      -----------------------------------------------------
      Date        Name      Version           Activity                                                                              

   ############################################################*)

   REGION Control Mode
       //AUTO:Auto Mode
       #ioGraphCtrl.AUTO := #ioGraphCtrl.SUP := #iSysInface.Auto.Mode;

       //MAN:Manual Mode
       #ioGraphCtrl.MAN :=  #iSysInface.ManualMode;
       #ioGraphCtrl.OFF := #ioPM_Inface.AlarmImdilyStop OR #iSysInface.ManualMode;
       IF #iSysInface.ManualMode OR #ioPM_Inface.AlarmImdilyStop THEN
           #ioPM_Inface.InitialRun      := 0;
           #ioPM_Inface.InitialOK       := 0;
           #ioPM_Inface.WaitRunning     := 0;
           // #ioPM_Inface.Running         := 0;
           #ioPM_Inface.UnPause    := 0;
           #ioPM_Inface.ProcessComplete := 0;

       END_IF;
       //AutoRunning
       //
       // #ioPM_Inface.Running := ((#iSysInface.Auto.StartAuto AND #iSysInface.Ready) OR #iSysInface.Auto.Running)
       // AND AND NOT "ST10_Sys".Auto.RunningOver 

       IF NOT #iSysInface.ManualMode AND #iSysInface.SysRun AND #ioPM_Inface.InitialOK AND NOT #ioPM_Inface.Alarm
           AND NOT #ioPM_Inface.AlarmImdilyStop AND NOT #iSysInface.Auto.RunningPause THEN
           IF #iSysInface.Auto.StartAuto AND #iSysInface.Ready AND  NOT  #ioPM_Inface.Running  THEN
               #ioPM_Inface.Running := 1;
           END_IF;
       ELSE
           #ioPM_Inface.Running := 0;
       END_IF;

       //Step Num






       //TAP:StepMode
       #ioGraphCtrl.TAP := #iSysInface.Auto.StepMode;
       #ioGraphCtrl.T_PUSH := #iSysInface.Auto.StepMode AND #ioPM_Inface.SetNextStep AND NOT #sHis[0];
       #sHis[0] := #ioPM_Inface.SetNextStep;

       //INTERLOCK
       #ioGraphCtrl.LOCK    := 1;
       #ioGraphCtrl.IL_PERM := 1;
       #ioGraphCtrl.T_PERM  := 1;

   END_REGION

   REGION Initialization

       #sSetInitialDelay(IN := #iSysInface.SetInitial OR #ioPM_Inface.SetInitial,
                         PT := T#2000ms);//20221221DB

       IF #sSetInitialDelay.Q AND #iSysInface.SysRun AND NOT #iSysInface.ManualMode THEN

           IF NOT #sHis[1] THEN
               //     #oStatus.Initializing := TRUE;
               //     #oStatus.InitializeOK := 0;
               //     #oStatus.WaitRunning := 0;
               //     #oStatus.Running := 0;
               //     #oStatus.RunningPause := 0;
               //     #oStatus.RunningFinished := 0;
               #ioGraphCtrl.INIT := #sSetInitialDelay.Q;
           END_IF;

       ELSE
           #ioGraphCtrl.INIT := 0;
       END_IF;
       #sHis[1] := #sSetInitialDelay.Q;
   END_REGION

   REGION Reset
       //
       #ioGraphCtrl.ACK := #iSysInface.Reset;


   END_REGION

   REGION Running and Pause(Halt)
       #ioGraphCtrl.HALT :=(#ioPM_Inface.InitialOK AND NOT #ioPM_Inface.Running )  OR   #ioPM_Inface.Alarm OR #ioPM_Inface.AlarmImdilyStop ; //#ioPM_Inface.UnPause  NOT #iSysInface.Auto.RunningPause
       #ioGraphCtrl.OPS_ZERO := #iSysInface.ManualMode OR NOT #iSysInface.SysRun OR #ioPM_Inface.AlarmImdilyStop ;
       #ioGraphCtrl.TMS_HALT := #iSysInface.ManualMode OR NOT #iSysInface.SysRun OR #ioPM_Inface.AlarmImdilyStop;
   END_REGION


   #S_NEXT_Delay[0](PT := t#3s,
                 IN := #ioGraphCtrl.S_NEXT);

   IF #S_NEXT_Delay[0].Q THEN
       #ioGraphCtrl.S_NEXT := 0;

   END_IF;

   #S_NEXT_Delay[1](PT := t#3s,
                    IN := NOT #ioGraphCtrl.S_NEXT);

   IF #S_NEXT_Delay[1].Q THEN
       #ioGraphCtrl.S_NEXT := 1;
   END_IF;
END_FUNCTION_BLOCK

FUNCTION_BLOCK "ST10_Flow2_A1TableUnloading"   // FB1072, GRAPH
// stored: AcknowledgeErrorsRequired false, AutoNumber false, GraphVersion 6.0, InitialValuesAcquisition false, SetENOAutomatically false
   // inherited from GRAPH_BASE
   VAR_INPUT
      iSysInface : "RCS_SysComInterface_V1";
   END_VAR
   VAR_IN_OUT
      ioPM_Inface : "RCS_PMInterface_V1";
      ioStatus : Int;
   END_VAR
   VAR
      sCtrlMode { S7_SetPoint := 'True'} : "SysFlowCtrlGraph";
      sUpdMES_Data : Bool;   // 更新MES数据
      工件放行中 : Bool;
      前站站号 { ExternalAccessible := 'False'; ExternalVisible := 'False'; ExternalWritable := 'False'} : UInt;
      本站站号 { ExternalAccessible := 'False'; ExternalVisible := 'False'; ExternalWritable := 'False'} : UInt;
      弹窗Temp : Array[1..10] of Int;
      AlarmID : Int;
      TON { S7_SetPoint := 'True'} : Array[0..10] of TON_TIME;
      TOF { S7_SetPoint := 'True'} : Array[0..10] of TOF_TIME;
      sUP { S7_SetPoint := 'True'} : Array[0..10] of Bool;
      更新RFID完成 : Bool;
   END_VAR
   VAR_TEMP
      Tempresult : USInt;
      本站站号乘10 : UInt;
   END_VAR
   // // TON[0] : 托盘流入1托盘到位传感器 / iA-Rotating product Check
   // // TON[1] : 托盘流入1托盘到位传感器
   // // TON[2] : 托盘流入1产品有无传感器
   // // TON[3] : 托盘流入1产品有无传感器
   // // TON[4] : 托盘流入1姿态检测光电2
   // // TON[5] : 托盘流入1姿态检测光电3
   // // TON[0].Q : 托盘流入1托盘到位 / iA-Rotating product Check
   // // TON[1].Q : 托盘流入1托盘无
   // // TON[2].Q : 托盘流入1有产品
   // // TON[3].Q : 托盘流入1无产品
   // // TON[4].Q : 托盘流入1姿态检测光电2
   // // TON[5].Q : 托盘流入1姿态检测光电3
   // // TOF[1] : iA-Rotating product Check
BEGIN
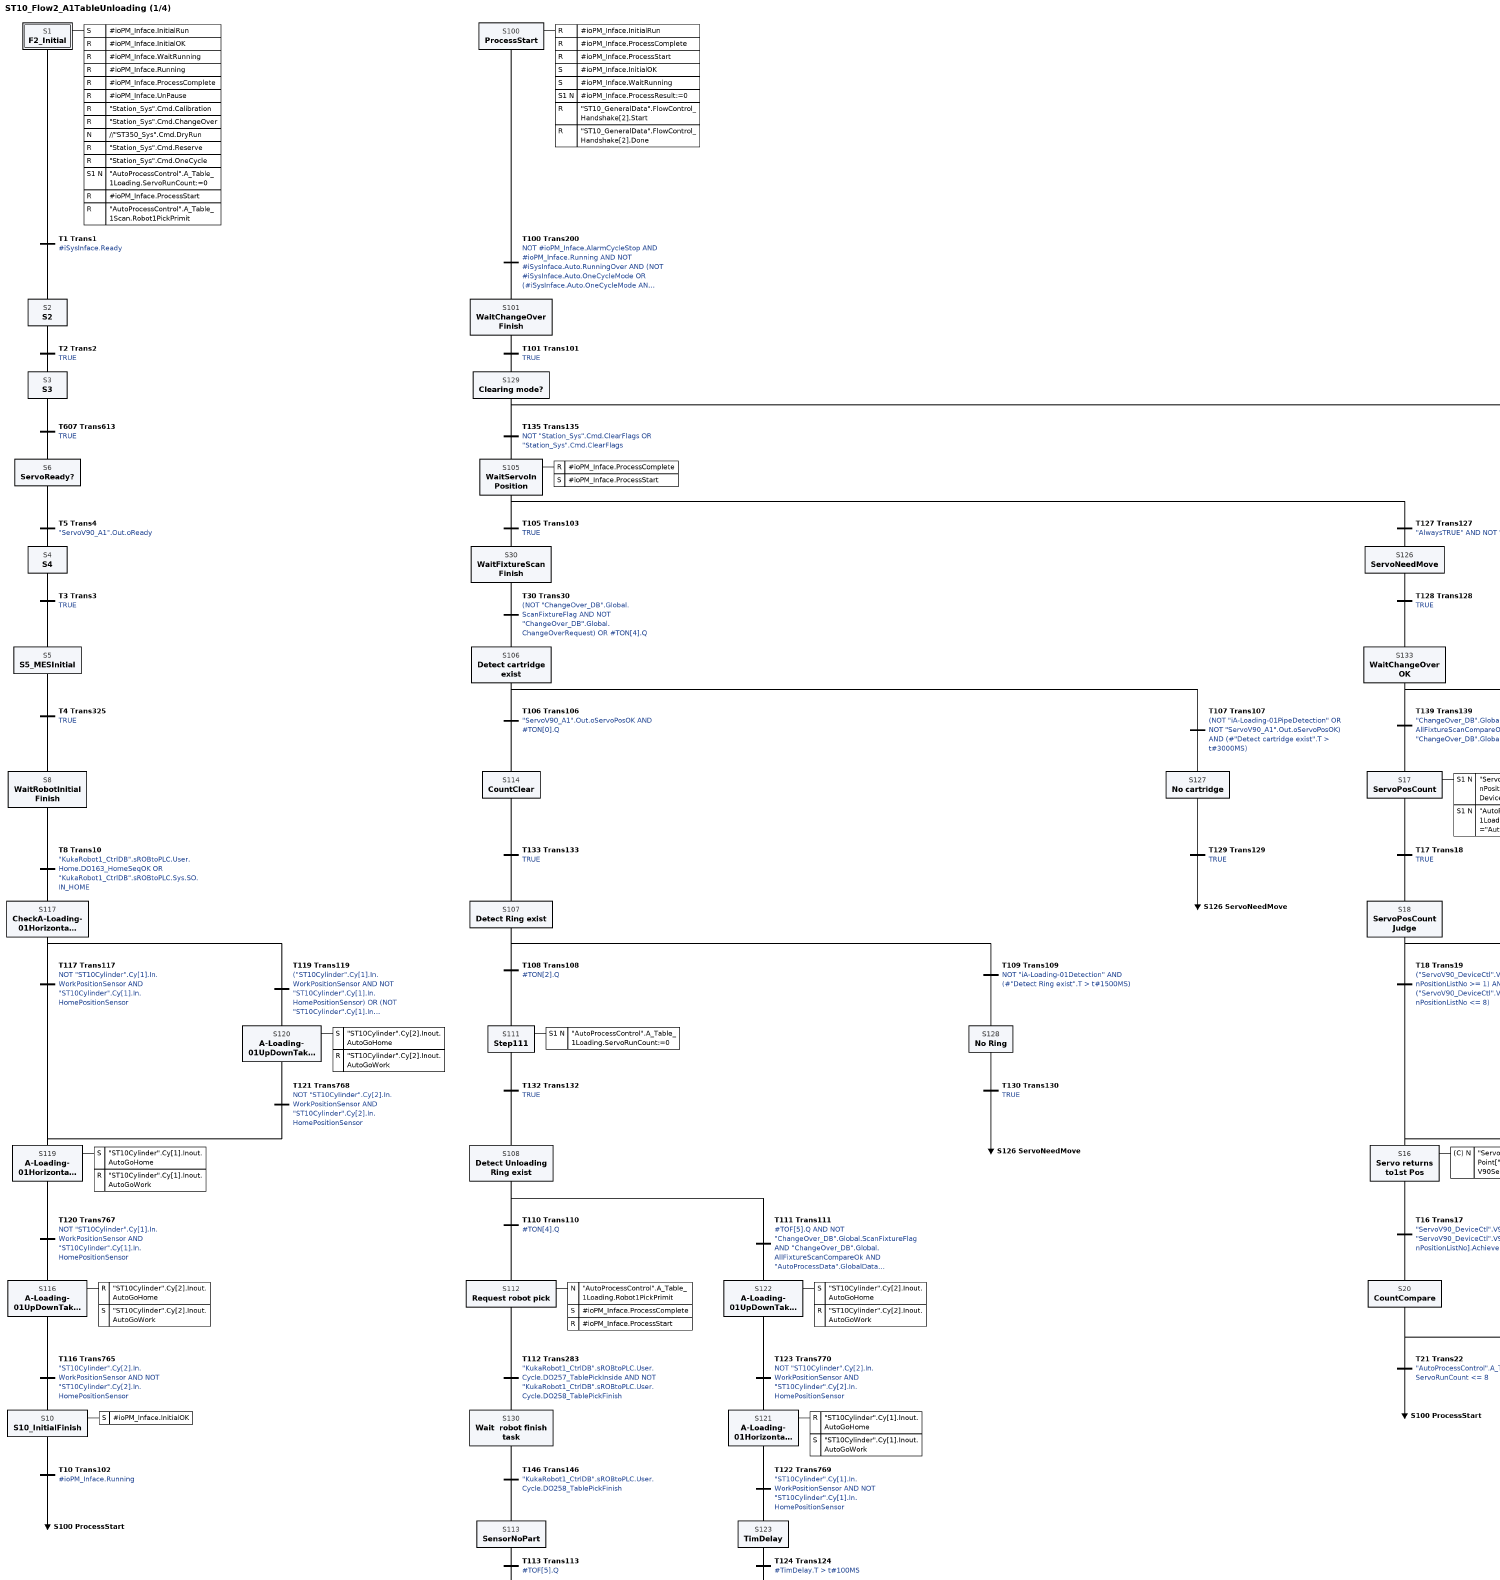
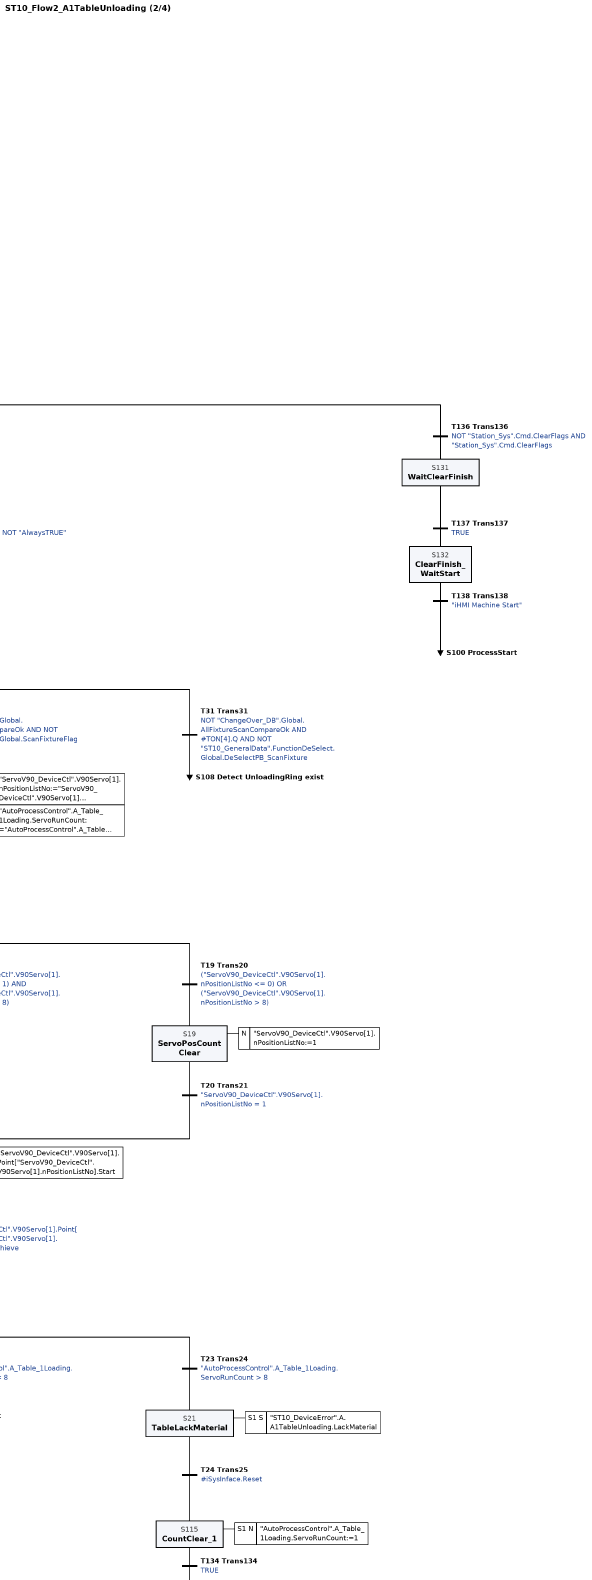
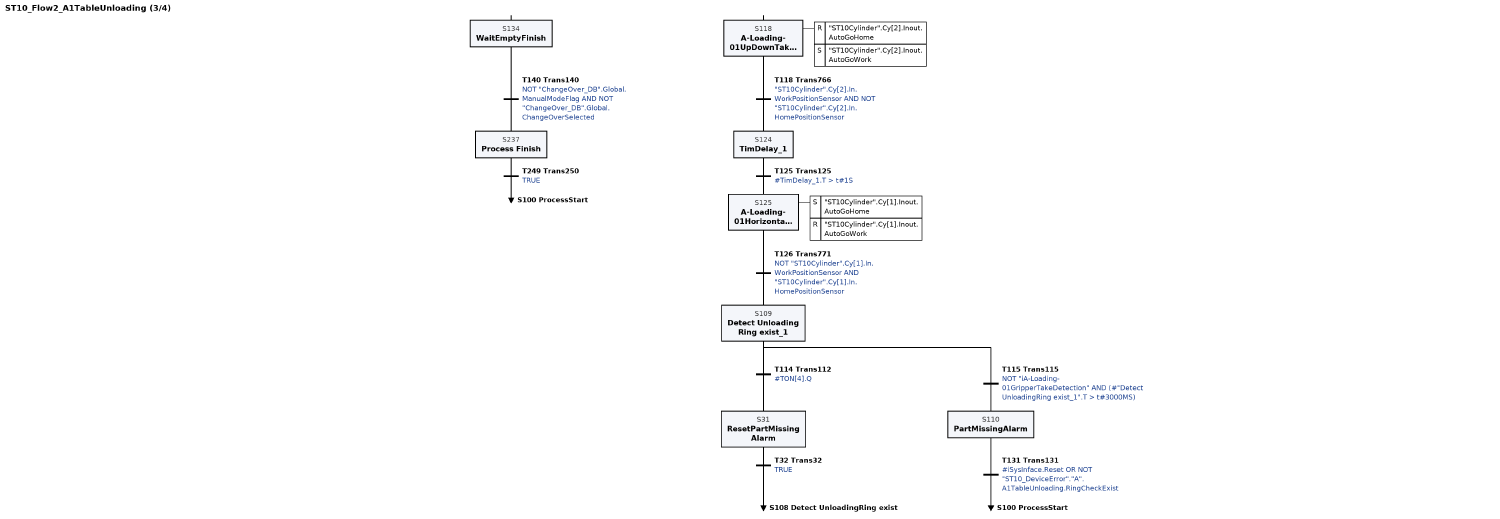
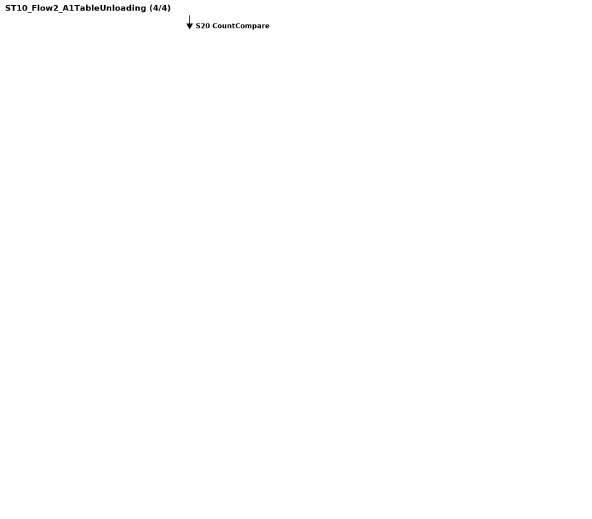
   // permanent pre-instructions
   NETWORK 1
      #TON[10].TON(IN := "AlwaysTRUE" AND "Station_Sys".Alarm.ImmediatelyStop, PT := T#300ms);
      #ioPM_Inface.AlarmImdilyStop := #TON[10].Q;
      #ioPM_Inface.AlarmCycleStop := "AlwaysTRUE" AND "Station_Sys".Alarm.CycleStop;
   NETWORK 2
      IF NOT False THEN
          #sCtrlMode(iSysInface := #iSysInface, ioPM_Inface := #ioPM_Inface, ioGraphCtrl := #RT_DATA.MOP);   // "SysFlowCtrlGraph"
      END_IF;
   NETWORK 3
      #TON[0].TON(IN := "AlwaysTRUE" AND "iA-Loading-01PipeDetection", PT := t#500ms);   // 工位11有托盘
      #TOF[1].TOF(IN := "AlwaysTRUE" AND NOT "iA-Loading-01PipeDetection", PT := T#300ms);   // 工位无托盘
      #TON[2].TON(IN := "AlwaysTRUE" AND "iA-Loading-01Detection", PT := T#300ms);
      #TOF[3].TOF(IN := "AlwaysTRUE" AND NOT "iA-Loading-01Detection", PT := T#300ms);
      #TON[4].TON(IN := "AlwaysTRUE" AND "iA-Loading-01GripperTakeDetection", PT := T#300ms);
      #TOF[5].TOF(IN := "AlwaysTRUE" AND NOT "iA-Loading-01GripperTakeDetection", PT := T#300ms);
   NETWORK 4
      #前站站号 := 345;
      #本站站号 := 350;

   // sequencer 1: S01-S99 初始化 / S01-S99 Initial
   INITIAL_STEP F2_Initial:   // S1, max time T#10S, warning time T#7S
              S    #ioPM_Inface.InitialRun
              R    #ioPM_Inface.InitialOK
              R    #ioPM_Inface.WaitRunning
              R    #ioPM_Inface.Running
              R    #ioPM_Inface.ProcessComplete
              R    #ioPM_Inface.UnPause
              R    "Station_Sys".Cmd.Calibration
              R    "Station_Sys".Cmd.ChangeOver
                   //"ST350_Sys".Cmd.DryRun
              R    "Station_Sys".Cmd.Reserve
              R    "Station_Sys".Cmd.OneCycle
          S1  N    "AutoProcessControl".A_Table_1Loading.ServoRunCount:=0
              R    #ioPM_Inface.ProcessStart
              R    "AutoProcessControl".A_Table_1Scan.Robot1PickPrimit
              R    "AutoProcessControl".A_Table_1Loading.Robot1PickPrimit
              R    "AutoProcessControl".A_Table_2Scan.Robot3PickPrimit
              R    "AutoProcessControl".A_Table_2Loading.Robot3PickPrimit
              R    "AutoProcessControl".A_ScanRotary.Robot1PickPrimit
              R    "AutoProcessControl".A_ScanRotary.Robot1PutPrimit
              R    "AutoProcessControl".H_ShafeLine.Robot1PickPrimit
              R    "AutoProcessControl".J_MagnetLine.Robot2PickPrimit
              R    "AutoProcessControl".K_ShafeLine.Robot2PickPrimit
              R    "AutoProcessControl".L_ShafeLine.Robot3PutPrimit
   END_STEP
   TRANSITION Trans1 FROM F2_Initial TO S2   // T1
      := #iSysInface.Ready;
   END_TRANSITION
   STEP S2:   // S2, max time T#10S, warning time T#7S
   END_STEP
   TRANSITION Trans2 FROM S2 TO S3   // T2
      := TRUE;
   END_TRANSITION
   STEP S4:   // S4, max time T#10S, warning time T#7S
   END_STEP
   TRANSITION Trans3 FROM S4 TO S5_MESInitial   // T3
      := TRUE;
   END_TRANSITION
   STEP S5_MESInitial:   // S5, max time T#10S, warning time T#7S
   END_STEP
   TRANSITION Trans325 FROM S5_MESInitial TO WaitRobotInitialFinish   // T4
      := TRUE;
   END_TRANSITION
   STEP S10_InitialFinish:   // S10, max time T#10S, warning time T#7S
              S    #ioPM_Inface.InitialOK
   END_STEP
   TRANSITION Trans102 FROM S10_InitialFinish TO ProcessStart   // T10, jump
      := #ioPM_Inface.Running;
   END_TRANSITION
   STEP S3:   // S3, max time T#10S, warning time T#7S
   END_STEP
   TRANSITION Trans613 FROM S3 TO "ServoReady?"   // T607
      := TRUE;
   END_TRANSITION
   STEP WaitRobotInitialFinish:   // S8, max time T#10S, warning time T#7S
   END_STEP
   TRANSITION Trans10 FROM WaitRobotInitialFinish TO "CheckA-Loading-01HorizontalCylindePos"   // T8
      := "KukaRobot1_CtrlDB".sROBtoPLC.User.Home.DO163_HomeSeqOK OR "KukaRobot1_CtrlDB".sROBtoPLC.Sys.SO.IN_HOME;
   END_TRANSITION
   STEP "A-Loading-01UpDownTakeCylinderToHP_2":   // S120, max time T#10S, warning time T#7S
              S    "ST10Cylinder".Cy[2].Inout.AutoGoHome
              R    "ST10Cylinder".Cy[2].Inout.AutoGoWork
   END_STEP
   TRANSITION Trans768 FROM "A-Loading-01UpDownTakeCylinderToHP_2" TO "A-Loading-01HorizontalCylinderToHP"   // T121
      := NOT "ST10Cylinder".Cy[2].In.WorkPositionSensor AND "ST10Cylinder".Cy[2].In.HomePositionSensor;
   END_TRANSITION
   STEP "CheckA-Loading-01HorizontalCylindePos":   // S117, max time T#10S, warning time T#7S
   END_STEP
   TRANSITION Trans117 FROM "CheckA-Loading-01HorizontalCylindePos" TO "A-Loading-01HorizontalCylinderToHP"   // T117
      := NOT "ST10Cylinder".Cy[1].In.WorkPositionSensor AND "ST10Cylinder".Cy[1].In.HomePositionSensor;
   END_TRANSITION
   TRANSITION Trans119 FROM "CheckA-Loading-01HorizontalCylindePos" TO "A-Loading-01UpDownTakeCylinderToHP_2"   // T119
      := ("ST10Cylinder".Cy[1].In.WorkPositionSensor AND NOT "ST10Cylinder".Cy[1].In.HomePositionSensor) OR (NOT "ST10Cylinder".Cy[1].In.WorkPositionSensor AND NOT "ST10Cylinder".Cy[1].In.HomePositionSensor);
   END_TRANSITION
   STEP "A-Loading-01HorizontalCylinderToHP":   // S119, max time T#10S, warning time T#7S
              S    "ST10Cylinder".Cy[1].Inout.AutoGoHome
              R    "ST10Cylinder".Cy[1].Inout.AutoGoWork
   END_STEP
   TRANSITION Trans767 FROM "A-Loading-01HorizontalCylinderToHP" TO "A-Loading-01UpDownTakeCylinderToWP"   // T120
      := NOT "ST10Cylinder".Cy[1].In.WorkPositionSensor AND "ST10Cylinder".Cy[1].In.HomePositionSensor;
   END_TRANSITION
   STEP "A-Loading-01UpDownTakeCylinderToWP":   // S116, max time T#10S, warning time T#7S
              R    "ST10Cylinder".Cy[2].Inout.AutoGoHome
              S    "ST10Cylinder".Cy[2].Inout.AutoGoWork
   END_STEP
   TRANSITION Trans765 FROM "A-Loading-01UpDownTakeCylinderToWP" TO S10_InitialFinish   // T116
      := "ST10Cylinder".Cy[2].In.WorkPositionSensor AND NOT "ST10Cylinder".Cy[2].In.HomePositionSensor;
   END_TRANSITION
   STEP "ServoReady?":   // S6, max time T#10S, warning time T#7S
   END_STEP
   TRANSITION Trans4 FROM "ServoReady?" TO S4   // T5
      := "ServoV90_A1".Out.oReady;
   END_TRANSITION

   // sequencer 2: S100-S199 等待到位 / S100-S199 CheckSysStatus
   STEP "A-Loading-01HorizontalCylinderToWP_1":   // S121, max time T#10S, warning time T#7S
              R    "ST10Cylinder".Cy[1].Inout.AutoGoHome
              S    "ST10Cylinder".Cy[1].Inout.AutoGoWork
   END_STEP
   TRANSITION Trans769 FROM "A-Loading-01HorizontalCylinderToWP_1" TO TimDelay   // T122
      := "ST10Cylinder".Cy[1].In.WorkPositionSensor AND NOT "ST10Cylinder".Cy[1].In.HomePositionSensor;
   END_TRANSITION
   STEP "A-Loading-01UpDownTakeCylinderToHP3":   // S122, max time T#10S, warning time T#7S
              S    "ST10Cylinder".Cy[2].Inout.AutoGoHome
              R    "ST10Cylinder".Cy[2].Inout.AutoGoWork
   END_STEP
   TRANSITION Trans770 FROM "A-Loading-01UpDownTakeCylinderToHP3" TO "A-Loading-01HorizontalCylinderToWP_1"   // T123
      := NOT "ST10Cylinder".Cy[2].In.WorkPositionSensor AND "ST10Cylinder".Cy[2].In.HomePositionSensor;
   END_TRANSITION
   STEP TimDelay:   // S123, max time T#10S, warning time T#7S
   END_STEP
   TRANSITION Trans124 FROM TimDelay TO "A-Loading-01UpDownTakeCylinderToWP_1"   // T124
      := #TimDelay.T > t#100MS;
   END_TRANSITION
   STEP SensorNoPart:   // S113, max time T#10S, warning time T#7S
   END_STEP
   TRANSITION Trans113 FROM SensorNoPart TO WaitEmptyFinish   // T113
      := #TOF[5].Q;
   END_TRANSITION
   STEP ProcessStart:   // S100, max time T#10S, warning time T#7S
      // 自动等待开始运行
              R    #ioPM_Inface.InitialRun
              R    #ioPM_Inface.ProcessComplete
              R    #ioPM_Inface.ProcessStart
              S    #ioPM_Inface.InitialOK
              S    #ioPM_Inface.WaitRunning
          S1  N    #ioPM_Inface.ProcessResult:=0
              R    "ST10_GeneralData".FlowControl_Handshake[2].Start
              R    "ST10_GeneralData".FlowControl_Handshake[2].Done
   END_STEP
   TRANSITION Trans200 FROM ProcessStart TO WaitChangeOverFinish   // T100
      := NOT #ioPM_Inface.AlarmCycleStop AND #ioPM_Inface.Running AND NOT #iSysInface.Auto.RunningOver AND (NOT #iSysInface.Auto.OneCycleMode OR (#iSysInface.Auto.OneCycleMode AND #ioPM_Inface.TriggerOneCycle));
   END_TRANSITION
   STEP TimDelay_1:   // S124, max time T#10S, warning time T#7S
   END_STEP
   TRANSITION Trans125 FROM TimDelay_1 TO "A-Loading-01HorizontalCylinderToHP_1"   // T125
      := #TimDelay_1.T > t#1S;
   END_TRANSITION
   STEP "Process Finish":   // S237, max time T#10S, warning time T#7S
   END_STEP
   TRANSITION Trans250 FROM "Process Finish" TO ProcessStart   // T249, jump
      := TRUE;
   END_TRANSITION
   STEP "A-Loading-01HorizontalCylinderToHP_1":   // S125, max time T#10S, warning time T#7S
              S    "ST10Cylinder".Cy[1].Inout.AutoGoHome
              R    "ST10Cylinder".Cy[1].Inout.AutoGoWork
   END_STEP
   TRANSITION Trans771 FROM "A-Loading-01HorizontalCylinderToHP_1" TO "Detect UnloadingRing exist_1"   // T126
      := NOT "ST10Cylinder".Cy[1].In.WorkPositionSensor AND "ST10Cylinder".Cy[1].In.HomePositionSensor;
   END_TRANSITION
   STEP "No cartridge":   // S127, max time T#10S, warning time T#7S
   END_STEP
   TRANSITION Trans129 FROM "No cartridge" TO ServoNeedMove   // T129, jump
      := TRUE;
   END_TRANSITION
   STEP "A-Loading-01UpDownTakeCylinderToWP_1":   // S118, max time T#10S, warning time T#7S
              R    "ST10Cylinder".Cy[2].Inout.AutoGoHome
              S    "ST10Cylinder".Cy[2].Inout.AutoGoWork
   END_STEP
   TRANSITION Trans766 FROM "A-Loading-01UpDownTakeCylinderToWP_1" TO TimDelay_1   // T118
      := "ST10Cylinder".Cy[2].In.WorkPositionSensor AND NOT "ST10Cylinder".Cy[2].In.HomePositionSensor;
   END_TRANSITION
   STEP ServoNeedMove:   // S126, max time T#10S, warning time T#7S
   END_STEP
   TRANSITION Trans128 FROM ServoNeedMove TO WaitChangeOverOK   // T128
      := TRUE;
   END_TRANSITION
   STEP WaitChangeOverFinish:   // S101, max time T#10S, warning time T#7S
   END_STEP
   TRANSITION Trans101 FROM WaitChangeOverFinish TO "Clearing mode?"   // T101
      := TRUE;
   END_TRANSITION
   STEP WaitServoInPosition:   // S105, max time T#10S, warning time T#7S
              R    #ioPM_Inface.ProcessComplete
              S    #ioPM_Inface.ProcessStart
   END_STEP
   TRANSITION Trans103 FROM WaitServoInPosition TO WaitFixtureScanFinish   // T105
      := TRUE;
   END_TRANSITION
   TRANSITION Trans127 FROM WaitServoInPosition TO ServoNeedMove   // T127
      := "AlwaysTRUE" AND NOT "AlwaysTRUE";
   END_TRANSITION
   STEP "Detect cartridge exist":   // S106, max time T#10S, warning time T#7S
   END_STEP
   TRANSITION Trans106 FROM "Detect cartridge exist" TO CountClear   // T106
      := "ServoV90_A1".Out.oServoPosOK AND #TON[0].Q;
   END_TRANSITION
   TRANSITION Trans107 FROM "Detect cartridge exist" TO "No cartridge"   // T107
      := (NOT "iA-Loading-01PipeDetection" OR NOT "ServoV90_A1".Out.oServoPosOK) AND (#"Detect cartridge exist".T > t#3000MS);
   END_TRANSITION
   STEP "Detect UnloadingRing exist":   // S108, max time T#10S, warning time T#7S
   END_STEP
   TRANSITION Trans110 FROM "Detect UnloadingRing exist" TO "Request robot pick"   // T110
      := #TON[4].Q;
   END_TRANSITION
   TRANSITION Trans111 FROM "Detect UnloadingRing exist" TO "A-Loading-01UpDownTakeCylinderToHP3"   // T111
      := #TOF[5].Q AND NOT "ChangeOver_DB".Global.ScanFixtureFlag AND "ChangeOver_DB".Global.AllFixtureScanCompareOk AND "AutoProcessData".GlobalData.Table1CodeOKFlag;
   END_TRANSITION
   STEP "Detect Ring exist":   // S107, max time T#10S, warning time T#7S
   END_STEP
   TRANSITION Trans108 FROM "Detect Ring exist" TO Step111   // T108
      := #TON[2].Q;
   END_TRANSITION
   TRANSITION Trans109 FROM "Detect Ring exist" TO "No Ring"   // T109
      := NOT "iA-Loading-01Detection" AND (#"Detect Ring exist".T > t#1500MS);
   END_TRANSITION
   STEP "Wait  robot finish task":   // S130, max time T#10S, warning time T#7S
   END_STEP
   TRANSITION Trans146 FROM "Wait  robot finish task" TO SensorNoPart   // T146
      := "KukaRobot1_CtrlDB".sROBtoPLC.User.Cycle.DO258_TablePickFinish;
   END_TRANSITION
   STEP "Request robot pick":   // S112, max time T#10S, warning time T#7S
              N    "AutoProcessControl".A_Table_1Loading.Robot1PickPrimit
              S    #ioPM_Inface.ProcessComplete
              R    #ioPM_Inface.ProcessStart
   END_STEP
   TRANSITION Trans283 FROM "Request robot pick" TO "Wait  robot finish task"   // T112
      := "KukaRobot1_CtrlDB".sROBtoPLC.User.Cycle.DO257_TablePickInside AND NOT "KukaRobot1_CtrlDB".sROBtoPLC.User.Cycle.DO258_TablePickFinish;
   END_TRANSITION
   STEP "No Ring":   // S128, max time T#10S, warning time T#7S
   END_STEP
   TRANSITION Trans130 FROM "No Ring" TO ServoNeedMove   // T130, jump
      := TRUE;
   END_TRANSITION
   STEP "Detect UnloadingRing exist_1":   // S109, max time T#10S, warning time T#7S
   END_STEP
   TRANSITION Trans112 FROM "Detect UnloadingRing exist_1" TO ResetPartMissingAlarm   // T114
      := #TON[4].Q;
   END_TRANSITION
   TRANSITION Trans115 FROM "Detect UnloadingRing exist_1" TO PartMissingAlarm   // T115
      := NOT "iA-Loading-01GripperTakeDetection" AND (#"Detect UnloadingRing exist_1".T > t#3000MS);
   END_TRANSITION
   STEP PartMissingAlarm:   // S110, max time T#10S, warning time T#7S
   END_STEP
   TRANSITION Trans131 FROM PartMissingAlarm TO ProcessStart   // T131, jump
      := #iSysInface.Reset OR NOT "ST10_DeviceError"."A".A1TableUnloading.RingCheckExist;
   END_TRANSITION
   STEP Step111:   // S111, max time T#10S, warning time T#7S
          S1  N    "AutoProcessControl".A_Table_1Loading.ServoRunCount:=0
   END_STEP
   TRANSITION Trans132 FROM Step111 TO "Detect UnloadingRing exist"   // T132
      := TRUE;
   END_TRANSITION
   STEP CountClear:   // S114, max time T#10S, warning time T#7S
   END_STEP
   TRANSITION Trans133 FROM CountClear TO "Detect Ring exist"   // T133
      := TRUE;
   END_TRANSITION
   STEP "Servo returns to1st Pos":   // S16, max time T#10S, warning time T#7S
      interlock C := "ServoV90_A1".Out.oReady;
      (C)     N    "ServoV90_DeviceCtl".V90Servo[1].Point["ServoV90_DeviceCtl".V90Servo[1].nPositionListNo].Start
   END_STEP
   TRANSITION Trans17 FROM "Servo returns to1st Pos" TO CountCompare   // T16
      := "ServoV90_DeviceCtl".V90Servo[1].Point["ServoV90_DeviceCtl".V90Servo[1].nPositionListNo].Achieve;
   END_TRANSITION
   STEP ServoPosCount:   // S17, max time T#10S, warning time T#7S
          S1  N    "ServoV90_DeviceCtl".V90Servo[1].nPositionListNo:="ServoV90_DeviceCtl".V90Servo[1].nPositionListNo+1
          S1  N    "AutoProcessControl".A_Table_1Loading.ServoRunCount:="AutoProcessControl".A_Table_1Loading.ServoRunCount+1
   END_STEP
   TRANSITION Trans18 FROM ServoPosCount TO ServoPosCountJudge   // T17
      := TRUE;
   END_TRANSITION
   STEP ServoPosCountJudge:   // S18, max time T#10S, warning time T#7S
   END_STEP
   TRANSITION Trans19 FROM ServoPosCountJudge TO "Servo returns to1st Pos"   // T18
      := ("ServoV90_DeviceCtl".V90Servo[1].nPositionListNo >= 1) AND ("ServoV90_DeviceCtl".V90Servo[1].nPositionListNo <= 8);
   END_TRANSITION
   TRANSITION Trans20 FROM ServoPosCountJudge TO ServoPosCountClear   // T19
      := ("ServoV90_DeviceCtl".V90Servo[1].nPositionListNo <= 0) OR ("ServoV90_DeviceCtl".V90Servo[1].nPositionListNo > 8);
   END_TRANSITION
   STEP ServoPosCountClear:   // S19, max time T#10S, warning time T#7S
              N    "ServoV90_DeviceCtl".V90Servo[1].nPositionListNo:=1
   END_STEP
   TRANSITION Trans21 FROM ServoPosCountClear TO "Servo returns to1st Pos"   // T20
      := "ServoV90_DeviceCtl".V90Servo[1].nPositionListNo = 1;
   END_TRANSITION
   STEP CountCompare:   // S20, max time T#10S, warning time T#7S
   END_STEP
   TRANSITION Trans22 FROM CountCompare TO ProcessStart   // T21, jump
      := "AutoProcessControl".A_Table_1Loading.ServoRunCount <= 8;
   END_TRANSITION
   TRANSITION Trans24 FROM CountCompare TO TableLackMaterial   // T23
      := "AutoProcessControl".A_Table_1Loading.ServoRunCount > 8;
   END_TRANSITION
   STEP TableLackMaterial:   // S21, max time T#10S, warning time T#7S
          S1  S    "ST10_DeviceError".A.A1TableUnloading.LackMaterial
   END_STEP
   TRANSITION Trans25 FROM TableLackMaterial TO CountClear_1   // T24
      := #iSysInface.Reset;
   END_TRANSITION
   STEP CountClear_1:   // S115, max time T#10S, warning time T#7S
          S1  N    "AutoProcessControl".A_Table_1Loading.ServoRunCount:=1
   END_STEP
   TRANSITION Trans134 FROM CountClear_1 TO CountCompare   // T134, jump
      := TRUE;
   END_TRANSITION
   STEP "Clearing mode?":   // S129, max time T#10S, warning time T#7S
   END_STEP
   TRANSITION Trans135 FROM "Clearing mode?" TO WaitServoInPosition   // T135
      := NOT "Station_Sys".Cmd.ClearFlags OR "Station_Sys".Cmd.ClearFlags;
   END_TRANSITION
   TRANSITION Trans136 FROM "Clearing mode?" TO WaitClearFinish   // T136
      := NOT "Station_Sys".Cmd.ClearFlags AND "Station_Sys".Cmd.ClearFlags;
   END_TRANSITION
   STEP WaitClearFinish:   // S131, max time T#10S, warning time T#7S
   END_STEP
   TRANSITION Trans137 FROM WaitClearFinish TO ClearFinish_WaitStart   // T137
      := TRUE;
   END_TRANSITION
   STEP ClearFinish_WaitStart:   // S132, max time T#10S, warning time T#7S
   END_STEP
   TRANSITION Trans138 FROM ClearFinish_WaitStart TO ProcessStart   // T138, jump
      := "iHMI Machine Start";
   END_TRANSITION
   STEP WaitChangeOverOK:   // S133, max time T#10S, warning time T#7S
   END_STEP
   TRANSITION Trans139 FROM WaitChangeOverOK TO ServoPosCount   // T139
      := "ChangeOver_DB".Global.AllFixtureScanCompareOk AND NOT "ChangeOver_DB".Global.ScanFixtureFlag;
   END_TRANSITION
   TRANSITION Trans31 FROM WaitChangeOverOK TO "Detect UnloadingRing exist"   // T31, jump
      := NOT "ChangeOver_DB".Global.AllFixtureScanCompareOk AND #TON[4].Q AND NOT "ST10_GeneralData".FunctionDeSelect.Global.DeSelectPB_ScanFixture;
   END_TRANSITION
   STEP WaitEmptyFinish:   // S134, max time T#10S, warning time T#7S
   END_STEP
   TRANSITION Trans140 FROM WaitEmptyFinish TO "Process Finish"   // T140
      := NOT "ChangeOver_DB".Global.ManualModeFlag AND NOT "ChangeOver_DB".Global.ChangeOverSelected;
   END_TRANSITION
   STEP WaitFixtureScanFinish:   // S30, max time T#10S, warning time T#7S
   END_STEP
   TRANSITION Trans30 FROM WaitFixtureScanFinish TO "Detect cartridge exist"   // T30
      := (NOT "ChangeOver_DB".Global.ScanFixtureFlag AND NOT "ChangeOver_DB".Global.ChangeOverRequest) OR #TON[4].Q;
   END_TRANSITION
   STEP ResetPartMissingAlarm:   // S31, max time T#10S, warning time T#7S
   END_STEP
   TRANSITION Trans32 FROM ResetPartMissingAlarm TO "Detect UnloadingRing exist"   // T32, jump
      := TRUE;
   END_TRANSITION

   // permanent post-instructions
   NETWORK 1
      #ioPM_Inface.StepNum := #RT_DATA.S_DISPLAY;
   NETWORK 2
      IF #iSysInface.Reset THEN #AlarmID := 0; END_IF;
   NETWORK 3
      #TON[10].TON(IN := #工件放行中, PT := T#0.5S);
      IF #TON[10].Q THEN #工件放行中 := FALSE; END_IF;
END_FUNCTION_BLOCK

FUNCTION_BLOCK "ST10_Flow3_A1RotaryShaftScan"   // FB1073, GRAPH
// stored: AcknowledgeErrorsRequired false, AutoNumber false, GraphVersion 6.0, InitialValuesAcquisition false, SetENOAutomatically false
   // inherited from GRAPH_BASE
   VAR_INPUT
      iSysInface : "RCS_SysComInterface_V1";
   END_VAR
   VAR_IN_OUT
      ioPM_Inface : "RCS_PMInterface_V1";
      ioStatus : Int;
   END_VAR
   VAR
      sCtrlMode { S7_SetPoint := 'True'} : "SysFlowCtrlGraph";
      sUpdMES_Data : Bool;   // 更新MES数据
      工件放行中 : Bool;
      前站站号 { ExternalAccessible := 'False'; ExternalVisible := 'False'; ExternalWritable := 'False'} : UInt;
      本站站号 { ExternalAccessible := 'False'; ExternalVisible := 'False'; ExternalWritable := 'False'} : UInt;
      弹窗Temp : Array[1..10] of Int;
      AlarmID : Int;
      TON { S7_SetPoint := 'True'} : Array[0..10] of TON_TIME;
      TOF { S7_SetPoint := 'True'} : Array[0..10] of TOF_TIME;
      sUP { S7_SetPoint := 'True'} : Array[0..10] of Bool;
      更新RFID完成 : Bool;
   END_VAR
   VAR_TEMP
      Tempresult : USInt;
      本站站号乘10 : UInt;
   END_VAR
   // // TON[0] : 托盘流入1托盘到位传感器 / iA-Rotating product Check
   // // TON[1] : 托盘流入1托盘到位传感器
   // // TON[2] : 托盘流入1产品有无传感器
   // // TON[3] : 托盘流入1产品有无传感器
   // // TON[4] : 托盘流入1姿态检测光电2
   // // TON[5] : 托盘流入1姿态检测光电3
   // // TON[0].Q : 托盘流入1托盘到位 / iA-Rotating product Check
   // // TON[1].Q : 托盘流入1托盘无
   // // TON[2].Q : 托盘流入1有产品
   // // TON[3].Q : 托盘流入1无产品
   // // TON[4].Q : 托盘流入1姿态检测光电2
   // // TON[5].Q : 托盘流入1姿态检测光电3
   // // TOF[1] : iA-Rotating product Check
BEGIN
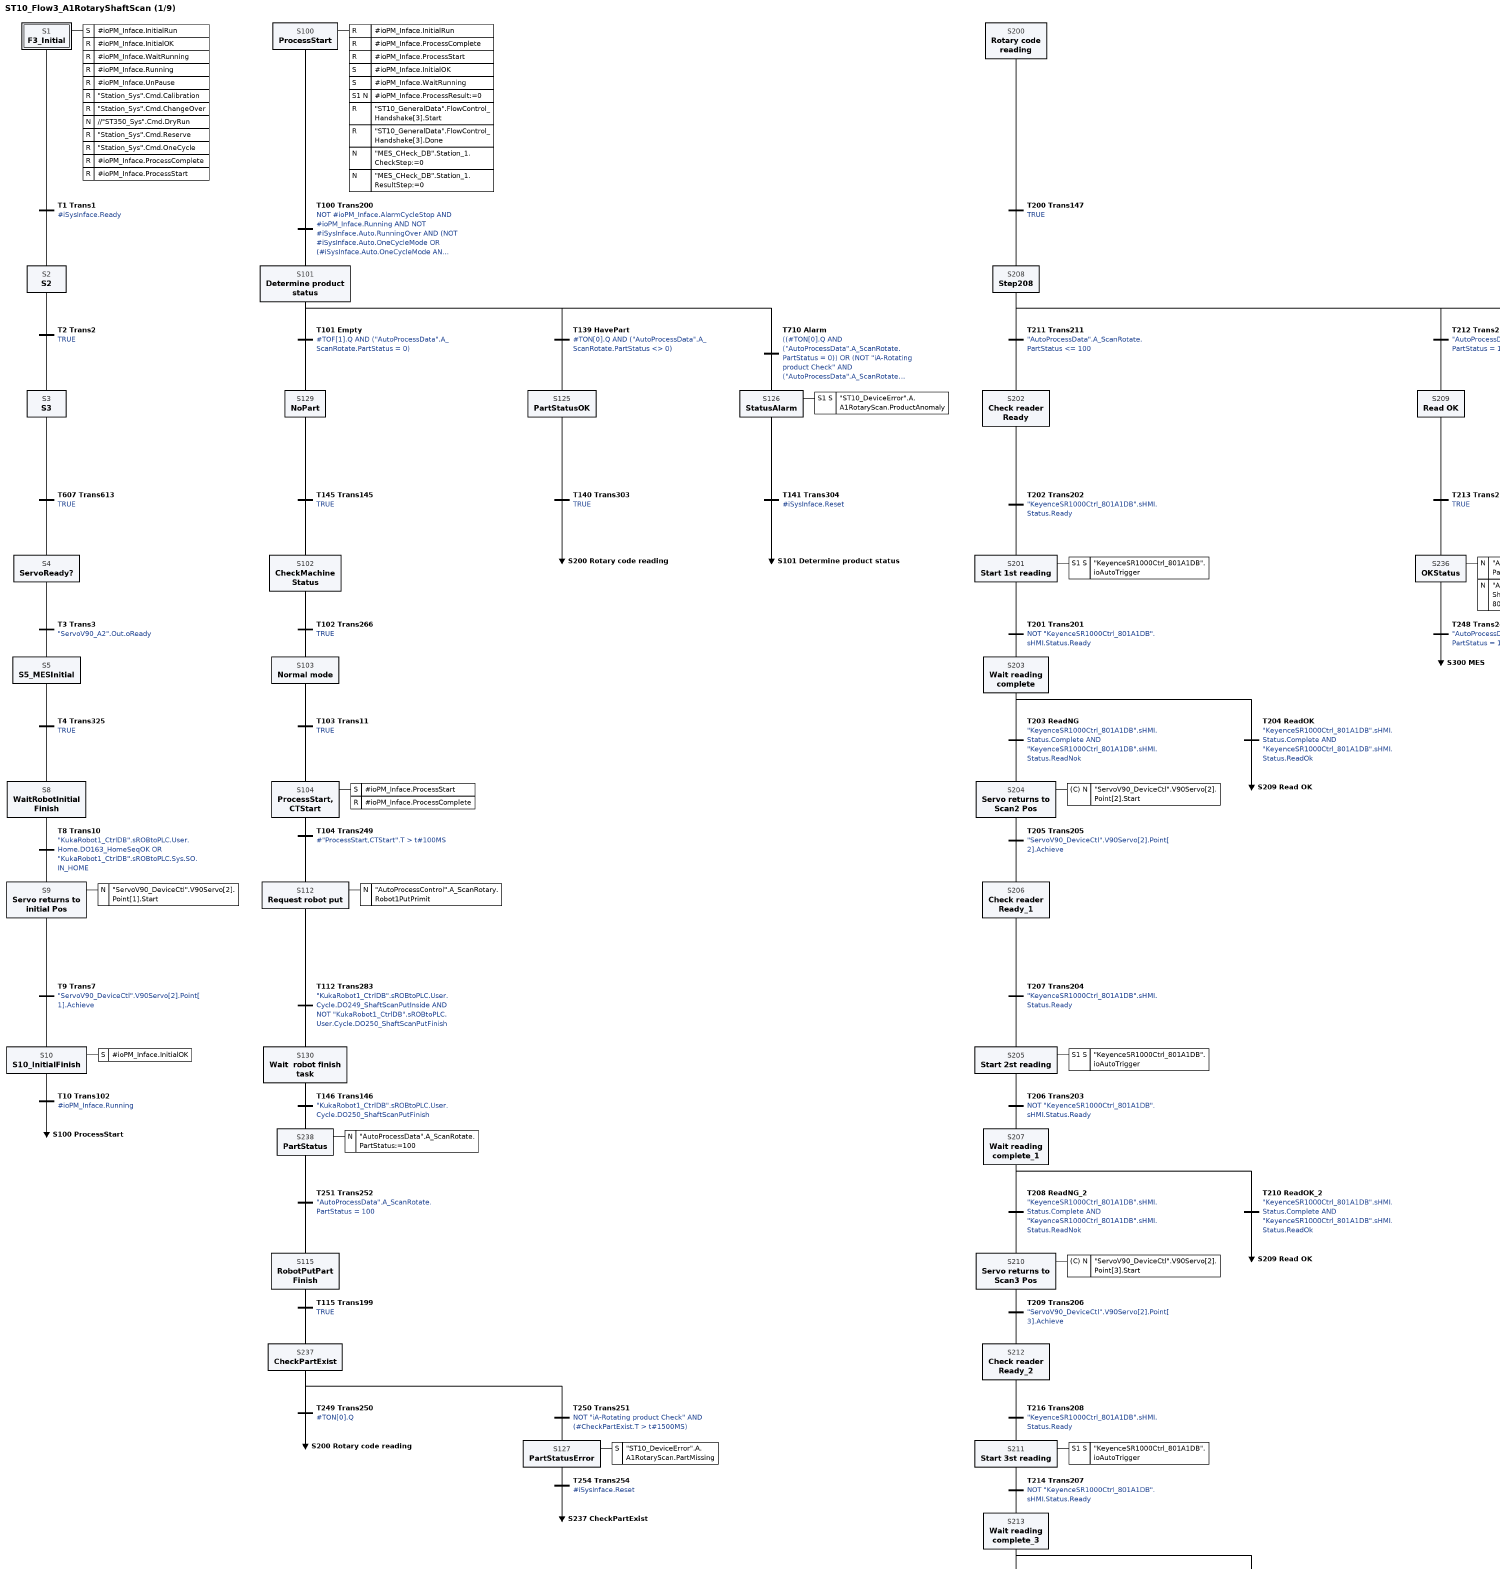
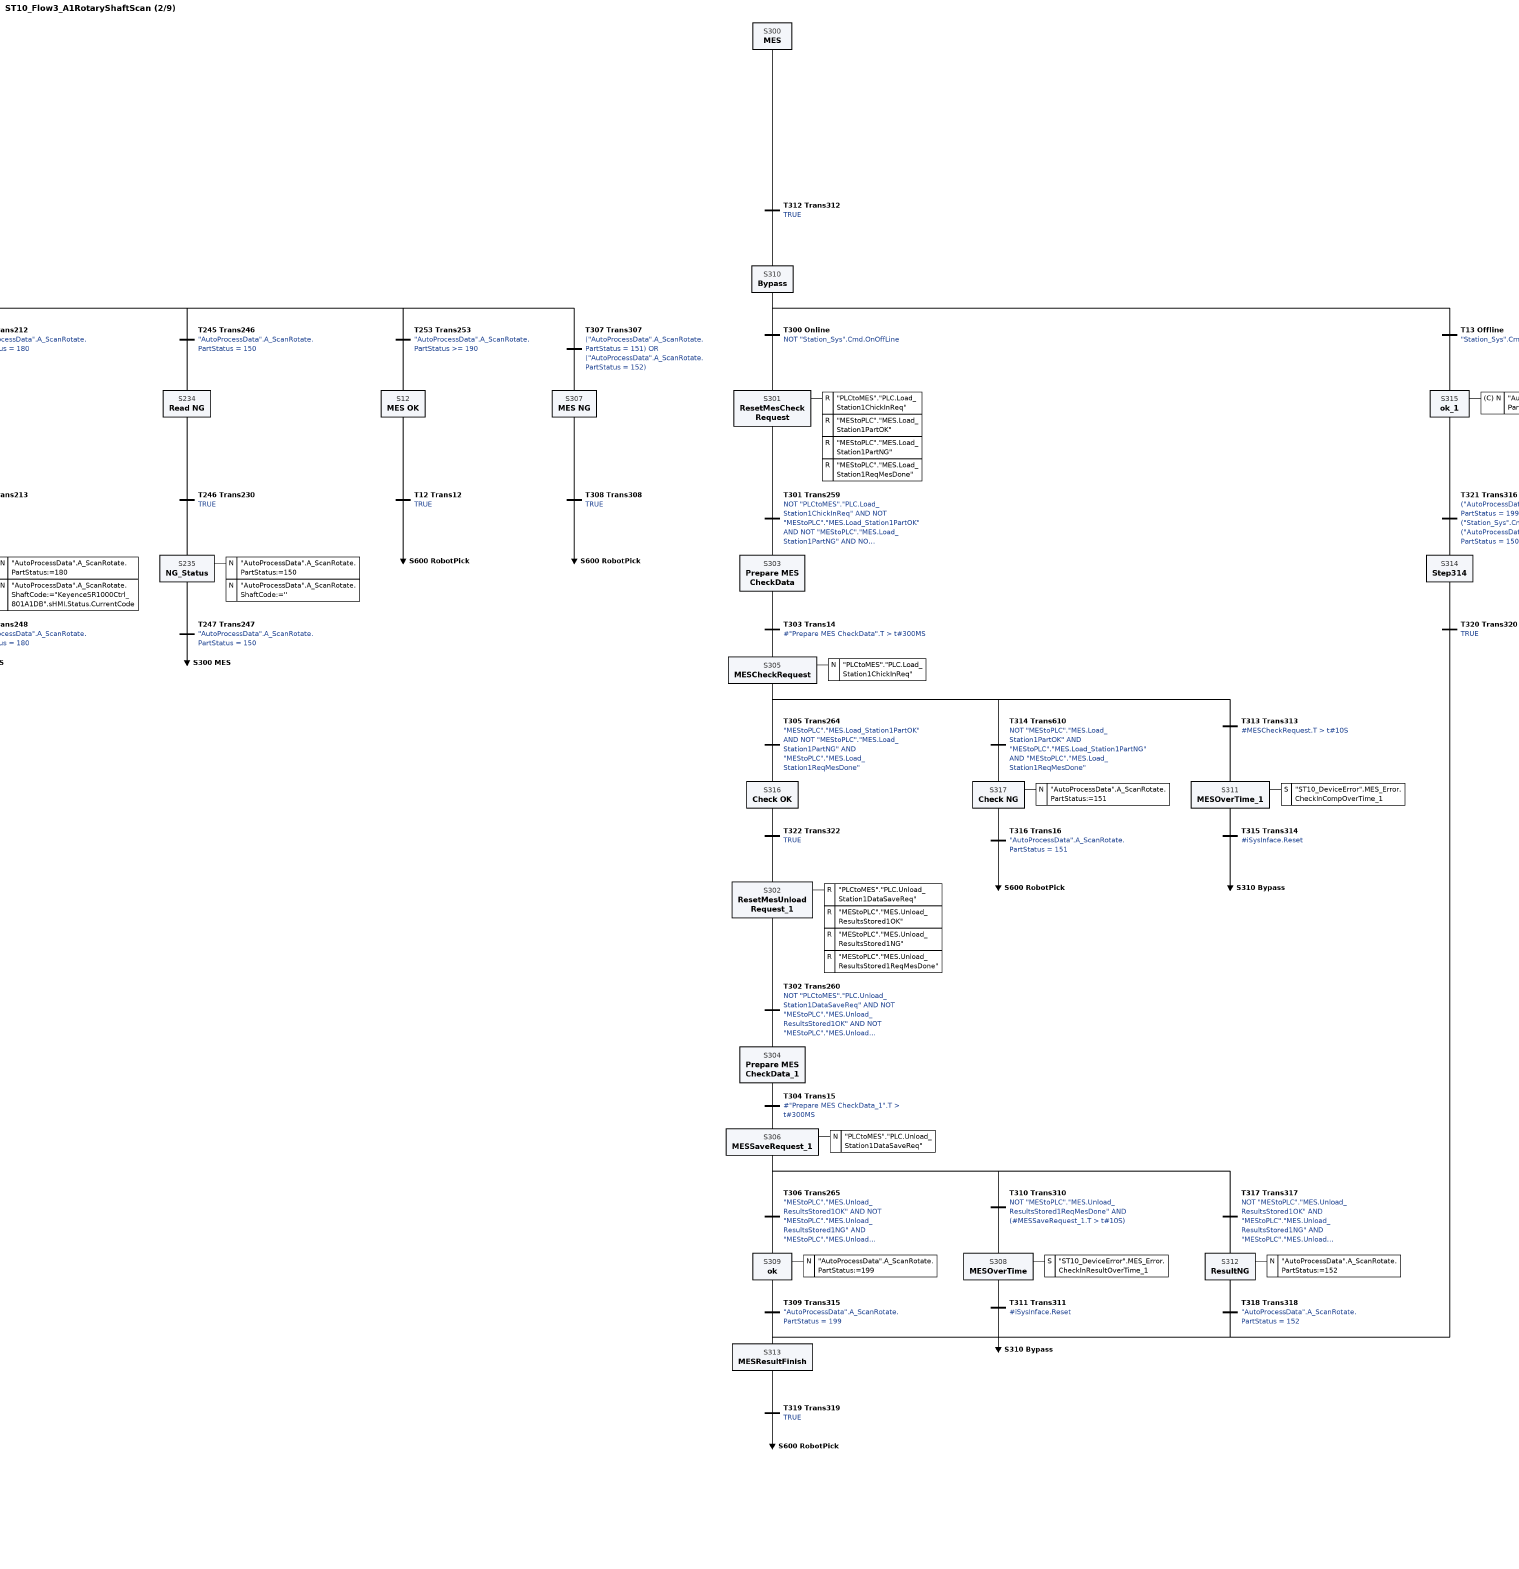
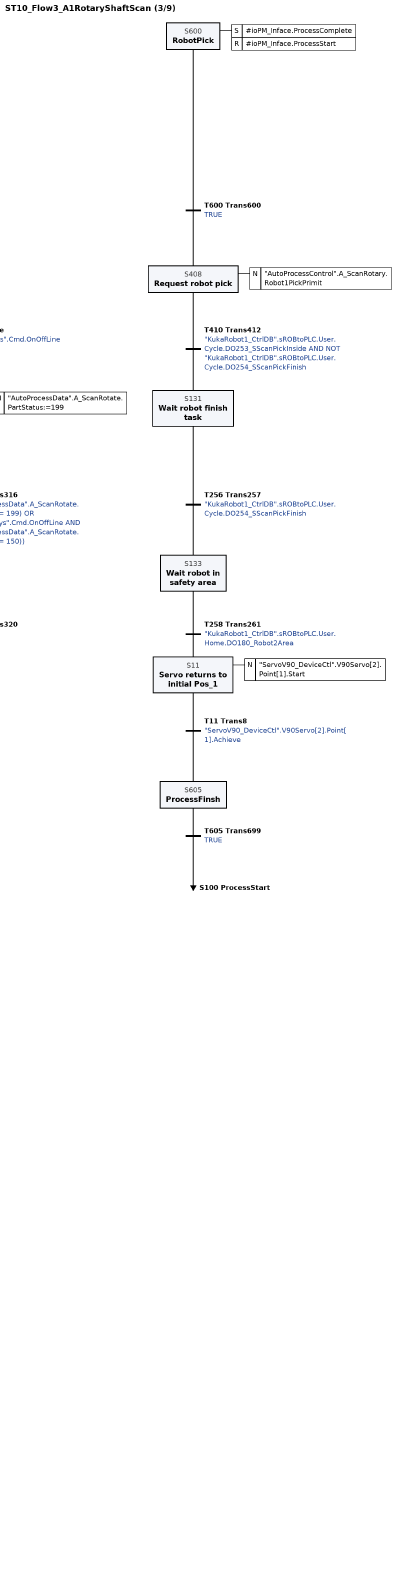
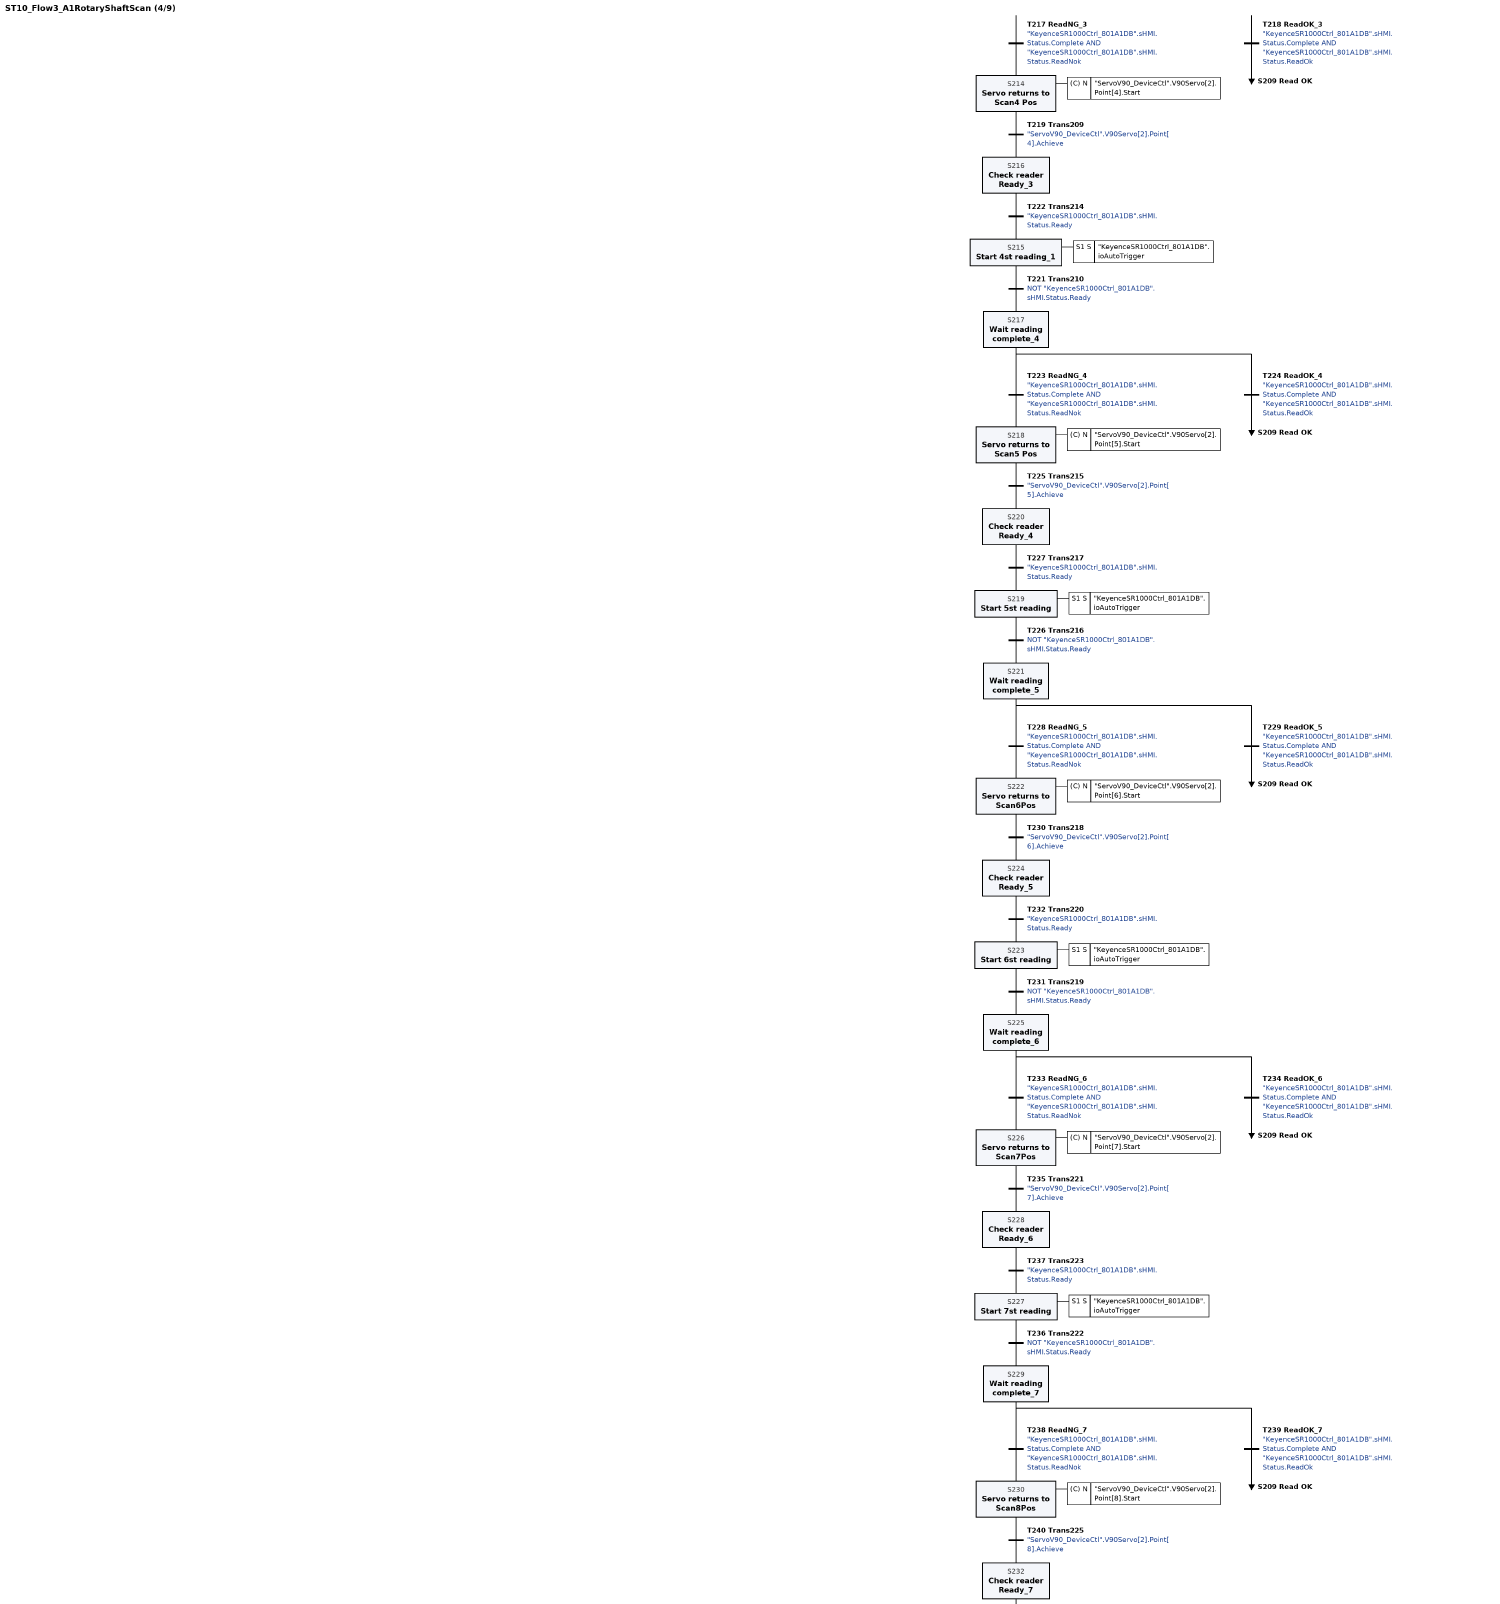
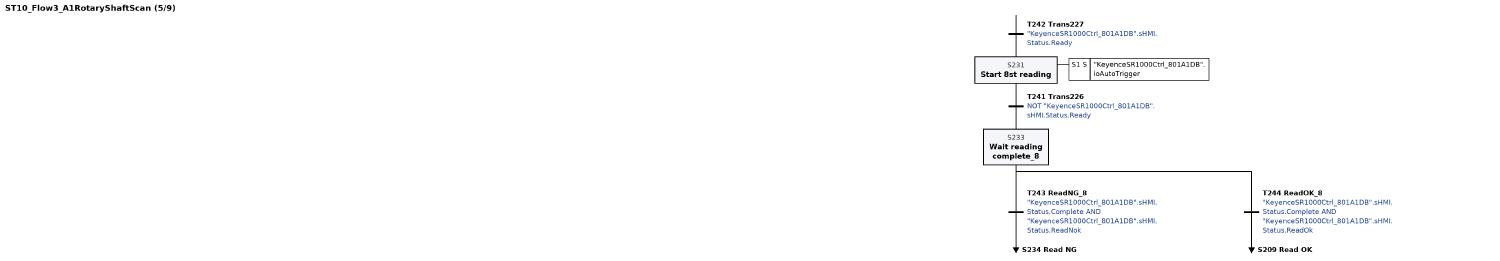
   // permanent pre-instructions
   NETWORK 1
      #TON[10].TON(IN := "AlwaysTRUE" AND "Station_Sys".Alarm.ImmediatelyStop, PT := T#300ms);
      #ioPM_Inface.AlarmImdilyStop := #TON[10].Q;
      #ioPM_Inface.AlarmCycleStop := "AlwaysTRUE" AND "Station_Sys".Alarm.CycleStop;
   NETWORK 2
      IF NOT False THEN
          #sCtrlMode(iSysInface := #iSysInface, ioPM_Inface := #ioPM_Inface, ioGraphCtrl := #RT_DATA.MOP);   // "SysFlowCtrlGraph"
      END_IF;
   NETWORK 3
      #TON[0].TON(IN := "AlwaysTRUE" AND "iA-Rotating product Check", PT := t#500ms);   // 工位11有托盘
      #TOF[1].TOF(IN := "AlwaysTRUE" AND NOT "iA-Rotating product Check", PT := T#300ms);   // 工位无托盘
      #TON[2].TON(IN := "AlwaysTRUE", PT := T#300ms);
      #TON[3].TON(IN := "AlwaysTRUE", PT := T#300ms);
      #TON[4].TON(IN := "AlwaysTRUE", PT := T#300ms);
      #TON[5].TON(IN := "AlwaysTRUE", PT := T#300ms);
   NETWORK 4
      #前站站号 := 345;
      #本站站号 := 350;

   // sequencer 1: S01-S99 初始化 / S01-S99 Initial
   INITIAL_STEP F3_Initial:   // S1, max time T#10S, warning time T#7S
              S    #ioPM_Inface.InitialRun
              R    #ioPM_Inface.InitialOK
              R    #ioPM_Inface.WaitRunning
              R    #ioPM_Inface.Running
              R    #ioPM_Inface.UnPause
              R    "Station_Sys".Cmd.Calibration
              R    "Station_Sys".Cmd.ChangeOver
                   //"ST350_Sys".Cmd.DryRun
              R    "Station_Sys".Cmd.Reserve
              R    "Station_Sys".Cmd.OneCycle
              R    #ioPM_Inface.ProcessComplete
              R    #ioPM_Inface.ProcessStart
   END_STEP
   TRANSITION Trans1 FROM F3_Initial TO S2   // T1
      := #iSysInface.Ready;
   END_TRANSITION
   STEP S2:   // S2, max time T#10S, warning time T#7S
   END_STEP
   TRANSITION Trans2 FROM S2 TO S3   // T2
      := TRUE;
   END_TRANSITION
   STEP "ServoReady?":   // S4, max time T#10S, warning time T#7S
   END_STEP
   TRANSITION Trans3 FROM "ServoReady?" TO S5_MESInitial   // T3
      := "ServoV90_A2".Out.oReady;
   END_TRANSITION
   STEP S5_MESInitial:   // S5, max time T#10S, warning time T#7S
   END_STEP
   TRANSITION Trans325 FROM S5_MESInitial TO WaitRobotInitialFinish   // T4
      := TRUE;
   END_TRANSITION
   STEP S10_InitialFinish:   // S10, max time T#10S, warning time T#7S
              S    #ioPM_Inface.InitialOK
   END_STEP
   TRANSITION Trans102 FROM S10_InitialFinish TO ProcessStart   // T10, jump
      := #ioPM_Inface.Running;
   END_TRANSITION
   STEP S3:   // S3, max time T#10S, warning time T#7S
   END_STEP
   TRANSITION Trans613 FROM S3 TO "ServoReady?"   // T607
      := TRUE;
   END_TRANSITION
   STEP WaitRobotInitialFinish:   // S8, max time T#10S, warning time T#7S
   END_STEP
   TRANSITION Trans10 FROM WaitRobotInitialFinish TO "Servo returns to initial Pos"   // T8
      := "KukaRobot1_CtrlDB".sROBtoPLC.User.Home.DO163_HomeSeqOK OR "KukaRobot1_CtrlDB".sROBtoPLC.Sys.SO.IN_HOME;
   END_TRANSITION
   STEP "Servo returns to initial Pos":   // S9, max time T#10S, warning time T#7S
              N    "ServoV90_DeviceCtl".V90Servo[2].Point[1].Start
   END_STEP
   TRANSITION Trans7 FROM "Servo returns to initial Pos" TO S10_InitialFinish   // T9
      := "ServoV90_DeviceCtl".V90Servo[2].Point[1].Achieve;
   END_TRANSITION

   // sequencer 2: S100-S199 等待到位 / S100-S199 CheckPartStatus
   STEP "Wait  robot finish task":   // S130, max time T#10S, warning time T#7S
   END_STEP
   TRANSITION Trans146 FROM "Wait  robot finish task" TO PartStatus   // T146
      := "KukaRobot1_CtrlDB".sROBtoPLC.User.Cycle.DO250_ShaftScanPutFinish;
   END_TRANSITION
   STEP CheckMachineStatus:   // S102, max time T#10S, warning time T#7S
   END_STEP
   TRANSITION Trans266 FROM CheckMachineStatus TO "Normal mode"   // T102
      := TRUE;
   END_TRANSITION
   STEP "Normal mode":   // S103, max time T#10S, warning time T#7S
   END_STEP
   TRANSITION Trans11 FROM "Normal mode" TO "ProcessStart,CTStart"   // T103
      := TRUE;
   END_TRANSITION
   STEP RobotPutPartFinish:   // S115, max time T#10S, warning time T#7S
   END_STEP
   TRANSITION Trans199 FROM RobotPutPartFinish TO CheckPartExist   // T115
      := TRUE;
   END_TRANSITION
   STEP ProcessStart:   // S100, max time T#10S, warning time T#7S
      // 自动等待开始运行
              R    #ioPM_Inface.InitialRun
              R    #ioPM_Inface.ProcessComplete
              R    #ioPM_Inface.ProcessStart
              S    #ioPM_Inface.InitialOK
              S    #ioPM_Inface.WaitRunning
          S1  N    #ioPM_Inface.ProcessResult:=0
              R    "ST10_GeneralData".FlowControl_Handshake[3].Start
              R    "ST10_GeneralData".FlowControl_Handshake[3].Done
              N    "MES_CHeck_DB".Station_1.CheckStep:=0
              N    "MES_CHeck_DB".Station_1.ResultStep:=0
   END_STEP
   TRANSITION Trans200 FROM ProcessStart TO "Determine product status"   // T100
      := NOT #ioPM_Inface.AlarmCycleStop AND #ioPM_Inface.Running AND NOT #iSysInface.Auto.RunningOver AND (NOT #iSysInface.Auto.OneCycleMode OR (#iSysInface.Auto.OneCycleMode AND #ioPM_Inface.TriggerOneCycle));
   END_TRANSITION
   STEP "ProcessStart,CTStart":   // S104, max time T#10S, warning time T#7S
              S    #ioPM_Inface.ProcessStart
              R    #ioPM_Inface.ProcessComplete
   END_STEP
   TRANSITION Trans249 FROM "ProcessStart,CTStart" TO "Request robot put"   // T104
      := #"ProcessStart,CTStart".T > t#100MS;
   END_TRANSITION
   STEP CheckPartExist:   // S237, max time T#10S, warning time T#7S
   END_STEP
   TRANSITION Trans250 FROM CheckPartExist TO "Rotary code reading"   // T249, jump
      := #TON[0].Q;
   END_TRANSITION
   TRANSITION Trans251 FROM CheckPartExist TO PartStatusError   // T250
      := NOT "iA-Rotating product Check" AND (#CheckPartExist.T > t#1500MS);
   END_TRANSITION
   STEP "Request robot put":   // S112, max time T#10S, warning time T#7S
              N    "AutoProcessControl".A_ScanRotary.Robot1PutPrimit
   END_STEP
   TRANSITION Trans283 FROM "Request robot put" TO "Wait  robot finish task"   // T112
      := "KukaRobot1_CtrlDB".sROBtoPLC.User.Cycle.DO249_ShaftScanPutInside AND NOT "KukaRobot1_CtrlDB".sROBtoPLC.User.Cycle.DO250_ShaftScanPutFinish;
   END_TRANSITION
   STEP PartStatusError:   // S127, max time T#10S, warning time T#7S
              S    "ST10_DeviceError".A.A1RotaryScan.PartMissing
   END_STEP
   TRANSITION Trans254 FROM PartStatusError TO CheckPartExist   // T254, jump
      := #iSysInface.Reset;
   END_TRANSITION
   STEP PartStatus:   // S238, max time T#10S, warning time T#7S
              N    "AutoProcessData".A_ScanRotate.PartStatus:=100
   END_STEP
   TRANSITION Trans252 FROM PartStatus TO RobotPutPartFinish   // T251
      := "AutoProcessData".A_ScanRotate.PartStatus = 100;
   END_TRANSITION
   STEP "Determine product status":   // S101, max time T#10S, warning time T#7S
   END_STEP
   TRANSITION Empty FROM "Determine product status" TO NoPart   // T101
      := #TOF[1].Q AND ("AutoProcessData".A_ScanRotate.PartStatus = 0);
   END_TRANSITION
   TRANSITION HavePart FROM "Determine product status" TO PartStatusOK   // T139
      := #TON[0].Q AND ("AutoProcessData".A_ScanRotate.PartStatus <> 0);
   END_TRANSITION
   TRANSITION Alarm FROM "Determine product status" TO StatusAlarm   // T710
      := ((#TON[0].Q AND ("AutoProcessData".A_ScanRotate.PartStatus = 0)) OR (NOT "iA-Rotating product Check" AND ("AutoProcessData".A_ScanRotate.PartStatus <> 0))) AND (#"Determine product status".T > t#1500MS);
   END_TRANSITION
   STEP PartStatusOK:   // S125, max time T#10S, warning time T#7S
   END_STEP
   TRANSITION Trans303 FROM PartStatusOK TO "Rotary code reading"   // T140, jump
      := TRUE;
   END_TRANSITION
   STEP StatusAlarm:   // S126, max time T#10S, warning time T#7S
          S1  S    "ST10_DeviceError".A.A1RotaryScan.ProductAnomaly
   END_STEP
   TRANSITION Trans304 FROM StatusAlarm TO "Determine product status"   // T141, jump
      := #iSysInface.Reset;
   END_TRANSITION
   STEP NoPart:   // S129, max time T#10S, warning time T#7S
   END_STEP
   TRANSITION Trans145 FROM NoPart TO CheckMachineStatus   // T145
      := TRUE;
   END_TRANSITION

   // sequencer 3: S200-S299Rotary code reading
   STEP "Rotary code reading":   // S200, max time T#10S, warning time T#7S
   END_STEP
   TRANSITION Trans147 FROM "Rotary code reading" TO Step208   // T200
      := TRUE;
   END_TRANSITION
   STEP "Start 1st reading":   // S201, max time T#10S, warning time T#7S
          S1  S    "KeyenceSR1000Ctrl_801A1DB".ioAutoTrigger
   END_STEP
   TRANSITION Trans201 FROM "Start 1st reading" TO "Wait reading complete"   // T201
      := NOT "KeyenceSR1000Ctrl_801A1DB".sHMI.Status.Ready;
   END_TRANSITION
   STEP "Check reader Ready":   // S202, max time T#10S, warning time T#7S
   END_STEP
   TRANSITION Trans202 FROM "Check reader Ready" TO "Start 1st reading"   // T202
      := "KeyenceSR1000Ctrl_801A1DB".sHMI.Status.Ready;
   END_TRANSITION
   STEP "Wait reading complete":   // S203, max time T#10S, warning time T#7S
   END_STEP
   TRANSITION ReadNG FROM "Wait reading complete" TO "Servo returns to Scan2 Pos"   // T203
      := "KeyenceSR1000Ctrl_801A1DB".sHMI.Status.Complete AND "KeyenceSR1000Ctrl_801A1DB".sHMI.Status.ReadNok;
   END_TRANSITION
   TRANSITION ReadOK FROM "Wait reading complete" TO "Read OK"   // T204, jump
      := "KeyenceSR1000Ctrl_801A1DB".sHMI.Status.Complete AND "KeyenceSR1000Ctrl_801A1DB".sHMI.Status.ReadOk;
   END_TRANSITION
   STEP "Servo returns to Scan2 Pos":   // S204, max time T#10S, warning time T#7S
      interlock C := "ServoV90_A2".Out.oReady;
      (C)     N    "ServoV90_DeviceCtl".V90Servo[2].Point[2].Start
   END_STEP
   TRANSITION Trans205 FROM "Servo returns to Scan2 Pos" TO "Check reader Ready_1"   // T205
      := "ServoV90_DeviceCtl".V90Servo[2].Point[2].Achieve;
   END_TRANSITION
   STEP "Start 2st reading":   // S205, max time T#10S, warning time T#7S
          S1  S    "KeyenceSR1000Ctrl_801A1DB".ioAutoTrigger
   END_STEP
   TRANSITION Trans203 FROM "Start 2st reading" TO "Wait reading complete_1"   // T206
      := NOT "KeyenceSR1000Ctrl_801A1DB".sHMI.Status.Ready;
   END_TRANSITION
   STEP "Check reader Ready_1":   // S206, max time T#10S, warning time T#7S
   END_STEP
   TRANSITION Trans204 FROM "Check reader Ready_1" TO "Start 2st reading"   // T207
      := "KeyenceSR1000Ctrl_801A1DB".sHMI.Status.Ready;
   END_TRANSITION
   STEP "Wait reading complete_1":   // S207, max time T#10S, warning time T#7S
   END_STEP
   TRANSITION ReadNG_2 FROM "Wait reading complete_1" TO "Servo returns to Scan3 Pos"   // T208
      := "KeyenceSR1000Ctrl_801A1DB".sHMI.Status.Complete AND "KeyenceSR1000Ctrl_801A1DB".sHMI.Status.ReadNok;
   END_TRANSITION
   TRANSITION ReadOK_2 FROM "Wait reading complete_1" TO "Read OK"   // T210, jump
      := "KeyenceSR1000Ctrl_801A1DB".sHMI.Status.Complete AND "KeyenceSR1000Ctrl_801A1DB".sHMI.Status.ReadOk;
   END_TRANSITION
   STEP Step208:   // S208, max time T#10S, warning time T#7S
   END_STEP
   TRANSITION Trans211 FROM Step208 TO "Check reader Ready"   // T211
      := "AutoProcessData".A_ScanRotate.PartStatus <= 100;
   END_TRANSITION
   TRANSITION Trans212 FROM Step208 TO "Read OK"   // T212
      := "AutoProcessData".A_ScanRotate.PartStatus = 180;
   END_TRANSITION
   TRANSITION Trans246 FROM Step208 TO "Read NG"   // T245
      := "AutoProcessData".A_ScanRotate.PartStatus = 150;
   END_TRANSITION
   TRANSITION Trans253 FROM Step208 TO "MES OK"   // T253
      := "AutoProcessData".A_ScanRotate.PartStatus >= 190;
   END_TRANSITION
   TRANSITION Trans307 FROM Step208 TO "MES NG"   // T307
      := ("AutoProcessData".A_ScanRotate.PartStatus = 151) OR ("AutoProcessData".A_ScanRotate.PartStatus = 152);
   END_TRANSITION
   STEP "Read OK":   // S209, max time T#10S, warning time T#7S
   END_STEP
   TRANSITION Trans213 FROM "Read OK" TO OKStatus   // T213
      := TRUE;
   END_TRANSITION
   STEP "Servo returns to Scan3 Pos":   // S210, max time T#10S, warning time T#7S
      interlock C := "ServoV90_A2".Out.oReady;
      (C)     N    "ServoV90_DeviceCtl".V90Servo[2].Point[3].Start
   END_STEP
   TRANSITION Trans206 FROM "Servo returns to Scan3 Pos" TO "Check reader Ready_2"   // T209
      := "ServoV90_DeviceCtl".V90Servo[2].Point[3].Achieve;
   END_TRANSITION
   STEP "Start 3st reading":   // S211, max time T#10S, warning time T#7S
          S1  S    "KeyenceSR1000Ctrl_801A1DB".ioAutoTrigger
   END_STEP
   TRANSITION Trans207 FROM "Start 3st reading" TO "Wait reading complete_3"   // T214
      := NOT "KeyenceSR1000Ctrl_801A1DB".sHMI.Status.Ready;
   END_TRANSITION
   STEP "Check reader Ready_2":   // S212, max time T#10S, warning time T#7S
   END_STEP
   TRANSITION Trans208 FROM "Check reader Ready_2" TO "Start 3st reading"   // T216
      := "KeyenceSR1000Ctrl_801A1DB".sHMI.Status.Ready;
   END_TRANSITION
   STEP "Wait reading complete_3":   // S213, max time T#10S, warning time T#7S
   END_STEP
   TRANSITION ReadNG_3 FROM "Wait reading complete_3" TO "Servo returns to Scan4 Pos"   // T217
      := "KeyenceSR1000Ctrl_801A1DB".sHMI.Status.Complete AND "KeyenceSR1000Ctrl_801A1DB".sHMI.Status.ReadNok;
   END_TRANSITION
   TRANSITION ReadOK_3 FROM "Wait reading complete_3" TO "Read OK"   // T218, jump
      := "KeyenceSR1000Ctrl_801A1DB".sHMI.Status.Complete AND "KeyenceSR1000Ctrl_801A1DB".sHMI.Status.ReadOk;
   END_TRANSITION
   STEP "Servo returns to Scan4 Pos":   // S214, max time T#10S, warning time T#7S
      interlock C := "ServoV90_A2".Out.oReady;
      (C)     N    "ServoV90_DeviceCtl".V90Servo[2].Point[4].Start
   END_STEP
   TRANSITION Trans209 FROM "Servo returns to Scan4 Pos" TO "Check reader Ready_3"   // T219
      := "ServoV90_DeviceCtl".V90Servo[2].Point[4].Achieve;
   END_TRANSITION
   STEP "Start 4st reading_1":   // S215, max time T#10S, warning time T#7S
          S1  S    "KeyenceSR1000Ctrl_801A1DB".ioAutoTrigger
   END_STEP
   TRANSITION Trans210 FROM "Start 4st reading_1" TO "Wait reading complete_4"   // T221
      := NOT "KeyenceSR1000Ctrl_801A1DB".sHMI.Status.Ready;
   END_TRANSITION
   STEP "Check reader Ready_3":   // S216, max time T#10S, warning time T#7S
   END_STEP
   TRANSITION Trans214 FROM "Check reader Ready_3" TO "Start 4st reading_1"   // T222
      := "KeyenceSR1000Ctrl_801A1DB".sHMI.Status.Ready;
   END_TRANSITION
   STEP "Wait reading complete_4":   // S217, max time T#10S, warning time T#7S
   END_STEP
   TRANSITION ReadNG_4 FROM "Wait reading complete_4" TO "Servo returns to Scan5 Pos"   // T223
      := "KeyenceSR1000Ctrl_801A1DB".sHMI.Status.Complete AND "KeyenceSR1000Ctrl_801A1DB".sHMI.Status.ReadNok;
   END_TRANSITION
   TRANSITION ReadOK_4 FROM "Wait reading complete_4" TO "Read OK"   // T224, jump
      := "KeyenceSR1000Ctrl_801A1DB".sHMI.Status.Complete AND "KeyenceSR1000Ctrl_801A1DB".sHMI.Status.ReadOk;
   END_TRANSITION
   STEP "Servo returns to Scan5 Pos":   // S218, max time T#10S, warning time T#7S
      interlock C := "ServoV90_A2".Out.oReady;
      (C)     N    "ServoV90_DeviceCtl".V90Servo[2].Point[5].Start
   END_STEP
   TRANSITION Trans215 FROM "Servo returns to Scan5 Pos" TO "Check reader Ready_4"   // T225
      := "ServoV90_DeviceCtl".V90Servo[2].Point[5].Achieve;
   END_TRANSITION
   STEP "Start 5st reading":   // S219, max time T#10S, warning time T#7S
          S1  S    "KeyenceSR1000Ctrl_801A1DB".ioAutoTrigger
   END_STEP
   TRANSITION Trans216 FROM "Start 5st reading" TO "Wait reading complete_5"   // T226
      := NOT "KeyenceSR1000Ctrl_801A1DB".sHMI.Status.Ready;
   END_TRANSITION
   STEP "Check reader Ready_4":   // S220, max time T#10S, warning time T#7S
   END_STEP
   TRANSITION Trans217 FROM "Check reader Ready_4" TO "Start 5st reading"   // T227
      := "KeyenceSR1000Ctrl_801A1DB".sHMI.Status.Ready;
   END_TRANSITION
   STEP "Wait reading complete_5":   // S221, max time T#10S, warning time T#7S
   END_STEP
   TRANSITION ReadNG_5 FROM "Wait reading complete_5" TO "Servo returns to Scan6Pos"   // T228
      := "KeyenceSR1000Ctrl_801A1DB".sHMI.Status.Complete AND "KeyenceSR1000Ctrl_801A1DB".sHMI.Status.ReadNok;
   END_TRANSITION
   TRANSITION ReadOK_5 FROM "Wait reading complete_5" TO "Read OK"   // T229, jump
      := "KeyenceSR1000Ctrl_801A1DB".sHMI.Status.Complete AND "KeyenceSR1000Ctrl_801A1DB".sHMI.Status.ReadOk;
   END_TRANSITION
   STEP "Servo returns to Scan6Pos":   // S222, max time T#10S, warning time T#7S
      interlock C := "ServoV90_A2".Out.oReady;
      (C)     N    "ServoV90_DeviceCtl".V90Servo[2].Point[6].Start
   END_STEP
   TRANSITION Trans218 FROM "Servo returns to Scan6Pos" TO "Check reader Ready_5"   // T230
      := "ServoV90_DeviceCtl".V90Servo[2].Point[6].Achieve;
   END_TRANSITION
   STEP "Start 6st reading":   // S223, max time T#10S, warning time T#7S
          S1  S    "KeyenceSR1000Ctrl_801A1DB".ioAutoTrigger
   END_STEP
   TRANSITION Trans219 FROM "Start 6st reading" TO "Wait reading complete_6"   // T231
      := NOT "KeyenceSR1000Ctrl_801A1DB".sHMI.Status.Ready;
   END_TRANSITION
   STEP "Check reader Ready_5":   // S224, max time T#10S, warning time T#7S
   END_STEP
   TRANSITION Trans220 FROM "Check reader Ready_5" TO "Start 6st reading"   // T232
      := "KeyenceSR1000Ctrl_801A1DB".sHMI.Status.Ready;
   END_TRANSITION
   STEP "Wait reading complete_6":   // S225, max time T#10S, warning time T#7S
   END_STEP
   TRANSITION ReadNG_6 FROM "Wait reading complete_6" TO "Servo returns to Scan7Pos"   // T233
      := "KeyenceSR1000Ctrl_801A1DB".sHMI.Status.Complete AND "KeyenceSR1000Ctrl_801A1DB".sHMI.Status.ReadNok;
   END_TRANSITION
   TRANSITION ReadOK_6 FROM "Wait reading complete_6" TO "Read OK"   // T234, jump
      := "KeyenceSR1000Ctrl_801A1DB".sHMI.Status.Complete AND "KeyenceSR1000Ctrl_801A1DB".sHMI.Status.ReadOk;
   END_TRANSITION
   STEP "Servo returns to Scan7Pos":   // S226, max time T#10S, warning time T#7S
      interlock C := "ServoV90_A2".Out.oReady;
      (C)     N    "ServoV90_DeviceCtl".V90Servo[2].Point[7].Start
   END_STEP
   TRANSITION Trans221 FROM "Servo returns to Scan7Pos" TO "Check reader Ready_6"   // T235
      := "ServoV90_DeviceCtl".V90Servo[2].Point[7].Achieve;
   END_TRANSITION
   STEP "Start 7st reading":   // S227, max time T#10S, warning time T#7S
          S1  S    "KeyenceSR1000Ctrl_801A1DB".ioAutoTrigger
   END_STEP
   TRANSITION Trans222 FROM "Start 7st reading" TO "Wait reading complete_7"   // T236
      := NOT "KeyenceSR1000Ctrl_801A1DB".sHMI.Status.Ready;
   END_TRANSITION
   STEP "Check reader Ready_6":   // S228, max time T#10S, warning time T#7S
   END_STEP
   TRANSITION Trans223 FROM "Check reader Ready_6" TO "Start 7st reading"   // T237
      := "KeyenceSR1000Ctrl_801A1DB".sHMI.Status.Ready;
   END_TRANSITION
   STEP "Wait reading complete_7":   // S229, max time T#10S, warning time T#7S
   END_STEP
   TRANSITION ReadNG_7 FROM "Wait reading complete_7" TO "Servo returns to Scan8Pos"   // T238
      := "KeyenceSR1000Ctrl_801A1DB".sHMI.Status.Complete AND "KeyenceSR1000Ctrl_801A1DB".sHMI.Status.ReadNok;
   END_TRANSITION
   TRANSITION ReadOK_7 FROM "Wait reading complete_7" TO "Read OK"   // T239, jump
      := "KeyenceSR1000Ctrl_801A1DB".sHMI.Status.Complete AND "KeyenceSR1000Ctrl_801A1DB".sHMI.Status.ReadOk;
   END_TRANSITION
   STEP "Servo returns to Scan8Pos":   // S230, max time T#10S, warning time T#7S
      interlock C := "ServoV90_A2".Out.oReady;
      (C)     N    "ServoV90_DeviceCtl".V90Servo[2].Point[8].Start
   END_STEP
   TRANSITION Trans225 FROM "Servo returns to Scan8Pos" TO "Check reader Ready_7"   // T240
      := "ServoV90_DeviceCtl".V90Servo[2].Point[8].Achieve;
   END_TRANSITION
   STEP "Start 8st reading":   // S231, max time T#10S, warning time T#7S
          S1  S    "KeyenceSR1000Ctrl_801A1DB".ioAutoTrigger
   END_STEP
   TRANSITION Trans226 FROM "Start 8st reading" TO "Wait reading complete_8"   // T241
      := NOT "KeyenceSR1000Ctrl_801A1DB".sHMI.Status.Ready;
   END_TRANSITION
   STEP "Check reader Ready_7":   // S232, max time T#10S, warning time T#7S
   END_STEP
   TRANSITION Trans227 FROM "Check reader Ready_7" TO "Start 8st reading"   // T242
      := "KeyenceSR1000Ctrl_801A1DB".sHMI.Status.Ready;
   END_TRANSITION
   STEP "Wait reading complete_8":   // S233, max time T#10S, warning time T#7S
   END_STEP
   TRANSITION ReadNG_8 FROM "Wait reading complete_8" TO "Read NG"   // T243, jump
      := "KeyenceSR1000Ctrl_801A1DB".sHMI.Status.Complete AND "KeyenceSR1000Ctrl_801A1DB".sHMI.Status.ReadNok;
   END_TRANSITION
   TRANSITION ReadOK_8 FROM "Wait reading complete_8" TO "Read OK"   // T244, jump
      := "KeyenceSR1000Ctrl_801A1DB".sHMI.Status.Complete AND "KeyenceSR1000Ctrl_801A1DB".sHMI.Status.ReadOk;
   END_TRANSITION
   STEP "Read NG":   // S234, max time T#10S, warning time T#7S
   END_STEP
   TRANSITION Trans230 FROM "Read NG" TO NG_Status   // T246
      := TRUE;
   END_TRANSITION
   STEP NG_Status:   // S235, max time T#10S, warning time T#7S
              N    "AutoProcessData".A_ScanRotate.PartStatus:=150
              N    "AutoProcessData".A_ScanRotate.ShaftCode:=''
   END_STEP
   TRANSITION Trans247 FROM NG_Status TO MES   // T247, jump
      := "AutoProcessData".A_ScanRotate.PartStatus = 150;
   END_TRANSITION
   STEP OKStatus:   // S236, max time T#10S, warning time T#7S
              N    "AutoProcessData".A_ScanRotate.PartStatus:=180
              N    "AutoProcessData".A_ScanRotate.ShaftCode:="KeyenceSR1000Ctrl_801A1DB".sHMI.Status.CurrentCode
   END_STEP
   TRANSITION Trans248 FROM OKStatus TO MES   // T248, jump
      := "AutoProcessData".A_ScanRotate.PartStatus = 180;
   END_TRANSITION
   STEP "MES NG":   // S307, max time T#10S, warning time T#7S
   END_STEP
   TRANSITION Trans308 FROM "MES NG" TO RobotPick   // T308, jump
      := TRUE;
   END_TRANSITION
   STEP "MES OK":   // S12, max time T#10S, warning time T#7S
   END_STEP
   TRANSITION Trans12 FROM "MES OK" TO RobotPick   // T12, jump
      := TRUE;
   END_TRANSITION

   // sequencer 4: S200-S299MES查询获取打标数据 / S300-S399 MES
   STEP "Prepare MES CheckData":   // S303, max time T#10S, warning time T#7S
   END_STEP
   TRANSITION Trans14 FROM "Prepare MES CheckData" TO MESCheckRequest   // T303
      := #"Prepare MES CheckData".T > t#300MS;
   END_TRANSITION
   STEP MESCheckRequest:   // S305, max time T#10S, warning time T#7S
              N    "PLCtoMES"."PLC.Load_Station1ChickInReq"
   END_STEP
   TRANSITION Trans264 FROM MESCheckRequest TO "Check OK"   // T305
      := "MEStoPLC"."MES.Load_Station1PartOK" AND NOT "MEStoPLC"."MES.Load_Station1PartNG" AND "MEStoPLC"."MES.Load_Station1ReqMesDone";
   END_TRANSITION
   TRANSITION Trans610 FROM MESCheckRequest TO "Check NG"   // T314
      := NOT "MEStoPLC"."MES.Load_Station1PartOK" AND "MEStoPLC"."MES.Load_Station1PartNG" AND "MEStoPLC"."MES.Load_Station1ReqMesDone";
   END_TRANSITION
   TRANSITION Trans313 FROM MESCheckRequest TO MESOverTime_1   // T313
      := #MESCheckRequest.T > t#10S;
   END_TRANSITION
   STEP MES:   // S300, max time T#10S, warning time T#7S
   END_STEP
   TRANSITION Trans312 FROM MES TO Bypass   // T312
      := TRUE;
   END_TRANSITION
   STEP ResetMesCheckRequest:   // S301, max time T#10S, warning time T#7S
              R    "PLCtoMES"."PLC.Load_Station1ChickInReq"
              R    "MEStoPLC"."MES.Load_Station1PartOK"
              R    "MEStoPLC"."MES.Load_Station1PartNG"
              R    "MEStoPLC"."MES.Load_Station1ReqMesDone"
   END_STEP
   TRANSITION Trans259 FROM ResetMesCheckRequest TO "Prepare MES CheckData"   // T301
      := NOT "PLCtoMES"."PLC.Load_Station1ChickInReq" AND NOT "MEStoPLC"."MES.Load_Station1PartOK" AND NOT "MEStoPLC"."MES.Load_Station1PartNG" AND NOT "MEStoPLC"."MES.Load_Station1ReqMesDone";
   END_TRANSITION
   STEP ok:   // S309, max time T#10S, warning time T#7S
              N    "AutoProcessData".A_ScanRotate.PartStatus:=199
   END_STEP
   TRANSITION Trans315 FROM ok TO MESResultFinish   // T309
      := "AutoProcessData".A_ScanRotate.PartStatus = 199;
   END_TRANSITION
   STEP "Check OK":   // S316, max time T#10S, warning time T#7S
   END_STEP
   TRANSITION Trans322 FROM "Check OK" TO ResetMesUnloadRequest_1   // T322
      := TRUE;
   END_TRANSITION
   STEP "Check NG":   // S317, max time T#10S, warning time T#7S
              N    "AutoProcessData".A_ScanRotate.PartStatus:=151
   END_STEP
   TRANSITION Trans16 FROM "Check NG" TO RobotPick   // T316, jump
      := "AutoProcessData".A_ScanRotate.PartStatus = 151;
   END_TRANSITION
   STEP "Prepare MES CheckData_1":   // S304, max time T#10S, warning time T#7S
   END_STEP
   TRANSITION Trans15 FROM "Prepare MES CheckData_1" TO MESSaveRequest_1   // T304
      := #"Prepare MES CheckData_1".T > t#300MS;
   END_TRANSITION
   STEP MESSaveRequest_1:   // S306, max time T#10S, warning time T#7S
              N    "PLCtoMES"."PLC.Unload_Station1DataSaveReq"
   END_STEP
   TRANSITION Trans265 FROM MESSaveRequest_1 TO ok   // T306
      := "MEStoPLC"."MES.Unload_ResultsStored1OK" AND NOT "MEStoPLC"."MES.Unload_ResultsStored1NG" AND "MEStoPLC"."MES.Unload_ResultsStored1ReqMesDone";
   END_TRANSITION
   TRANSITION Trans310 FROM MESSaveRequest_1 TO MESOverTime   // T310
      := NOT "MEStoPLC"."MES.Unload_ResultsStored1ReqMesDone" AND (#MESSaveRequest_1.T > t#10S);
   END_TRANSITION
   TRANSITION Trans317 FROM MESSaveRequest_1 TO ResultNG   // T317
      := NOT "MEStoPLC"."MES.Unload_ResultsStored1OK" AND "MEStoPLC"."MES.Unload_ResultsStored1NG" AND "MEStoPLC"."MES.Unload_ResultsStored1ReqMesDone";
   END_TRANSITION
   STEP ResetMesUnloadRequest_1:   // S302, max time T#10S, warning time T#7S
              R    "PLCtoMES"."PLC.Unload_Station1DataSaveReq"
              R    "MEStoPLC"."MES.Unload_ResultsStored1OK"
              R    "MEStoPLC"."MES.Unload_ResultsStored1NG"
              R    "MEStoPLC"."MES.Unload_ResultsStored1ReqMesDone"
   END_STEP
   TRANSITION Trans260 FROM ResetMesUnloadRequest_1 TO "Prepare MES CheckData_1"   // T302
      := NOT "PLCtoMES"."PLC.Unload_Station1DataSaveReq" AND NOT "MEStoPLC"."MES.Unload_ResultsStored1OK" AND NOT "MEStoPLC"."MES.Unload_ResultsStored1NG" AND NOT "MEStoPLC"."MES.Unload_ResultsStored1ReqMesDone";
   END_TRANSITION
   STEP MESOverTime:   // S308, max time T#10S, warning time T#7S
              S    "ST10_DeviceError".MES_Error.CheckInResultOverTime_1
   END_STEP
   TRANSITION Trans311 FROM MESOverTime TO Bypass   // T311, jump
      := #iSysInface.Reset;
   END_TRANSITION
   STEP Bypass:   // S310, max time T#10S, warning time T#7S
   END_STEP
   TRANSITION Online FROM Bypass TO ResetMesCheckRequest   // T300
      := NOT "Station_Sys".Cmd.OnOffLine;
   END_TRANSITION
   TRANSITION Offline FROM Bypass TO ok_1   // T13
      := "Station_Sys".Cmd.OnOffLine;
   END_TRANSITION
   STEP MESOverTime_1:   // S311, max time T#10S, warning time T#7S
              S    "ST10_DeviceError".MES_Error.CheckInCompOverTime_1
   END_STEP
   TRANSITION Trans314 FROM MESOverTime_1 TO Bypass   // T315, jump
      := #iSysInface.Reset;
   END_TRANSITION
   STEP ResultNG:   // S312, max time T#10S, warning time T#7S
              N    "AutoProcessData".A_ScanRotate.PartStatus:=152
   END_STEP
   TRANSITION Trans318 FROM ResultNG TO MESResultFinish   // T318
      := "AutoProcessData".A_ScanRotate.PartStatus = 152;
   END_TRANSITION
   STEP MESResultFinish:   // S313, max time T#10S, warning time T#7S
   END_STEP
   TRANSITION Trans319 FROM MESResultFinish TO RobotPick   // T319, jump
      := TRUE;
   END_TRANSITION
   STEP Step314:   // S314, max time T#10S, warning time T#7S
   END_STEP
   TRANSITION Trans320 FROM Step314 TO MESResultFinish   // T320
      := TRUE;
   END_TRANSITION
   STEP ok_1:   // S315, max time T#10S, warning time T#7S
      interlock C := "AutoProcessData".A_ScanRotate.PartStatus = 180;
      (C)     N    "AutoProcessData".A_ScanRotate.PartStatus:=199
   END_STEP
   TRANSITION Trans316 FROM ok_1 TO Step314   // T321
      := ("AutoProcessData".A_ScanRotate.PartStatus = 199) OR ("Station_Sys".Cmd.OnOffLine AND ("AutoProcessData".A_ScanRotate.PartStatus = 150));
   END_TRANSITION

   // sequencer 5: S600-S699工件放行 / S600-S699 RobotPick
   STEP RobotPick:   // S600, max time T#10S, warning time T#7S
              S    #ioPM_Inface.ProcessComplete
              R    #ioPM_Inface.ProcessStart
   END_STEP
   TRANSITION Trans600 FROM RobotPick TO "Request robot pick"   // T600
      := TRUE;
   END_TRANSITION
   STEP ProcessFinsh:   // S605, max time T#10S, warning time T#7S: 正式使用时，需要激活复位空循环
   END_STEP
   TRANSITION Trans699 FROM ProcessFinsh TO ProcessStart   // T605, jump
      := TRUE;
   END_TRANSITION
   STEP "Request robot pick":   // S408, max time T#10S, warning time T#7S
              N    "AutoProcessControl".A_ScanRotary.Robot1PickPrimit
   END_STEP
   TRANSITION Trans412 FROM "Request robot pick" TO "Wait robot finish task"   // T410
      := "KukaRobot1_CtrlDB".sROBtoPLC.User.Cycle.DO253_SScanPickInside AND NOT "KukaRobot1_CtrlDB".sROBtoPLC.User.Cycle.DO254_SScanPickFinish;
   END_TRANSITION
   STEP "Wait robot finish task":   // S131, max time T#10S, warning time T#7S
   END_STEP
   TRANSITION Trans257 FROM "Wait robot finish task" TO "Wait robot in safety area"   // T256
      := "KukaRobot1_CtrlDB".sROBtoPLC.User.Cycle.DO254_SScanPickFinish;
   END_TRANSITION
   STEP "Wait robot in safety area":   // S133, max time T#10S, warning time T#7S
   END_STEP
   TRANSITION Trans261 FROM "Wait robot in safety area" TO "Servo returns to initial Pos_1"   // T258
      := "KukaRobot1_CtrlDB".sROBtoPLC.User.Home.DO180_Robot2Area;
   END_TRANSITION
   STEP "Servo returns to initial Pos_1":   // S11, max time T#10S, warning time T#7S
              N    "ServoV90_DeviceCtl".V90Servo[2].Point[1].Start
   END_STEP
   TRANSITION Trans8 FROM "Servo returns to initial Pos_1" TO ProcessFinsh   // T11
      := "ServoV90_DeviceCtl".V90Servo[2].Point[1].Achieve;
   END_TRANSITION

   // permanent post-instructions
   NETWORK 1
      #ioPM_Inface.StepNum := #RT_DATA.S_DISPLAY;
   NETWORK 2
      IF #iSysInface.Reset THEN #AlarmID := 0; END_IF;
   NETWORK 3
      #TON[10].TON(IN := #工件放行中, PT := T#0.5S);
      IF #TON[10].Q THEN #工件放行中 := FALSE; END_IF;
END_FUNCTION_BLOCK

FUNCTION_BLOCK "ST10_Flow4_B1Press"   // FB1074, GRAPH
// stored: AcknowledgeErrorsRequired false, AutoNumber false, GraphVersion 6.0, InitialValuesAcquisition false, SetENOAutomatically false
   // inherited from GRAPH_BASE
   VAR_INPUT
      iSysInface : "RCS_SysComInterface_V1";
   END_VAR
   VAR_IN_OUT
      ioPM_Inface : "RCS_PMInterface_V1";
      ioStatus : Int;
   END_VAR
   VAR
      sCtrlMode { S7_SetPoint := 'True'} : "SysFlowCtrlGraph";
      sUpdMES_Data : Bool;   // 更新MES数据
      工件放行中 : Bool;
      前站站号 { ExternalAccessible := 'False'; ExternalVisible := 'False'; ExternalWritable := 'False'} : UInt;
      本站站号 { ExternalAccessible := 'False'; ExternalVisible := 'False'; ExternalWritable := 'False'} : UInt;
      弹窗Temp : Array[1..10] of Int;
      AlarmID : Int;
      TON { S7_SetPoint := 'True'} : Array[0..10] of TON_TIME;
      TOF { S7_SetPoint := 'True'} : Array[0..10] of TOF_TIME;
      sUP { S7_SetPoint := 'True'} : Array[0..10] of Bool;
      更新RFID完成 : Bool;
   END_VAR
   VAR_TEMP
      Tempresult : USInt;
      本站站号乘10 : UInt;
   END_VAR
   // // TON[0] : 托盘流入1托盘到位传感器 / iA-Rotating product Check
   // // TON[1] : 托盘流入1托盘到位传感器
   // // TON[2] : 托盘流入1产品有无传感器
   // // TON[3] : 托盘流入1产品有无传感器
   // // TON[4] : 托盘流入1姿态检测光电2
   // // TON[5] : 托盘流入1姿态检测光电3
   // // TON[0].Q : 托盘流入1托盘到位 / iA-Rotating product Check
   // // TON[1].Q : 托盘流入1托盘无
   // // TON[2].Q : 托盘流入1有产品
   // // TON[3].Q : 托盘流入1无产品
   // // TON[4].Q : 托盘流入1姿态检测光电2
   // // TON[5].Q : 托盘流入1姿态检测光电3
   // // TOF[1] : iA-Rotating product Check
BEGIN
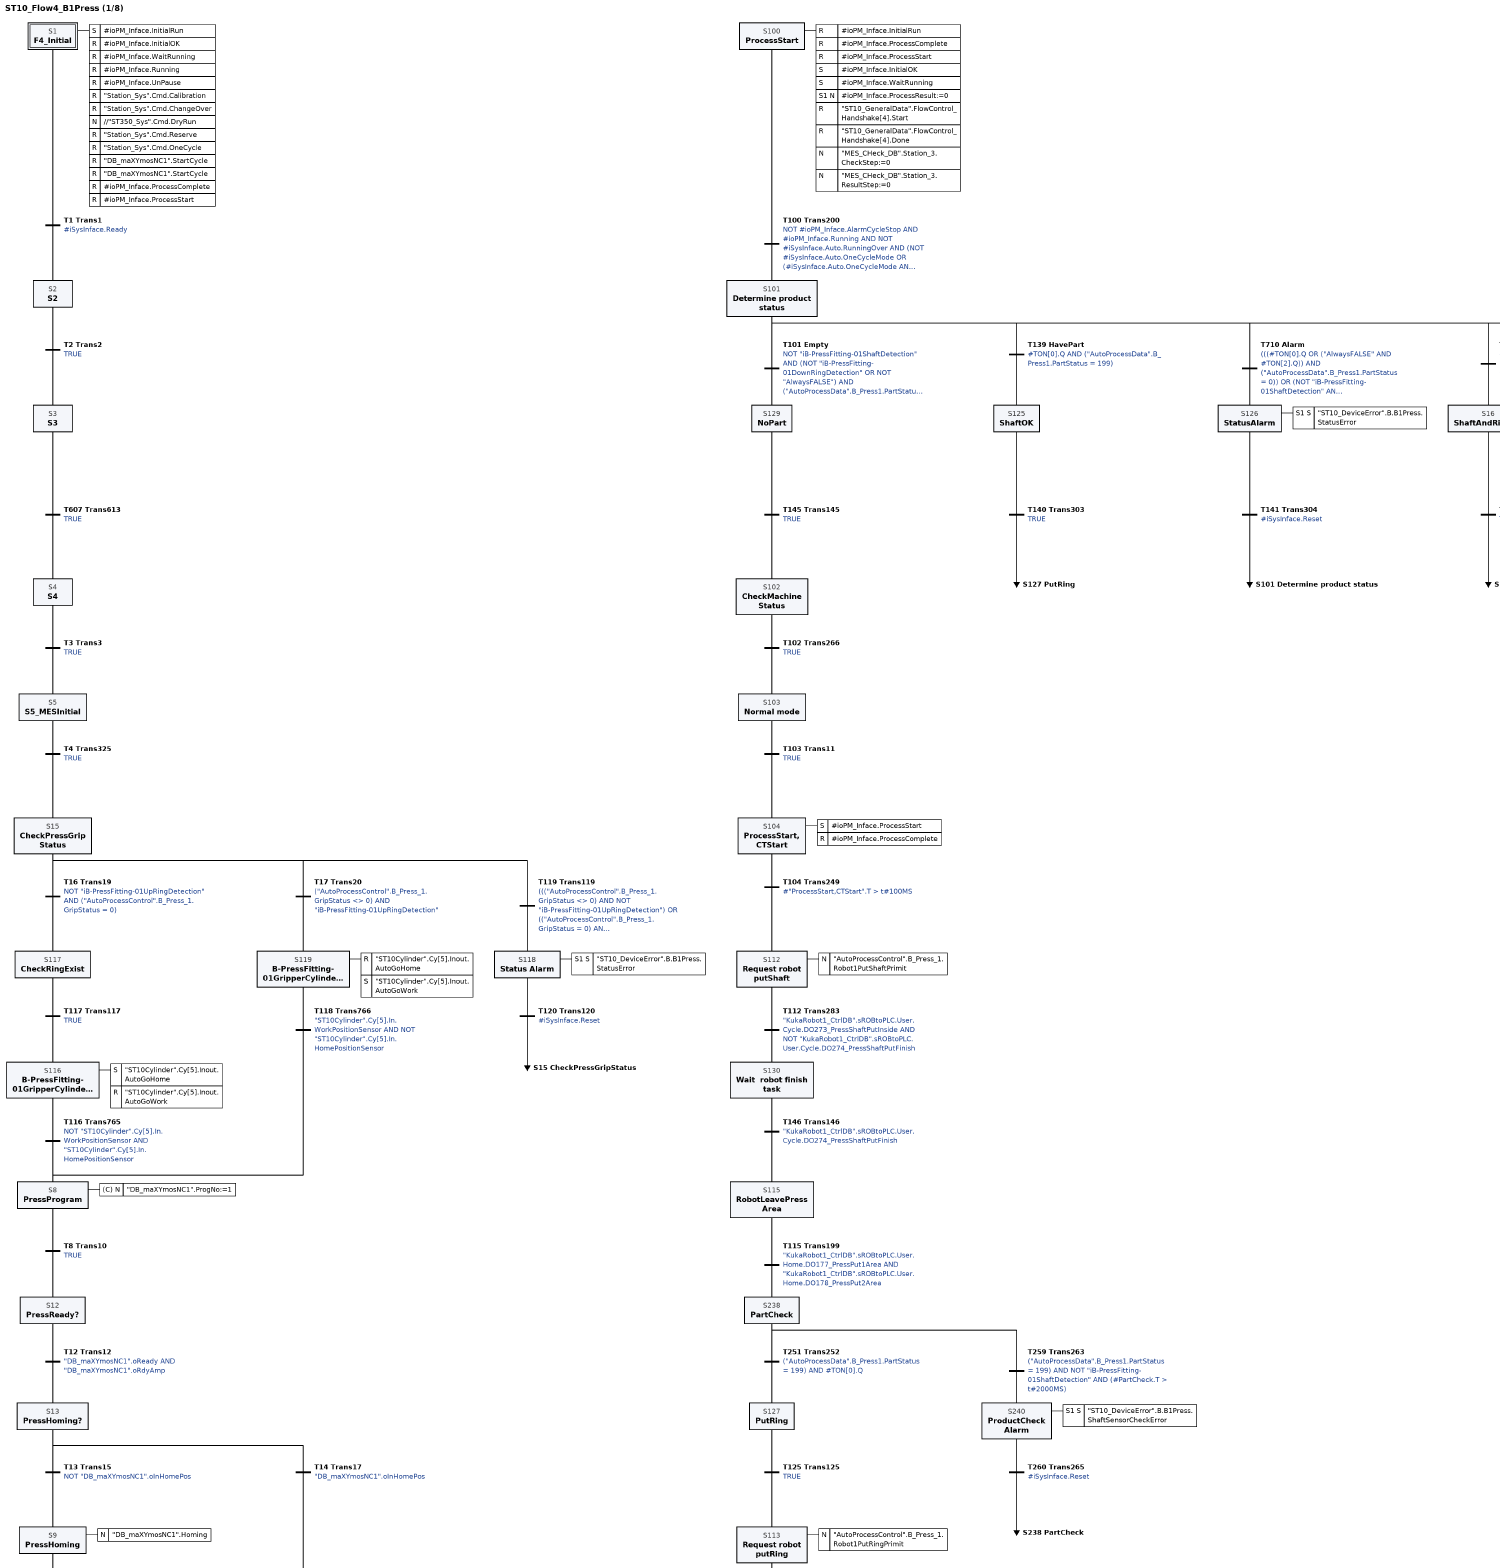
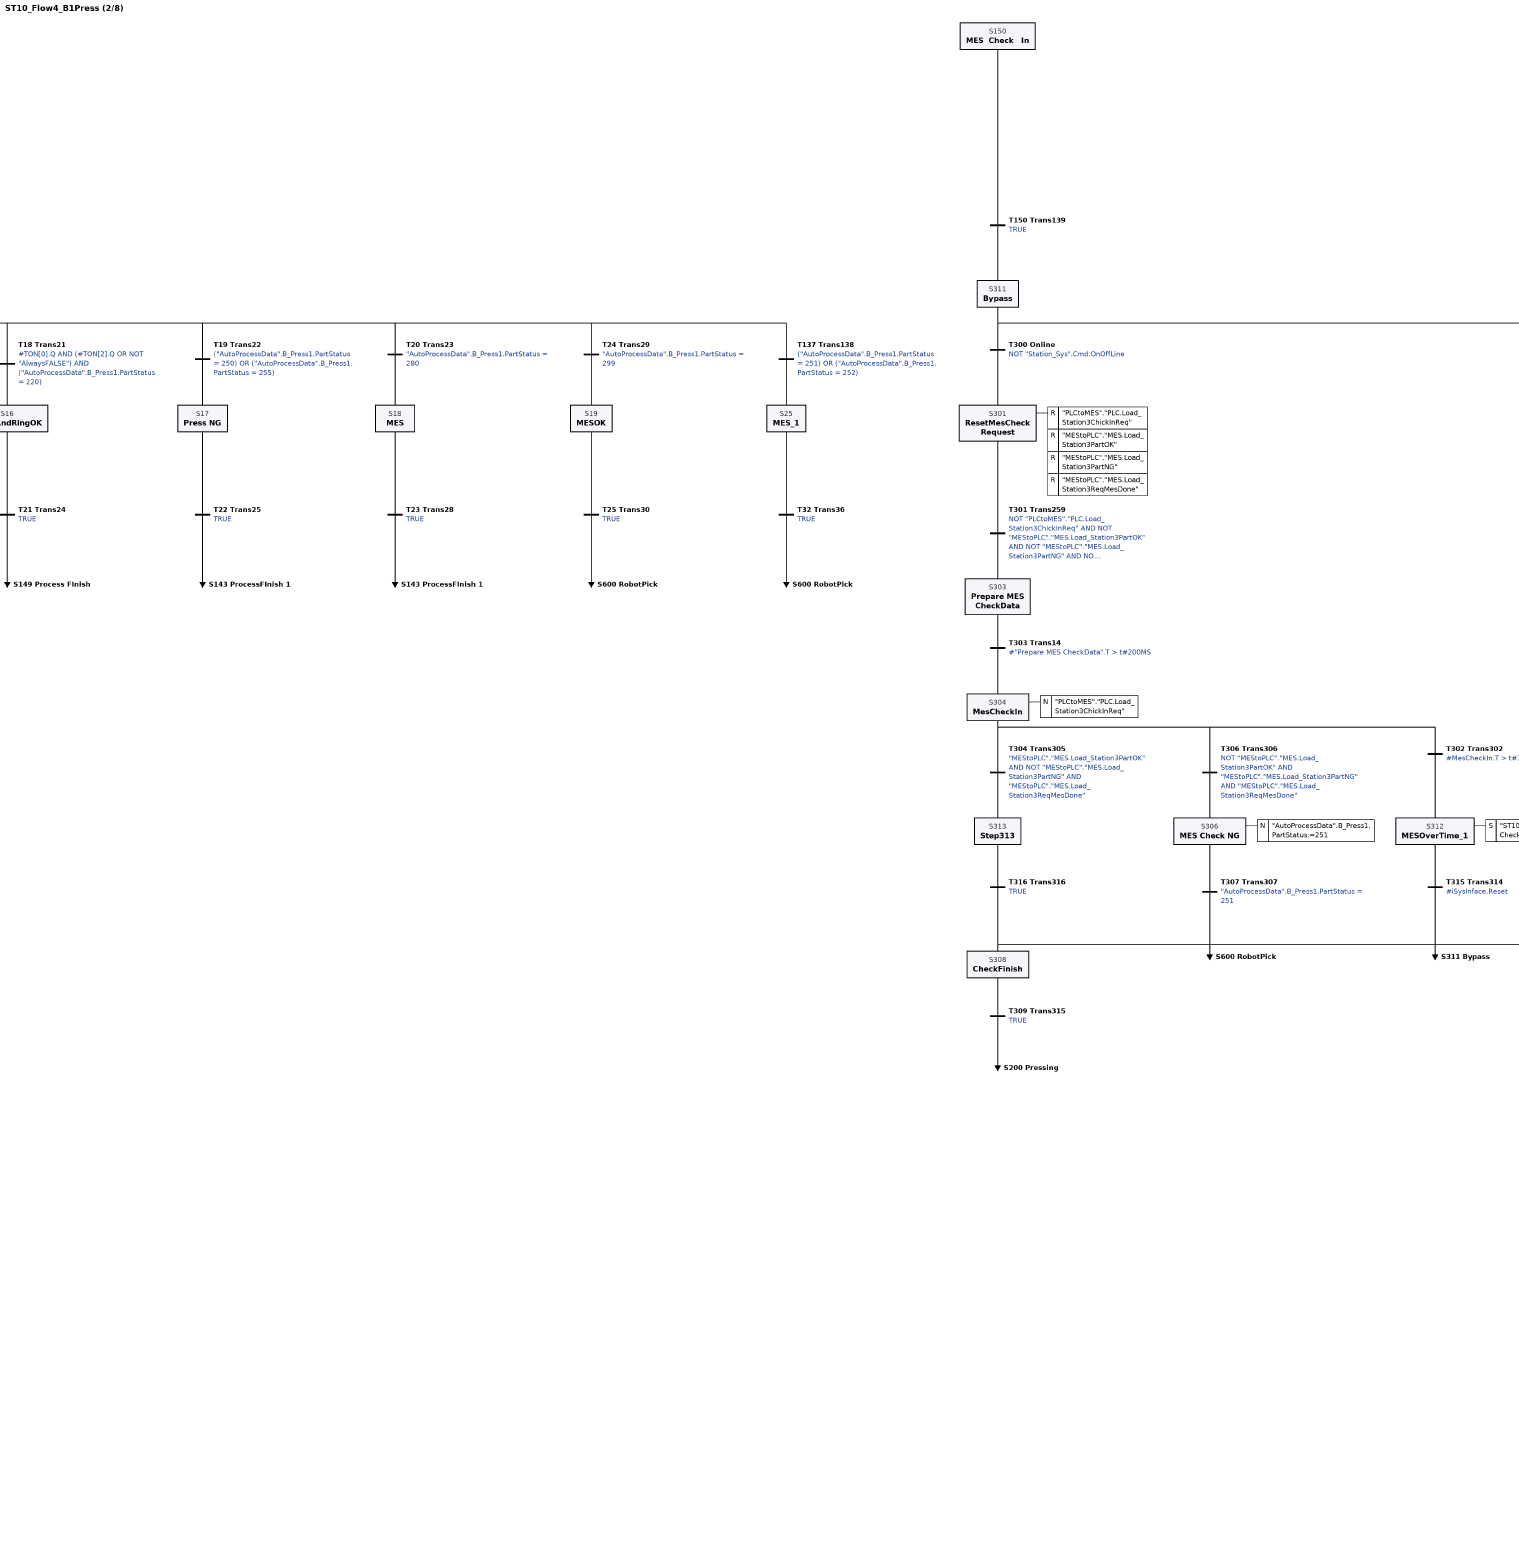
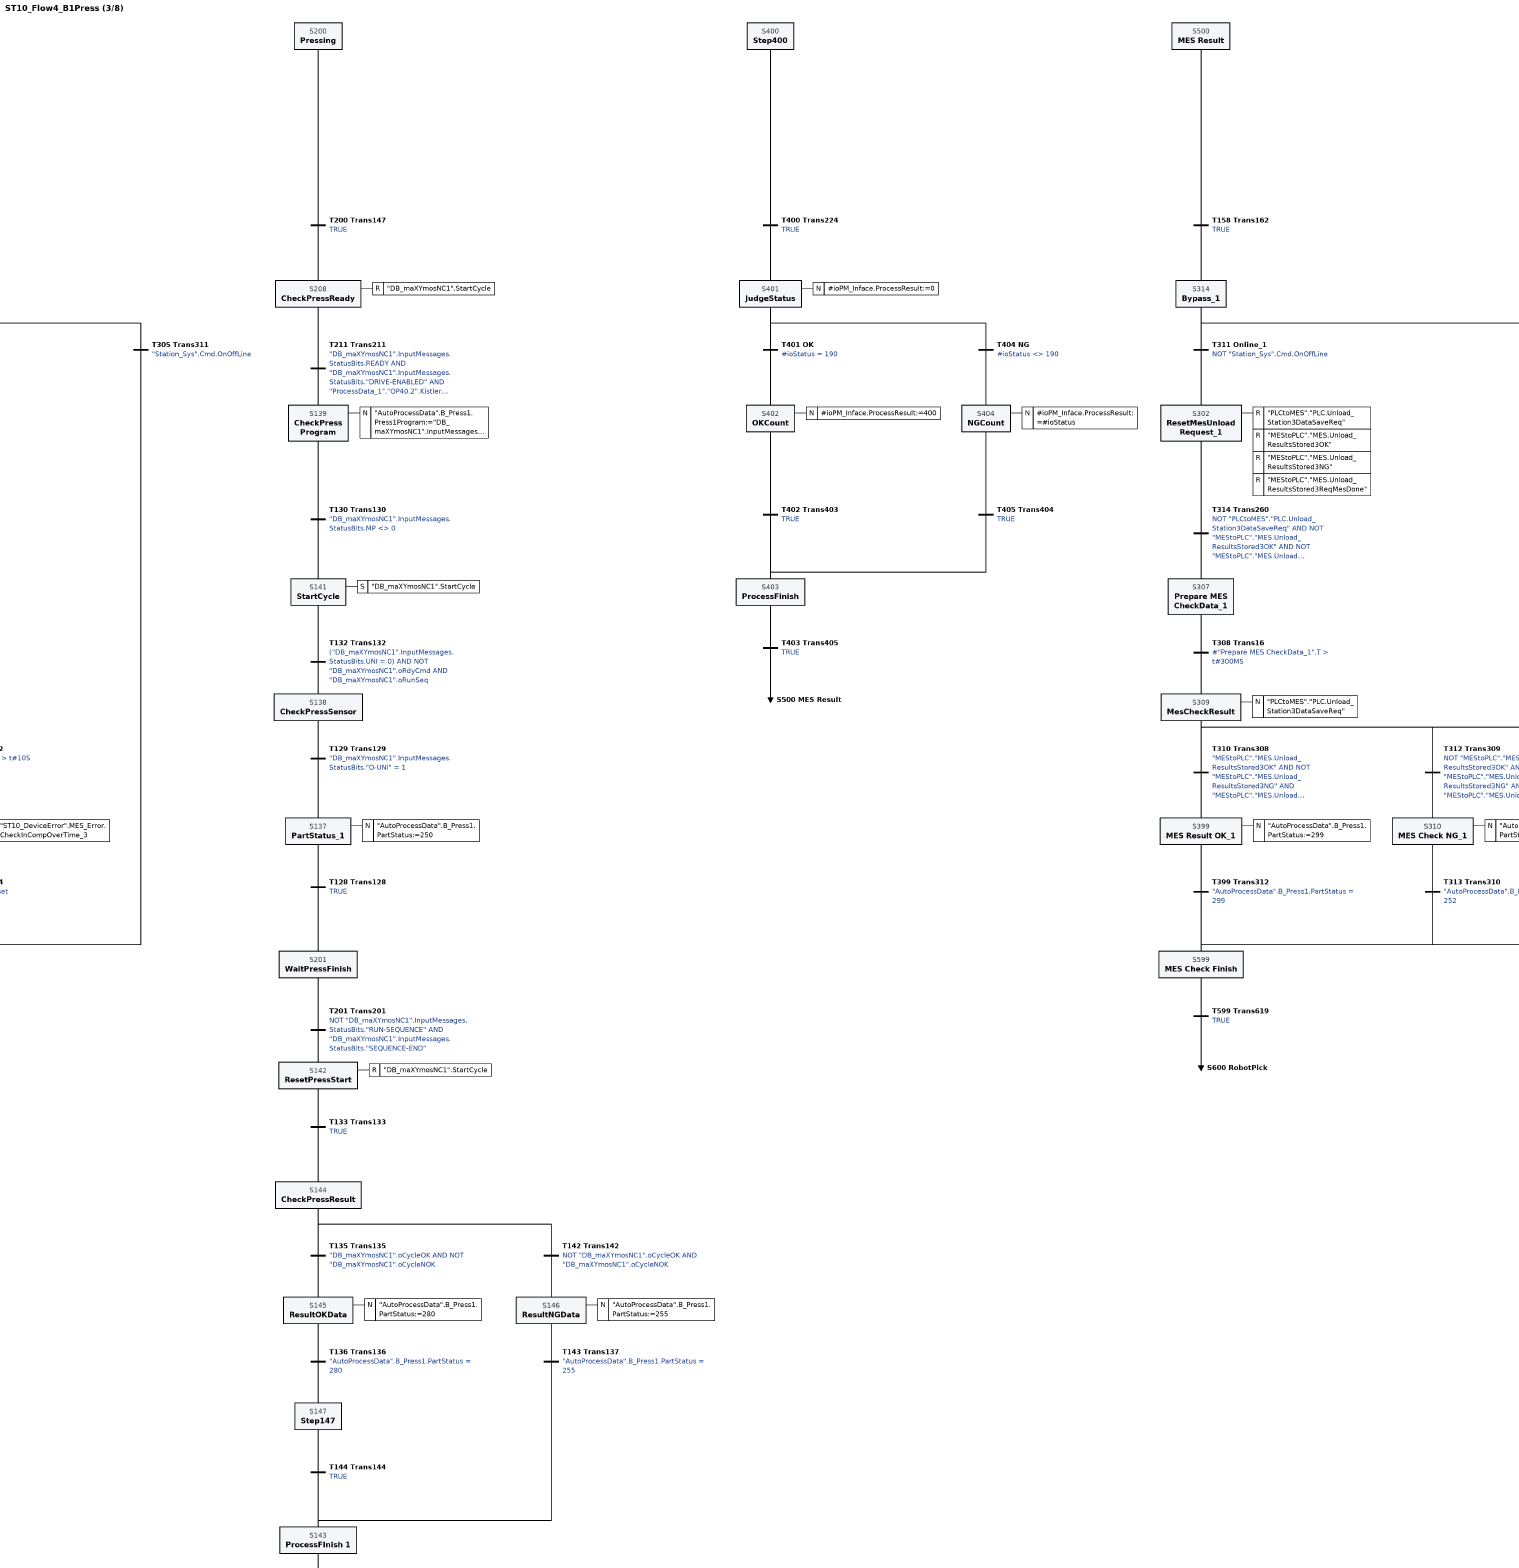
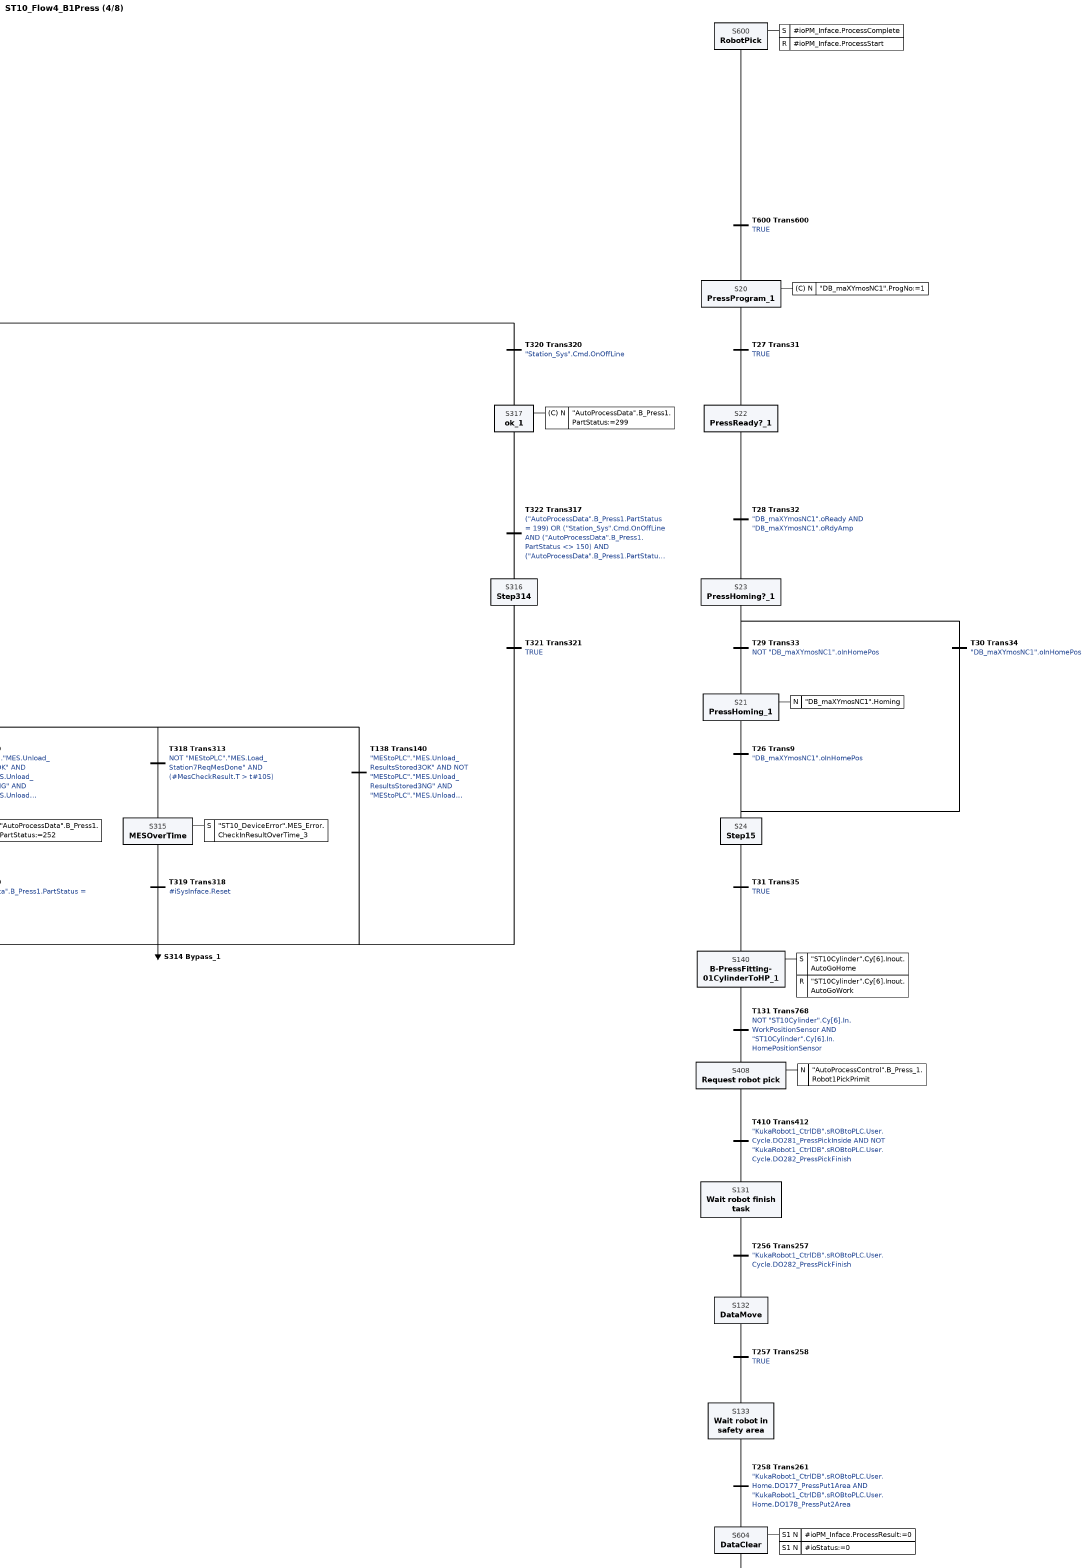
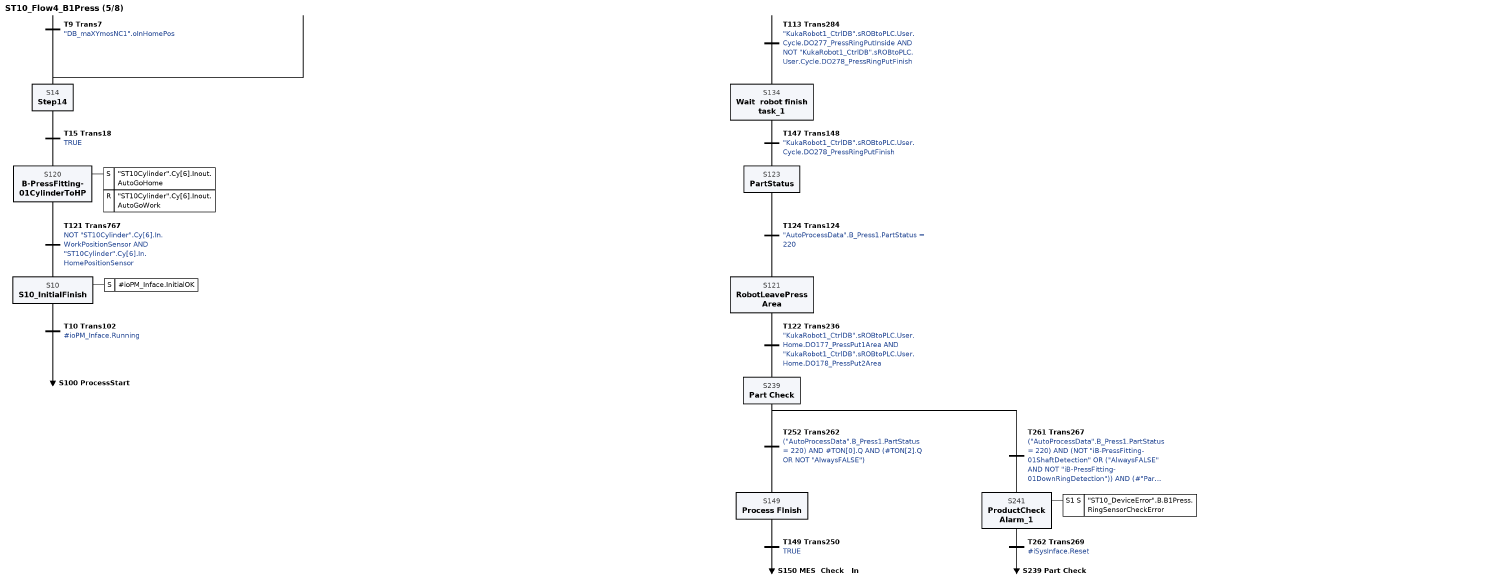
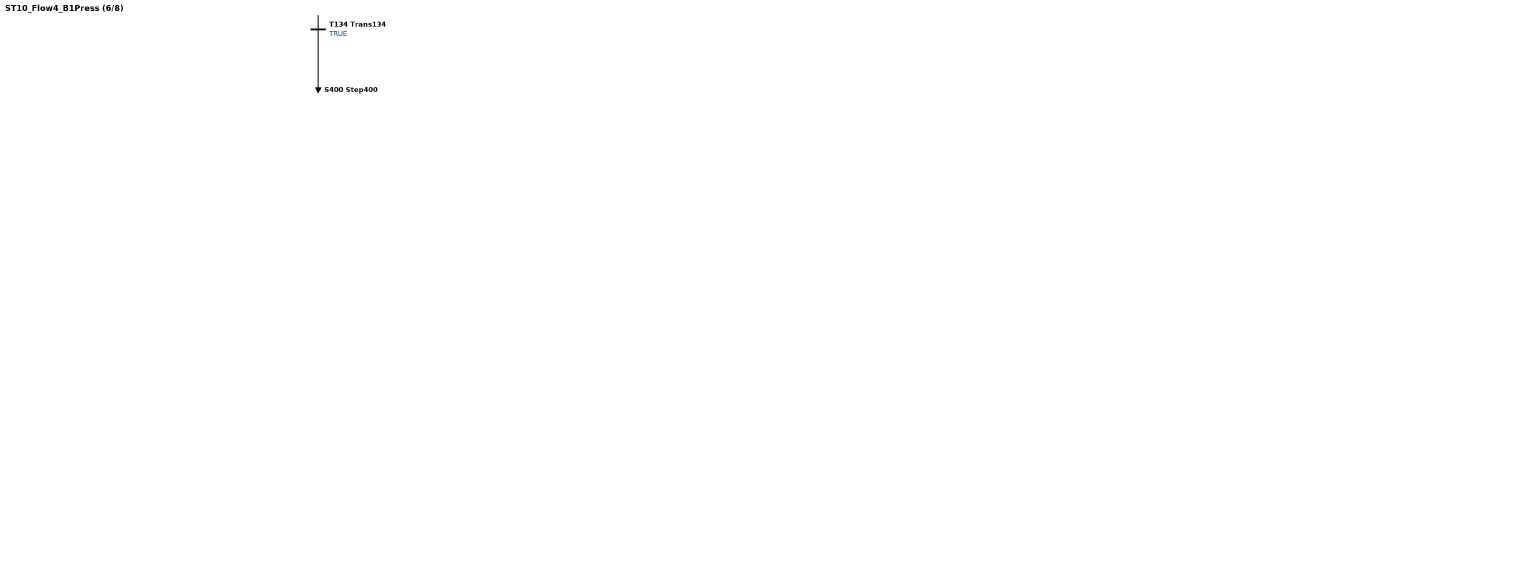
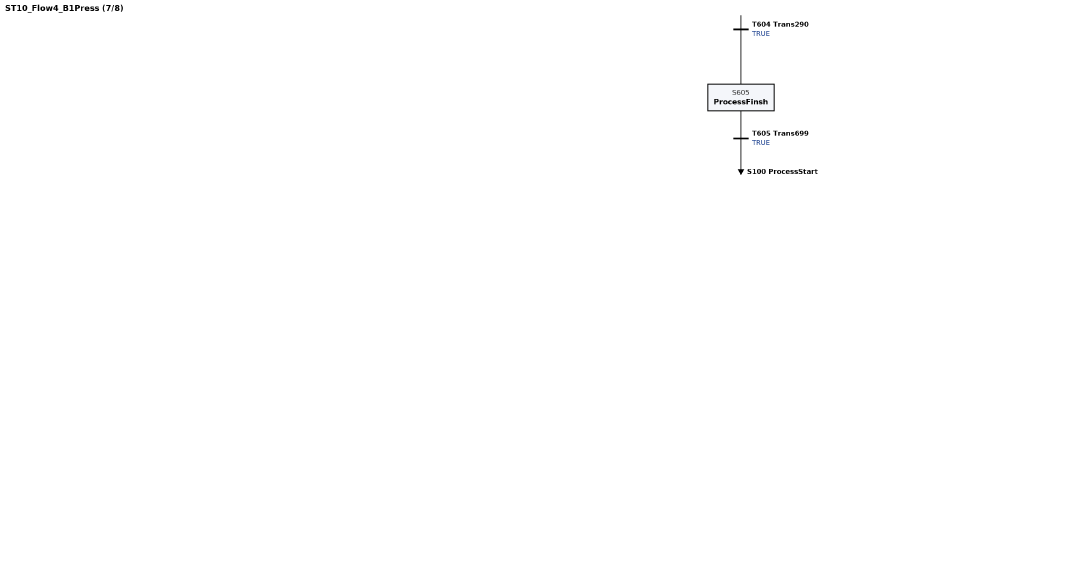
   // permanent pre-instructions
   NETWORK 1
      #TON[10].TON(IN := "AlwaysTRUE" AND "Station_Sys".Alarm.ImmediatelyStop, PT := T#300ms);
      #ioPM_Inface.AlarmImdilyStop := #TON[10].Q;
      #ioPM_Inface.AlarmCycleStop := "AlwaysTRUE" AND "Station_Sys".Alarm.CycleStop;
   NETWORK 2
      IF NOT False THEN
          #sCtrlMode(iSysInface := #iSysInface, ioPM_Inface := #ioPM_Inface, ioGraphCtrl := #RT_DATA.MOP);   // "SysFlowCtrlGraph"
      END_IF;
   NETWORK 3
      #TON[0].TON(IN := "AlwaysTRUE" AND "iB-PressFitting-01ShaftDetection", PT := t#500ms);   // 工位11有托盘
      #TOF[1].TOF(IN := "AlwaysTRUE" AND NOT "iB-PressFitting-01ShaftDetection", PT := T#300ms);   // 工位无托盘
      #TON[2].TON(IN := "AlwaysTRUE" AND "iB-PressFitting-01DownRingDetection", PT := T#300ms);
      #TOF[3].TOF(IN := "AlwaysTRUE" AND NOT "iB-PressFitting-01DownRingDetection", PT := T#300ms);
      #TON[4].TON(IN := "AlwaysTRUE" AND "iB-PressFitting-01UpRingDetection", PT := T#300ms);
      #TON[5].TON(IN := "AlwaysTRUE" AND NOT "iB-PressFitting-01UpRingDetection", PT := T#300ms);
   NETWORK 4
      #前站站号 := 345;
      #本站站号 := 350;

   // sequencer 1: S01-S99 初始化 / S01-S99 Initial
   INITIAL_STEP F4_Initial:   // S1, max time T#10S, warning time T#7S
              S    #ioPM_Inface.InitialRun
              R    #ioPM_Inface.InitialOK
              R    #ioPM_Inface.WaitRunning
              R    #ioPM_Inface.Running
              R    #ioPM_Inface.UnPause
              R    "Station_Sys".Cmd.Calibration
              R    "Station_Sys".Cmd.ChangeOver
                   //"ST350_Sys".Cmd.DryRun
              R    "Station_Sys".Cmd.Reserve
              R    "Station_Sys".Cmd.OneCycle
              R    "DB_maXYmosNC1".StartCycle
              R    "DB_maXYmosNC1".StartCycle
              R    #ioPM_Inface.ProcessComplete
              R    #ioPM_Inface.ProcessStart
              R    "AutoProcessControl".B_Press_1.Robot1PickPrimit
              R    "AutoProcessControl".B_Press_1.Robot1PutShaftPrimit
              R    "AutoProcessControl".B_Press_1.Robot1PutRingPrimit
   END_STEP
   TRANSITION Trans1 FROM F4_Initial TO S2   // T1
      := #iSysInface.Ready;
   END_TRANSITION
   STEP S2:   // S2, max time T#10S, warning time T#7S
   END_STEP
   TRANSITION Trans2 FROM S2 TO S3   // T2
      := TRUE;
   END_TRANSITION
   STEP S4:   // S4, max time T#10S, warning time T#7S
   END_STEP
   TRANSITION Trans3 FROM S4 TO S5_MESInitial   // T3
      := TRUE;
   END_TRANSITION
   STEP S5_MESInitial:   // S5, max time T#10S, warning time T#7S
   END_STEP
   TRANSITION Trans325 FROM S5_MESInitial TO CheckPressGripStatus   // T4
      := TRUE;
   END_TRANSITION
   STEP S10_InitialFinish:   // S10, max time T#10S, warning time T#7S
              S    #ioPM_Inface.InitialOK
   END_STEP
   TRANSITION Trans102 FROM S10_InitialFinish TO ProcessStart   // T10, jump
      := #ioPM_Inface.Running;
   END_TRANSITION
   STEP S3:   // S3, max time T#10S, warning time T#7S
   END_STEP
   TRANSITION Trans613 FROM S3 TO S4   // T607
      := TRUE;
   END_TRANSITION
   STEP PressProgram:   // S8, max time T#10S, warning time T#7S
      interlock C := NOT "ST10_GeneralData".FunctionDeSelect."B".FunctionDeSelected_TestPress372A1;
      (C)     N    "DB_maXYmosNC1".ProgNo:=1
   END_STEP
   TRANSITION Trans10 FROM PressProgram TO "PressReady?"   // T8
      := TRUE;
   END_TRANSITION
   STEP PressHoming:   // S9, max time T#10S, warning time T#7S
              N    "DB_maXYmosNC1".Homing
   END_STEP
   TRANSITION Trans7 FROM PressHoming TO Step14   // T9
      := "DB_maXYmosNC1".oInHomePos;
   END_TRANSITION
   STEP "PressReady?":   // S12, max time T#10S, warning time T#7S
   END_STEP
   TRANSITION Trans12 FROM "PressReady?" TO "PressHoming?"   // T12
      := "DB_maXYmosNC1".oReady AND "DB_maXYmosNC1".oRdyAmp;
   END_TRANSITION
   STEP "PressHoming?":   // S13, max time T#10S, warning time T#7S
   END_STEP
   TRANSITION Trans15 FROM "PressHoming?" TO PressHoming   // T13
      := NOT "DB_maXYmosNC1".oInHomePos;
   END_TRANSITION
   TRANSITION Trans17 FROM "PressHoming?" TO Step14   // T14
      := "DB_maXYmosNC1".oInHomePos;
   END_TRANSITION
   STEP Step14:   // S14, max time T#10S, warning time T#7S
   END_STEP
   TRANSITION Trans18 FROM Step14 TO "B-PressFitting-01CylinderToHP"   // T15
      := TRUE;
   END_TRANSITION
   STEP CheckPressGripStatus:   // S15, max time T#10S, warning time T#7S
   END_STEP
   TRANSITION Trans19 FROM CheckPressGripStatus TO CheckRingExist   // T16
      := NOT "iB-PressFitting-01UpRingDetection" AND ("AutoProcessControl".B_Press_1.GripStatus = 0);
   END_TRANSITION
   TRANSITION Trans20 FROM CheckPressGripStatus TO "B-PressFitting-01GripperCylinderToWP"   // T17
      := ("AutoProcessControl".B_Press_1.GripStatus <> 0) AND "iB-PressFitting-01UpRingDetection";
   END_TRANSITION
   TRANSITION Trans119 FROM CheckPressGripStatus TO "Status Alarm"   // T119
      := ((("AutoProcessControl".B_Press_1.GripStatus <> 0) AND NOT "iB-PressFitting-01UpRingDetection") OR (("AutoProcessControl".B_Press_1.GripStatus = 0) AND "iB-PressFitting-01UpRingDetection")) AND (#CheckPressGripStatus.T > t#1500MS);
   END_TRANSITION
   STEP "B-PressFitting-01GripperCylinderToHP":   // S116, max time T#10S, warning time T#7S
              S    "ST10Cylinder".Cy[5].Inout.AutoGoHome
              R    "ST10Cylinder".Cy[5].Inout.AutoGoWork
   END_STEP
   TRANSITION Trans765 FROM "B-PressFitting-01GripperCylinderToHP" TO PressProgram   // T116
      := NOT "ST10Cylinder".Cy[5].In.WorkPositionSensor AND "ST10Cylinder".Cy[5].In.HomePositionSensor;
   END_TRANSITION
   STEP CheckRingExist:   // S117, max time T#10S, warning time T#7S
   END_STEP
   TRANSITION Trans117 FROM CheckRingExist TO "B-PressFitting-01GripperCylinderToHP"   // T117
      := TRUE;
   END_TRANSITION
   STEP "Status Alarm":   // S118, max time T#10S, warning time T#7S
          S1  S    "ST10_DeviceError".B.B1Press.StatusError
   END_STEP
   TRANSITION Trans120 FROM "Status Alarm" TO CheckPressGripStatus   // T120, jump
      := #iSysInface.Reset;
   END_TRANSITION
   STEP "B-PressFitting-01GripperCylinderToWP":   // S119, max time T#10S, warning time T#7S
              R    "ST10Cylinder".Cy[5].Inout.AutoGoHome
              S    "ST10Cylinder".Cy[5].Inout.AutoGoWork
   END_STEP
   TRANSITION Trans766 FROM "B-PressFitting-01GripperCylinderToWP" TO PressProgram   // T118
      := "ST10Cylinder".Cy[5].In.WorkPositionSensor AND NOT "ST10Cylinder".Cy[5].In.HomePositionSensor;
   END_TRANSITION
   STEP "B-PressFitting-01CylinderToHP":   // S120, max time T#10S, warning time T#7S
              S    "ST10Cylinder".Cy[6].Inout.AutoGoHome
              R    "ST10Cylinder".Cy[6].Inout.AutoGoWork
   END_STEP
   TRANSITION Trans767 FROM "B-PressFitting-01CylinderToHP" TO S10_InitialFinish   // T121
      := NOT "ST10Cylinder".Cy[6].In.WorkPositionSensor AND "ST10Cylinder".Cy[6].In.HomePositionSensor;
   END_TRANSITION

   // sequencer 2: S100-S199 等待到位 / S100-S149 CheckPartStatus
   STEP "Wait  robot finish task":   // S130, max time T#10S, warning time T#7S
   END_STEP
   TRANSITION Trans146 FROM "Wait  robot finish task" TO "RobotLeavePress Area"   // T146
      := "KukaRobot1_CtrlDB".sROBtoPLC.User.Cycle.DO274_PressShaftPutFinish;
   END_TRANSITION
   STEP CheckMachineStatus:   // S102, max time T#10S, warning time T#7S
   END_STEP
   TRANSITION Trans266 FROM CheckMachineStatus TO "Normal mode"   // T102
      := TRUE;
   END_TRANSITION
   STEP "Normal mode":   // S103, max time T#10S, warning time T#7S
   END_STEP
   TRANSITION Trans11 FROM "Normal mode" TO "ProcessStart,CTStart"   // T103
      := TRUE;
   END_TRANSITION
   STEP ProcessStart:   // S100, max time T#10S, warning time T#7S
      // 自动等待开始运行
              R    #ioPM_Inface.InitialRun
              R    #ioPM_Inface.ProcessComplete
              R    #ioPM_Inface.ProcessStart
              S    #ioPM_Inface.InitialOK
              S    #ioPM_Inface.WaitRunning
          S1  N    #ioPM_Inface.ProcessResult:=0
              R    "ST10_GeneralData".FlowControl_Handshake[4].Start
              R    "ST10_GeneralData".FlowControl_Handshake[4].Done
              N    "MES_CHeck_DB".Station_3.CheckStep:=0
              N    "MES_CHeck_DB".Station_3.ResultStep:=0
   END_STEP
   TRANSITION Trans200 FROM ProcessStart TO "Determine product status"   // T100
      := NOT #ioPM_Inface.AlarmCycleStop AND #ioPM_Inface.Running AND NOT #iSysInface.Auto.RunningOver AND (NOT #iSysInface.Auto.OneCycleMode OR (#iSysInface.Auto.OneCycleMode AND #ioPM_Inface.TriggerOneCycle));
   END_TRANSITION
   STEP "ProcessStart,CTStart":   // S104, max time T#10S, warning time T#7S
              S    #ioPM_Inface.ProcessStart
              R    #ioPM_Inface.ProcessComplete
   END_STEP
   TRANSITION Trans249 FROM "ProcessStart,CTStart" TO "Request robot putShaft"   // T104
      := #"ProcessStart,CTStart".T > t#100MS;
   END_TRANSITION
   STEP "Process FInish":   // S149, max time T#10S, warning time T#7S
   END_STEP
   TRANSITION Trans250 FROM "Process FInish" TO "MES  Check   In"   // T149, jump
      := TRUE;
   END_TRANSITION
   STEP "Request robot putShaft":   // S112, max time T#10S, warning time T#7S
              N    "AutoProcessControl".B_Press_1.Robot1PutShaftPrimit
   END_STEP
   TRANSITION Trans283 FROM "Request robot putShaft" TO "Wait  robot finish task"   // T112
      := "KukaRobot1_CtrlDB".sROBtoPLC.User.Cycle.DO273_PressShaftPutInside AND NOT "KukaRobot1_CtrlDB".sROBtoPLC.User.Cycle.DO274_PressShaftPutFinish;
   END_TRANSITION
   STEP PutRing:   // S127, max time T#10S, warning time T#7S
   END_STEP
   TRANSITION Trans125 FROM PutRing TO "Request robot putRing"   // T125
      := TRUE;
   END_TRANSITION
   STEP PartCheck:   // S238, max time T#10S, warning time T#7S
   END_STEP
   TRANSITION Trans252 FROM PartCheck TO PutRing   // T251
      := ("AutoProcessData".B_Press1.PartStatus = 199) AND #TON[0].Q;
   END_TRANSITION
   TRANSITION Trans263 FROM PartCheck TO ProductCheckAlarm   // T259
      := ("AutoProcessData".B_Press1.PartStatus = 199) AND NOT "iB-PressFitting-01ShaftDetection" AND (#PartCheck.T > t#2000MS);
   END_TRANSITION
   STEP "Determine product status":   // S101, max time T#10S, warning time T#7S
   END_STEP
   TRANSITION Empty FROM "Determine product status" TO NoPart   // T101
      := NOT "iB-PressFitting-01ShaftDetection" AND (NOT "iB-PressFitting-01DownRingDetection" OR NOT "AlwaysFALSE") AND ("AutoProcessData".B_Press1.PartStatus = 0) AND (#"Determine product status".T > t#100MS);
   END_TRANSITION
   TRANSITION HavePart FROM "Determine product status" TO ShaftOK   // T139
      := #TON[0].Q AND ("AutoProcessData".B_Press1.PartStatus = 199);
   END_TRANSITION
   TRANSITION Alarm FROM "Determine product status" TO StatusAlarm   // T710
      := (((#TON[0].Q OR ("AlwaysFALSE" AND #TON[2].Q)) AND ("AutoProcessData".B_Press1.PartStatus = 0)) OR (NOT "iB-PressFitting-01ShaftDetection" AND ("AutoProcessData".B_Press1.PartStatus = 199)) OR ("AlwaysFALSE" AND NOT "iB-PressFitting-01DownRingDetection" AND ("AutoProcessData".B_Press1.PartStatus = 220)) OR (NOT "iB-PressFitting-01ShaftDetection" AND (NOT "iB-PressFitting-01DownRingDetection" OR NOT "AlwaysFALSE") AND ("AutoProcessData".B_Press1.PartStatus <> 199) AND ("AutoProcessData".B_Press1.PartStatus <> 220) AND ("AutoProcessData".B_Press1.PartStatus <> 0))) AND (#"Determine product status".T > t#3000MS);
   END_TRANSITION
   TRANSITION Trans21 FROM "Determine product status" TO ShaftAndRingOK   // T18
      := #TON[0].Q AND (#TON[2].Q OR NOT "AlwaysFALSE") AND ("AutoProcessData".B_Press1.PartStatus = 220);
   END_TRANSITION
   TRANSITION Trans22 FROM "Determine product status" TO "Press NG"   // T19
      := ("AutoProcessData".B_Press1.PartStatus = 250) OR ("AutoProcessData".B_Press1.PartStatus = 255);
   END_TRANSITION
   TRANSITION Trans23 FROM "Determine product status" TO MES   // T20
      := "AutoProcessData".B_Press1.PartStatus = 280;
   END_TRANSITION
   TRANSITION Trans29 FROM "Determine product status" TO MESOK   // T24
      := "AutoProcessData".B_Press1.PartStatus = 299;
   END_TRANSITION
   TRANSITION Trans138 FROM "Determine product status" TO MES_1   // T137
      := ("AutoProcessData".B_Press1.PartStatus = 251) OR ("AutoProcessData".B_Press1.PartStatus = 252);
   END_TRANSITION
   STEP ShaftOK:   // S125, max time T#10S, warning time T#7S
   END_STEP
   TRANSITION Trans303 FROM ShaftOK TO PutRing   // T140, jump
      := TRUE;
   END_TRANSITION
   STEP StatusAlarm:   // S126, max time T#10S, warning time T#7S
          S1  S    "ST10_DeviceError".B.B1Press.StatusError
   END_STEP
   TRANSITION Trans304 FROM StatusAlarm TO "Determine product status"   // T141, jump
      := #iSysInface.Reset;
   END_TRANSITION
   STEP NoPart:   // S129, max time T#10S, warning time T#7S
   END_STEP
   TRANSITION Trans145 FROM NoPart TO CheckMachineStatus   // T145
      := TRUE;
   END_TRANSITION
   STEP ShaftAndRingOK:   // S16, max time T#10S, warning time T#7S
   END_STEP
   TRANSITION Trans24 FROM ShaftAndRingOK TO "Process FInish"   // T21, jump
      := TRUE;
   END_TRANSITION
   STEP "Press NG":   // S17, max time T#10S, warning time T#7S
   END_STEP
   TRANSITION Trans25 FROM "Press NG" TO "ProcessFInish 1"   // T22, jump
      := TRUE;
   END_TRANSITION
   STEP MES:   // S18, max time T#10S, warning time T#7S
   END_STEP
   TRANSITION Trans28 FROM MES TO "ProcessFInish 1"   // T23, jump
      := TRUE;
   END_TRANSITION
   STEP MESOK:   // S19, max time T#10S, warning time T#7S
   END_STEP
   TRANSITION Trans30 FROM MESOK TO RobotPick   // T25, jump
      := TRUE;
   END_TRANSITION
   STEP "Wait  robot finish task_1":   // S134, max time T#10S, warning time T#7S
   END_STEP
   TRANSITION Trans148 FROM "Wait  robot finish task_1" TO PartStatus   // T147
      := "KukaRobot1_CtrlDB".sROBtoPLC.User.Cycle.DO278_PressRingPutFinish;
   END_TRANSITION
   STEP "Request robot putRing":   // S113, max time T#10S, warning time T#7S
              N    "AutoProcessControl".B_Press_1.Robot1PutRingPrimit
   END_STEP
   TRANSITION Trans284 FROM "Request robot putRing" TO "Wait  robot finish task_1"   // T113
      := "KukaRobot1_CtrlDB".sROBtoPLC.User.Cycle.DO277_PressRingPutInside AND NOT "KukaRobot1_CtrlDB".sROBtoPLC.User.Cycle.DO278_PressRingPutFinish;
   END_TRANSITION
   STEP "Part Check":   // S239, max time T#10S, warning time T#7S
   END_STEP
   TRANSITION Trans262 FROM "Part Check" TO "Process FInish"   // T252
      := ("AutoProcessData".B_Press1.PartStatus = 220) AND #TON[0].Q AND (#TON[2].Q OR NOT "AlwaysFALSE");
   END_TRANSITION
   TRANSITION Trans267 FROM "Part Check" TO ProductCheckAlarm_1   // T261
      := ("AutoProcessData".B_Press1.PartStatus = 220) AND (NOT "iB-PressFitting-01ShaftDetection" OR ("AlwaysFALSE" AND NOT "iB-PressFitting-01DownRingDetection")) AND (#"Part Check".T > t#2000MS);
   END_TRANSITION
   STEP ProductCheckAlarm:   // S240, max time T#10S, warning time T#7S
          S1  S    "ST10_DeviceError".B.B1Press.ShaftSensorCheckError
   END_STEP
   TRANSITION Trans265 FROM ProductCheckAlarm TO PartCheck   // T260, jump
      := #iSysInface.Reset;
   END_TRANSITION
   STEP ProductCheckAlarm_1:   // S241, max time T#10S, warning time T#7S
          S1  S    "ST10_DeviceError".B.B1Press.RingSensorCheckError
   END_STEP
   TRANSITION Trans269 FROM ProductCheckAlarm_1 TO "Part Check"   // T262, jump
      := #iSysInface.Reset;
   END_TRANSITION
   STEP RobotLeavePressArea:   // S121, max time T#10S, warning time T#7S
   END_STEP
   TRANSITION Trans236 FROM RobotLeavePressArea TO "Part Check"   // T122
      := "KukaRobot1_CtrlDB".sROBtoPLC.User.Home.DO177_PressPut1Area AND "KukaRobot1_CtrlDB".sROBtoPLC.User.Home.DO178_PressPut2Area;
   END_TRANSITION
   STEP "RobotLeavePress Area":   // S115, max time T#10S, warning time T#7S
   END_STEP
   TRANSITION Trans199 FROM "RobotLeavePress Area" TO PartCheck   // T115
      := "KukaRobot1_CtrlDB".sROBtoPLC.User.Home.DO177_PressPut1Area AND "KukaRobot1_CtrlDB".sROBtoPLC.User.Home.DO178_PressPut2Area;
   END_TRANSITION
   STEP PartStatus:   // S123, max time T#10S, warning time T#7S
   END_STEP
   TRANSITION Trans124 FROM PartStatus TO RobotLeavePressArea   // T124
      := "AutoProcessData".B_Press1.PartStatus = 220;
   END_TRANSITION
   STEP MES_1:   // S25, max time T#10S, warning time T#7S
   END_STEP
   TRANSITION Trans36 FROM MES_1 TO RobotPick   // T32, jump
      := TRUE;
   END_TRANSITION

   // sequencer 3: S150-S199 MES Check In
   STEP "MES  Check   In":   // S150, max time T#10S, warning time T#7S
   END_STEP
   TRANSITION Trans139 FROM "MES  Check   In" TO Bypass   // T150
      := TRUE;
   END_TRANSITION
   STEP MESOverTime_1:   // S312, max time T#10S, warning time T#7S
              S    "ST10_DeviceError".MES_Error.CheckInCompOverTime_3
   END_STEP
   TRANSITION Trans314 FROM MESOverTime_1 TO Bypass   // T315, jump
      := #iSysInface.Reset;
   END_TRANSITION
   STEP "MES Check NG":   // S306, max time T#10S, warning time T#7S
              N    "AutoProcessData".B_Press1.PartStatus:=251
   END_STEP
   TRANSITION Trans307 FROM "MES Check NG" TO RobotPick   // T307, jump
      := "AutoProcessData".B_Press1.PartStatus = 251;
   END_TRANSITION
   STEP ResetMesCheckRequest:   // S301, max time T#10S, warning time T#7S
              R    "PLCtoMES"."PLC.Load_Station3ChickInReq"
              R    "MEStoPLC"."MES.Load_Station3PartOK"
              R    "MEStoPLC"."MES.Load_Station3PartNG"
              R    "MEStoPLC"."MES.Load_Station3ReqMesDone"
   END_STEP
   TRANSITION Trans259 FROM ResetMesCheckRequest TO "Prepare MES CheckData"   // T301
      := NOT "PLCtoMES"."PLC.Load_Station3ChickInReq" AND NOT "MEStoPLC"."MES.Load_Station3PartOK" AND NOT "MEStoPLC"."MES.Load_Station3PartNG" AND NOT "MEStoPLC"."MES.Load_Station3ReqMesDone";
   END_TRANSITION
   STEP "Prepare MES CheckData":   // S303, max time T#10S, warning time T#7S
   END_STEP
   TRANSITION Trans14 FROM "Prepare MES CheckData" TO MesCheckIn   // T303
      := #"Prepare MES CheckData".T > t#200MS;
   END_TRANSITION
   STEP MesCheckIn:   // S304, max time T#10S, warning time T#7S
              N    "PLCtoMES"."PLC.Load_Station3ChickInReq"
   END_STEP
   TRANSITION Trans305 FROM MesCheckIn TO Step313   // T304
      := "MEStoPLC"."MES.Load_Station3PartOK" AND NOT "MEStoPLC"."MES.Load_Station3PartNG" AND "MEStoPLC"."MES.Load_Station3ReqMesDone";
   END_TRANSITION
   TRANSITION Trans306 FROM MesCheckIn TO "MES Check NG"   // T306
      := NOT "MEStoPLC"."MES.Load_Station3PartOK" AND "MEStoPLC"."MES.Load_Station3PartNG" AND "MEStoPLC"."MES.Load_Station3ReqMesDone";
   END_TRANSITION
   TRANSITION Trans302 FROM MesCheckIn TO MESOverTime_1   // T302
      := #MesCheckIn.T > t#10S;
   END_TRANSITION
   STEP CheckFinish:   // S308, max time T#10S, warning time T#7S
   END_STEP
   TRANSITION Trans315 FROM CheckFinish TO Pressing   // T309, jump
      := TRUE;
   END_TRANSITION
   STEP Bypass:   // S311, max time T#10S, warning time T#7S
   END_STEP
   TRANSITION Online FROM Bypass TO ResetMesCheckRequest   // T300
      := NOT "Station_Sys".Cmd.OnOffLine;
   END_TRANSITION
   TRANSITION Trans311 FROM Bypass TO CheckFinish   // T305
      := "Station_Sys".Cmd.OnOffLine;
   END_TRANSITION
   STEP Step313:   // S313, max time T#10S, warning time T#7S
   END_STEP
   TRANSITION Trans316 FROM Step313 TO CheckFinish   // T316
      := TRUE;
   END_TRANSITION

   // sequencer 4: S200-S299Pressing
   STEP Pressing:   // S200, max time T#10S, warning time T#7S
   END_STEP
   TRANSITION Trans147 FROM Pressing TO CheckPressReady   // T200
      := TRUE;
   END_TRANSITION
   STEP WaitPressFinish:   // S201, max time T#10S, warning time T#7S
   END_STEP
   TRANSITION Trans201 FROM WaitPressFinish TO ResetPressStart   // T201
      := NOT "DB_maXYmosNC1".InputMessages.StatusBits."RUN-SEQUENCE" AND "DB_maXYmosNC1".InputMessages.StatusBits."SEQUENCE-END";
   END_TRANSITION
   STEP ResultNGData:   // S146, max time T#10S, warning time T#7S
              N    "AutoProcessData".B_Press1.PartStatus:=255
   END_STEP
   TRANSITION Trans137 FROM ResultNGData TO "ProcessFInish 1"   // T143
      := "AutoProcessData".B_Press1.PartStatus = 255;
   END_TRANSITION
   STEP PartStatus_1:   // S137, max time T#10S, warning time T#7S
              N    "AutoProcessData".B_Press1.PartStatus:=250
   END_STEP
   TRANSITION Trans128 FROM PartStatus_1 TO WaitPressFinish   // T128
      := TRUE;
   END_TRANSITION
   STEP CheckPressSensor:   // S138, max time T#10S, warning time T#7S
   END_STEP
   TRANSITION Trans129 FROM CheckPressSensor TO PartStatus_1   // T129
      := "DB_maXYmosNC1".InputMessages.StatusBits."O-UNI" = 1;
   END_TRANSITION
   STEP ResetPressStart:   // S142, max time T#10S, warning time T#7S
              R    "DB_maXYmosNC1".StartCycle
   END_STEP
   TRANSITION Trans133 FROM ResetPressStart TO CheckPressResult   // T133
      := TRUE;
   END_TRANSITION
   STEP CheckPressProgram:   // S139, max time T#10S, warning time T#7S
              N    "AutoProcessData".B_Press1.Press1Program:="DB_maXYmosNC1".InputMessages.StatusBits.MP
   END_STEP
   TRANSITION Trans130 FROM CheckPressProgram TO StartCycle   // T130
      := "DB_maXYmosNC1".InputMessages.StatusBits.MP <> 0;
   END_TRANSITION
   STEP StartCycle:   // S141, max time T#10S, warning time T#7S
              S    "DB_maXYmosNC1".StartCycle
   END_STEP
   TRANSITION Trans132 FROM StartCycle TO CheckPressSensor   // T132
      := ("DB_maXYmosNC1".InputMessages.StatusBits.UNI = 0) AND NOT "DB_maXYmosNC1".oRdyCmd AND "DB_maXYmosNC1".oRunSeq;
   END_TRANSITION
   STEP CheckPressReady:   // S208, max time T#10S, warning time T#7S
              R    "DB_maXYmosNC1".StartCycle
   END_STEP
   TRANSITION Trans211 FROM CheckPressReady TO CheckPressProgram   // T211
      := "DB_maXYmosNC1".InputMessages.StatusBits.READY AND "DB_maXYmosNC1".InputMessages.StatusBits."DRIVE-ENABLED" AND "ProcessData_1"."OP40.2".Kistler_Interlock;
   END_TRANSITION
   STEP "ProcessFInish 1":   // S143, max time T#10S, warning time T#7S
   END_STEP
   TRANSITION Trans134 FROM "ProcessFInish 1" TO Step400   // T134, jump
      := TRUE;
   END_TRANSITION
   STEP ResultOKData:   // S145, max time T#10S, warning time T#7S
              N    "AutoProcessData".B_Press1.PartStatus:=280
   END_STEP
   TRANSITION Trans136 FROM ResultOKData TO Step147   // T136
      := "AutoProcessData".B_Press1.PartStatus = 280;
   END_TRANSITION
   STEP CheckPressResult:   // S144, max time T#10S, warning time T#7S
   END_STEP
   TRANSITION Trans135 FROM CheckPressResult TO ResultOKData   // T135
      := "DB_maXYmosNC1".oCycleOK AND NOT "DB_maXYmosNC1".oCycleNOK;
   END_TRANSITION
   TRANSITION Trans142 FROM CheckPressResult TO ResultNGData   // T142
      := NOT "DB_maXYmosNC1".oCycleOK AND "DB_maXYmosNC1".oCycleNOK;
   END_TRANSITION
   STEP Step147:   // S147, max time T#10S, warning time T#7S
   END_STEP
   TRANSITION Trans144 FROM Step147 TO "ProcessFInish 1"   // T144
      := TRUE;
   END_TRANSITION

   // sequencer 5: S400-S499OK&NG数据处理 / S400-S499OK&NG Status Count
   STEP Step400:   // S400, max time T#10S, warning time T#7S
   END_STEP
   TRANSITION Trans224 FROM Step400 TO JudgeStatus   // T400
      := TRUE;
   END_TRANSITION
   STEP JudgeStatus:   // S401, max time T#10S, warning time T#7S
              N    #ioPM_Inface.ProcessResult:=0
   END_STEP
   TRANSITION OK FROM JudgeStatus TO OKCount   // T401
      := #ioStatus = 190;
   END_TRANSITION
   TRANSITION NG FROM JudgeStatus TO NGCount   // T404
      := #ioStatus <> 190;
   END_TRANSITION
   STEP OKCount:   // S402, max time T#10S, warning time T#7S
              N    #ioPM_Inface.ProcessResult:=400
   END_STEP
   TRANSITION Trans403 FROM OKCount TO ProcessFinish   // T402
      := TRUE;
   END_TRANSITION
   STEP NGCount:   // S404, max time T#10S, warning time T#7S
              N    #ioPM_Inface.ProcessResult:=#ioStatus
   END_STEP
   TRANSITION Trans404 FROM NGCount TO ProcessFinish   // T405
      := TRUE;
   END_TRANSITION
   STEP ProcessFinish:   // S403, max time T#10S, warning time T#7S
   END_STEP
   TRANSITION Trans405 FROM ProcessFinish TO "MES Result"   // T403, jump
      := TRUE;
   END_TRANSITION

   // sequencer 6: S500-S599 MES上传RFID写入 / S500-S599 MES Result
   STEP "MES Result":   // S500, max time T#10S, warning time T#7S
   END_STEP
   TRANSITION Trans162 FROM "MES Result" TO Bypass_1   // T158
      := TRUE;
   END_TRANSITION
   STEP "MES Result OK_1":   // S399, max time T#10S, warning time T#7S
              N    "AutoProcessData".B_Press1.PartStatus:=299
   END_STEP
   TRANSITION Trans312 FROM "MES Result OK_1" TO "MES Check Finish"   // T399
      := "AutoProcessData".B_Press1.PartStatus = 299;
   END_TRANSITION
   STEP "Prepare MES CheckData_1":   // S307, max time T#10S, warning time T#7S
   END_STEP
   TRANSITION Trans16 FROM "Prepare MES CheckData_1" TO MesCheckResult   // T308
      := #"Prepare MES CheckData_1".T > t#300MS;
   END_TRANSITION
   STEP "MES Check Finish":   // S599, max time T#10S, warning time T#7S
   END_STEP
   TRANSITION Trans619 FROM "MES Check Finish" TO RobotPick   // T599, jump
      := TRUE;
   END_TRANSITION
   STEP "MES Check NG_1":   // S310, max time T#10S, warning time T#7S
              N    "AutoProcessData".B_Press1.PartStatus:=252
   END_STEP
   TRANSITION Trans310 FROM "MES Check NG_1" TO "MES Check Finish"   // T313
      := "AutoProcessData".B_Press1.PartStatus = 252;
   END_TRANSITION
   STEP MesCheckResult:   // S309, max time T#10S, warning time T#7S
              N    "PLCtoMES"."PLC.Unload_Station3DataSaveReq"
   END_STEP
   TRANSITION Trans308 FROM MesCheckResult TO "MES Result OK_1"   // T310
      := "MEStoPLC"."MES.Unload_ResultsStored3OK" AND NOT "MEStoPLC"."MES.Unload_ResultsStored3NG" AND "MEStoPLC"."MES.Unload_ResultsStored3ReqMesDone" AND ("AutoProcessData".B_Press1.PartStatus = 280);
   END_TRANSITION
   TRANSITION Trans309 FROM MesCheckResult TO "MES Check NG_1"   // T312
      := NOT "MEStoPLC"."MES.Unload_ResultsStored3OK" AND "MEStoPLC"."MES.Unload_ResultsStored3NG" AND "MEStoPLC"."MES.Unload_ResultsStored3ReqMesDone";
   END_TRANSITION
   TRANSITION Trans313 FROM MesCheckResult TO MESOverTime   // T318
      := NOT "MEStoPLC"."MES.Load_Station7ReqMesDone" AND (#MesCheckResult.T > t#10S);
   END_TRANSITION
   TRANSITION Trans140 FROM MesCheckResult TO "MES Check Finish"   // T138
      := "MEStoPLC"."MES.Unload_ResultsStored3OK" AND NOT "MEStoPLC"."MES.Unload_ResultsStored3NG" AND "MEStoPLC"."MES.Unload_ResultsStored3ReqMesDone" AND ("AutoProcessData".B_Press1.PartStatus <> 280);
   END_TRANSITION
   STEP Bypass_1:   // S314, max time T#10S, warning time T#7S
   END_STEP
   TRANSITION Online_1 FROM Bypass_1 TO ResetMesUnloadRequest_1   // T311
      := NOT "Station_Sys".Cmd.OnOffLine;
   END_TRANSITION
   TRANSITION Trans320 FROM Bypass_1 TO ok_1   // T320
      := "Station_Sys".Cmd.OnOffLine;
   END_TRANSITION
   STEP ResetMesUnloadRequest_1:   // S302, max time T#10S, warning time T#7S
              R    "PLCtoMES"."PLC.Unload_Station3DataSaveReq"
              R    "MEStoPLC"."MES.Unload_ResultsStored3OK"
              R    "MEStoPLC"."MES.Unload_ResultsStored3NG"
              R    "MEStoPLC"."MES.Unload_ResultsStored3ReqMesDone"
   END_STEP
   TRANSITION Trans260 FROM ResetMesUnloadRequest_1 TO "Prepare MES CheckData_1"   // T314
      := NOT "PLCtoMES"."PLC.Unload_Station3DataSaveReq" AND NOT "MEStoPLC"."MES.Unload_ResultsStored3OK" AND NOT "MEStoPLC"."MES.Unload_ResultsStored3NG" AND NOT "MEStoPLC"."MES.Unload_ResultsStored3ReqMesDone";
   END_TRANSITION
   STEP Step314:   // S316, max time T#10S, warning time T#7S
   END_STEP
   TRANSITION Trans321 FROM Step314 TO "MES Check Finish"   // T321
      := TRUE;
   END_TRANSITION
   STEP MESOverTime:   // S315, max time T#10S, warning time T#7S
              S    "ST10_DeviceError".MES_Error.CheckInResultOverTime_3
   END_STEP
   TRANSITION Trans318 FROM MESOverTime TO Bypass_1   // T319, jump
      := #iSysInface.Reset;
   END_TRANSITION
   STEP ok_1:   // S317, max time T#10S, warning time T#7S
      interlock C := "AutoProcessData".B_Press1.PartStatus = 280;
      (C)     N    "AutoProcessData".B_Press1.PartStatus:=299
   END_STEP
   TRANSITION Trans317 FROM ok_1 TO Step314   // T322
      := ("AutoProcessData".B_Press1.PartStatus = 199) OR ("Station_Sys".Cmd.OnOffLine AND ("AutoProcessData".B_Press1.PartStatus <> 150) AND ("AutoProcessData".B_Press1.PartStatus <> 155));
   END_TRANSITION

   // sequencer 7: S600-S699工件放行 / S600-S699 RobotPick
   STEP RobotPick:   // S600, max time T#10S, warning time T#7S
              S    #ioPM_Inface.ProcessComplete
              R    #ioPM_Inface.ProcessStart
   END_STEP
   TRANSITION Trans600 FROM RobotPick TO PressProgram_1   // T600
      := TRUE;
   END_TRANSITION
   STEP ProcessFinsh:   // S605, max time T#10S, warning time T#7S: 正式使用时，需要激活复位空循环
   END_STEP
   TRANSITION Trans699 FROM ProcessFinsh TO ProcessStart   // T605, jump
      := TRUE;
   END_TRANSITION
   STEP DataClear:   // S604, max time T#10S, warning time T#7S
          S1  N    #ioPM_Inface.ProcessResult:=0
          S1  N    #ioStatus:=0
   END_STEP
   TRANSITION Trans290 FROM DataClear TO ProcessFinsh   // T604
      := TRUE;
   END_TRANSITION
   STEP "Request robot pick":   // S408, max time T#10S, warning time T#7S
              N    "AutoProcessControl".B_Press_1.Robot1PickPrimit
   END_STEP
   TRANSITION Trans412 FROM "Request robot pick" TO "Wait robot finish task"   // T410
      := "KukaRobot1_CtrlDB".sROBtoPLC.User.Cycle.DO281_PressPickInside AND NOT "KukaRobot1_CtrlDB".sROBtoPLC.User.Cycle.DO282_PressPickFinish;
   END_TRANSITION
   STEP "Wait robot finish task":   // S131, max time T#10S, warning time T#7S
   END_STEP
   TRANSITION Trans257 FROM "Wait robot finish task" TO DataMove   // T256
      := "KukaRobot1_CtrlDB".sROBtoPLC.User.Cycle.DO282_PressPickFinish;
   END_TRANSITION
   STEP DataMove:   // S132, max time T#10S, warning time T#7S
   END_STEP
   TRANSITION Trans258 FROM DataMove TO "Wait robot in safety area"   // T257
      := TRUE;
   END_TRANSITION
   STEP "Wait robot in safety area":   // S133, max time T#10S, warning time T#7S
   END_STEP
   TRANSITION Trans261 FROM "Wait robot in safety area" TO DataClear   // T258
      := "KukaRobot1_CtrlDB".sROBtoPLC.User.Home.DO177_PressPut1Area AND "KukaRobot1_CtrlDB".sROBtoPLC.User.Home.DO178_PressPut2Area;
   END_TRANSITION
   STEP PressProgram_1:   // S20, max time T#10S, warning time T#7S
      interlock C := NOT "ST10_GeneralData".FunctionDeSelect."B".FunctionDeSelected_TestPress372A1;
      (C)     N    "DB_maXYmosNC1".ProgNo:=1
   END_STEP
   TRANSITION Trans31 FROM PressProgram_1 TO "PressReady?_1"   // T27
      := TRUE;
   END_TRANSITION
   STEP PressHoming_1:   // S21, max time T#10S, warning time T#7S
              N    "DB_maXYmosNC1".Homing
   END_STEP
   TRANSITION Trans9 FROM PressHoming_1 TO Step15   // T26
      := "DB_maXYmosNC1".oInHomePos;
   END_TRANSITION
   STEP "PressReady?_1":   // S22, max time T#10S, warning time T#7S
   END_STEP
   TRANSITION Trans32 FROM "PressReady?_1" TO "PressHoming?_1"   // T28
      := "DB_maXYmosNC1".oReady AND "DB_maXYmosNC1".oRdyAmp;
   END_TRANSITION
   STEP "PressHoming?_1":   // S23, max time T#10S, warning time T#7S
   END_STEP
   TRANSITION Trans33 FROM "PressHoming?_1" TO PressHoming_1   // T29
      := NOT "DB_maXYmosNC1".oInHomePos;
   END_TRANSITION
   TRANSITION Trans34 FROM "PressHoming?_1" TO Step15   // T30
      := "DB_maXYmosNC1".oInHomePos;
   END_TRANSITION
   STEP Step15:   // S24, max time T#10S, warning time T#7S
   END_STEP
   TRANSITION Trans35 FROM Step15 TO "B-PressFitting-01CylinderToHP_1"   // T31
      := TRUE;
   END_TRANSITION
   STEP "B-PressFitting-01CylinderToHP_1":   // S140, max time T#10S, warning time T#7S
              S    "ST10Cylinder".Cy[6].Inout.AutoGoHome
              R    "ST10Cylinder".Cy[6].Inout.AutoGoWork
   END_STEP
   TRANSITION Trans768 FROM "B-PressFitting-01CylinderToHP_1" TO "Request robot pick"   // T131
      := NOT "ST10Cylinder".Cy[6].In.WorkPositionSensor AND "ST10Cylinder".Cy[6].In.HomePositionSensor;
   END_TRANSITION

   // permanent post-instructions
   NETWORK 1
      #ioPM_Inface.StepNum := #RT_DATA.S_DISPLAY;
   NETWORK 2
      IF #iSysInface.Reset THEN #AlarmID := 0; END_IF;
   NETWORK 3
      #TON[10].TON(IN := #工件放行中, PT := T#0.5S);
      IF #TON[10].Q THEN #工件放行中 := FALSE; END_IF;
END_FUNCTION_BLOCK

FUNCTION_BLOCK "ST10_Flow5_FRobot_1"   // FB1075, GRAPH
// stored: AcknowledgeErrorsRequired false, AutoNumber false, GraphVersion 6.0, InitialValuesAcquisition false, SetENOAutomatically false
   // inherited from GRAPH_BASE
   VAR_INPUT
      iSysInface : "RCS_SysComInterface_V1";
   END_VAR
   VAR_IN_OUT
      ioPM_Inface : "RCS_PMInterface_V1";
      ioStatus : Int;
   END_VAR
   VAR
      sCtrlMode { S7_SetPoint := 'True'} : "SysFlowCtrlGraph";
      sUpdMES_Data : Bool;   // 更新MES数据
      工件放行中 : Bool;
      前站站号 { ExternalAccessible := 'False'; ExternalVisible := 'False'; ExternalWritable := 'False'} : UInt;
      本站站号 { ExternalAccessible := 'False'; ExternalVisible := 'False'; ExternalWritable := 'False'} : UInt;
      弹窗Temp : Array[1..10] of Int;
      AlarmID : Int;
      TON { S7_SetPoint := 'True'} : Array[0..10] of TON_TIME;
      TOF { S7_SetPoint := 'True'} : Array[0..10] of TOF_TIME;
      sUP { S7_SetPoint := 'True'} : Array[0..10] of Bool;
      更新RFID完成 : Bool;
   END_VAR
   VAR_TEMP
      Tempresult : USInt;
      本站站号乘10 : UInt;
   END_VAR
   // // TON[0] : 托盘流入1托盘到位传感器
   // // TON[1] : 托盘流入1托盘到位传感器
   // // TON[2] : 托盘流入1产品有无传感器
   // // TON[3] : 托盘流入1产品有无传感器
   // // TON[4] : 托盘流入1姿态检测光电2
   // // TON[5] : 托盘流入1姿态检测光电3
   // // TON[0].Q : 托盘流入1托盘到位
   // // TON[1].Q : 托盘流入1托盘无
   // // TON[2].Q : 托盘流入1有产品
   // // TON[3].Q : 托盘流入1无产品
   // // TON[4].Q : 托盘流入1姿态检测光电2
   // // TON[5].Q : 托盘流入1姿态检测光电3
BEGIN
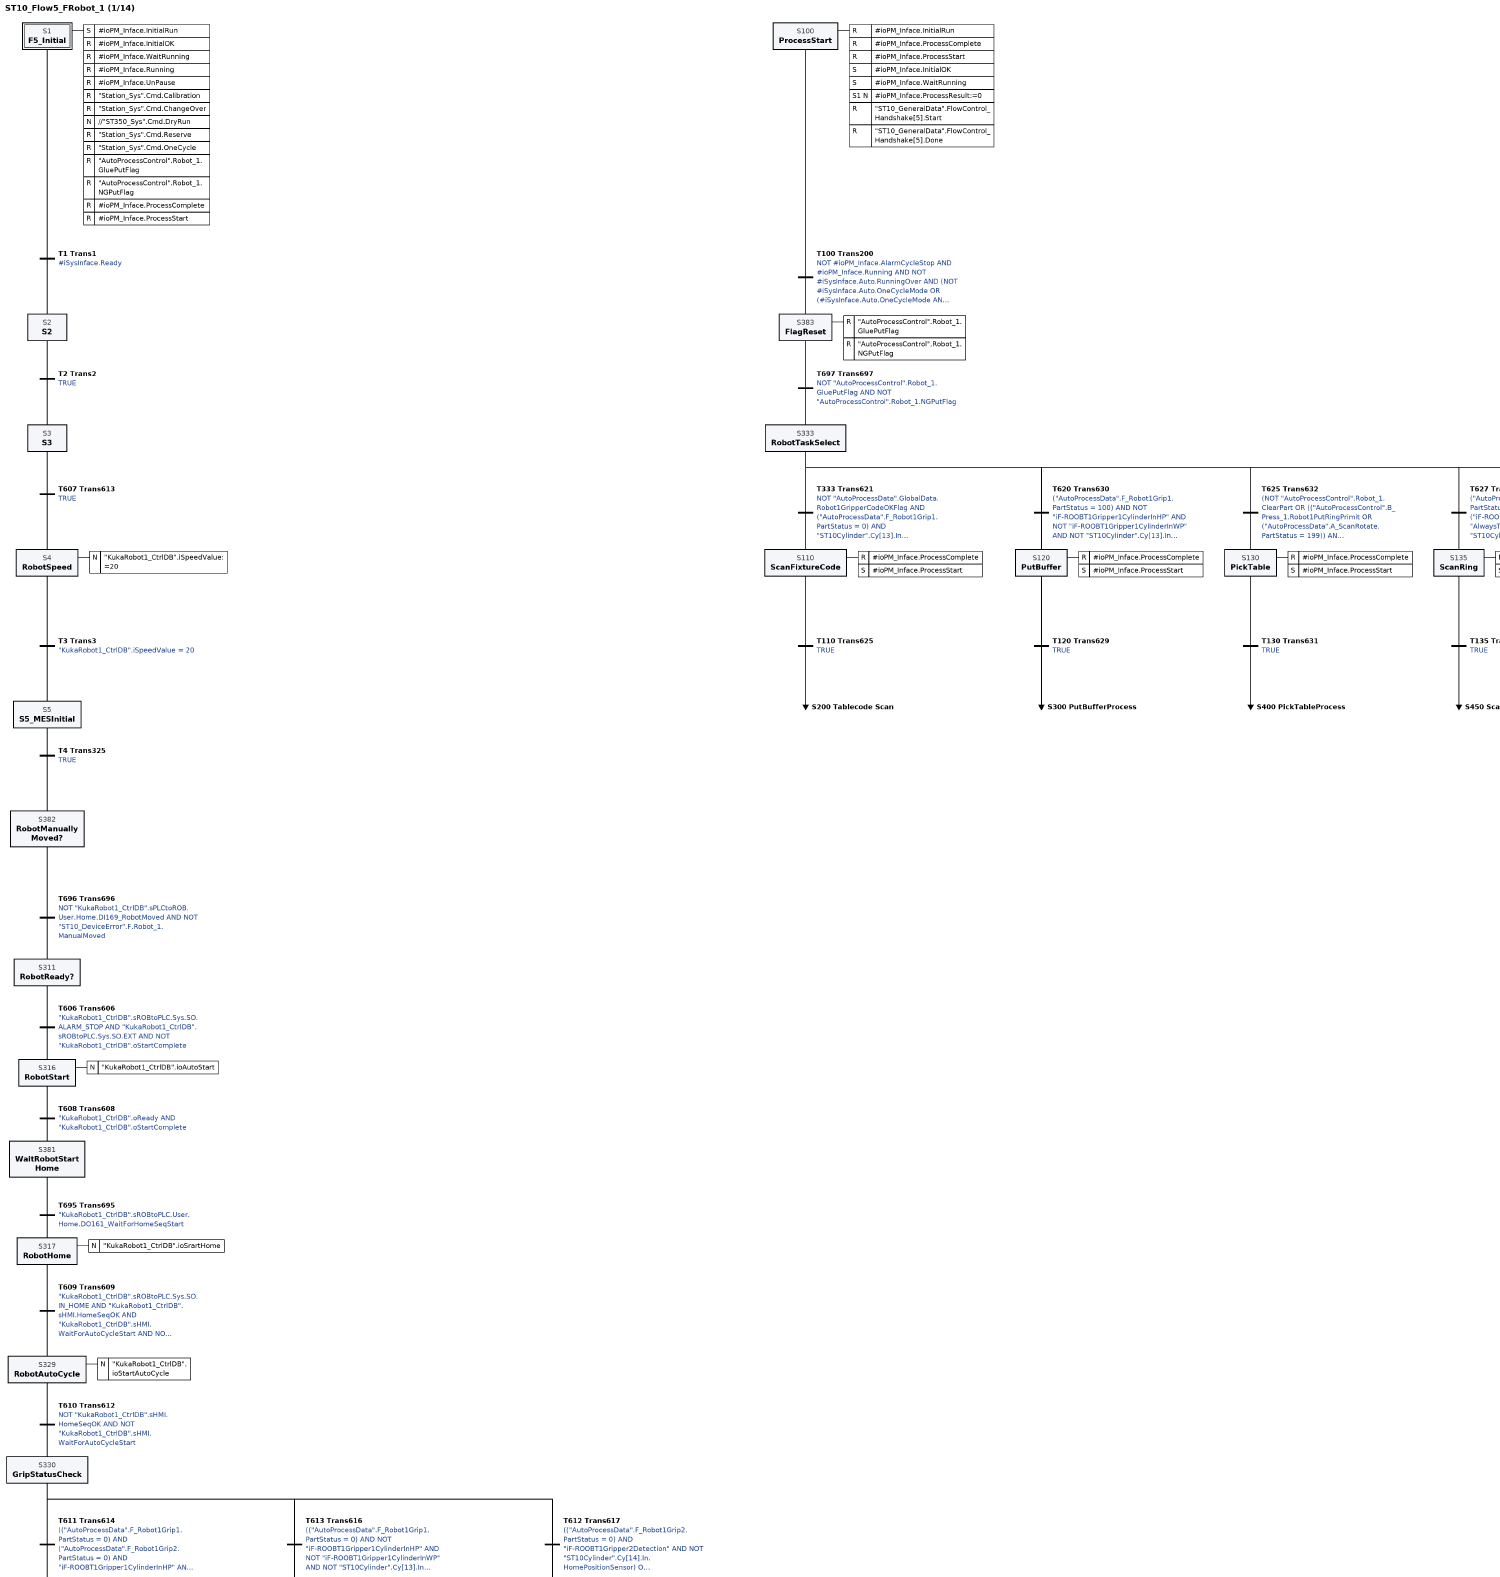
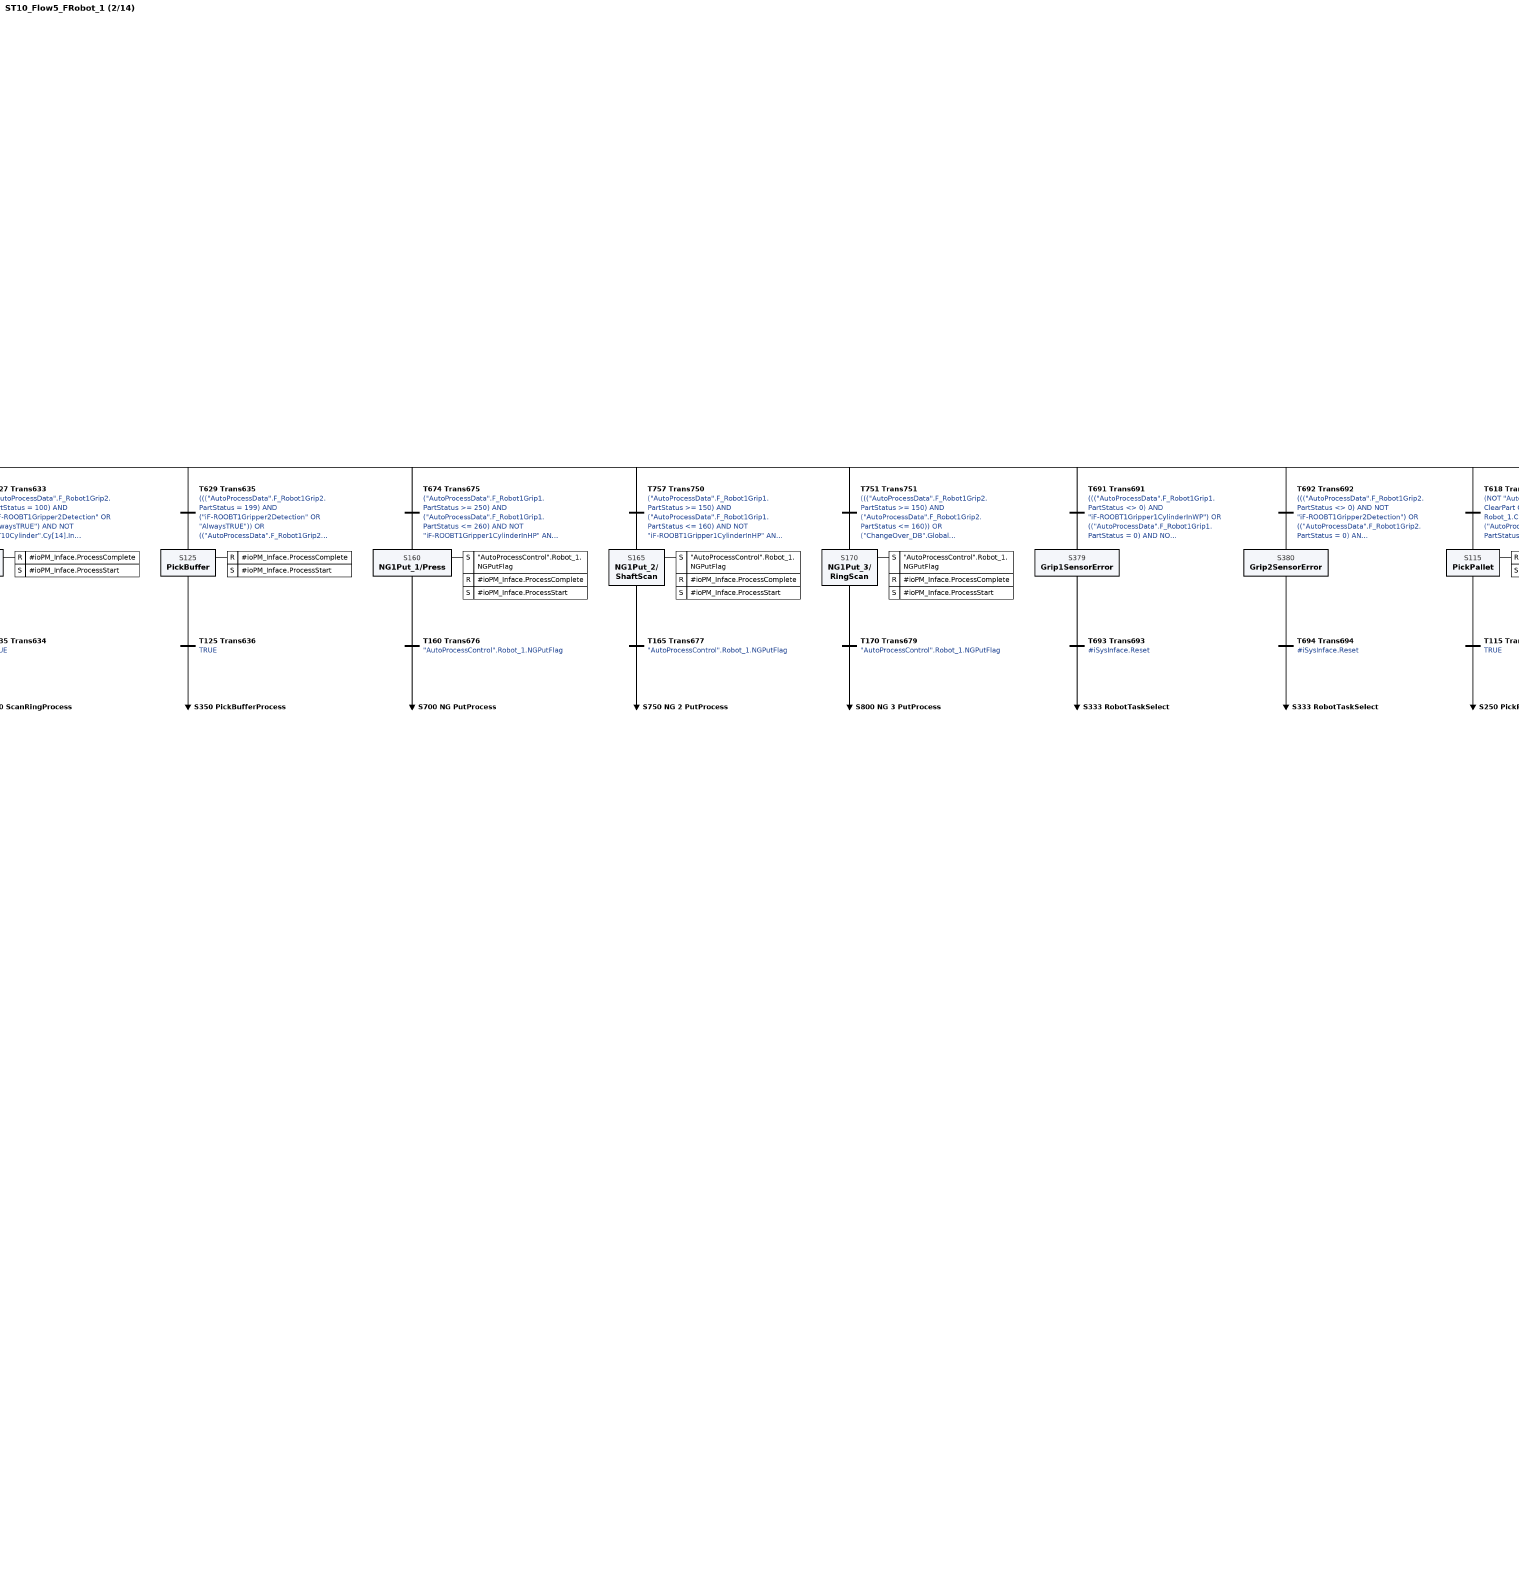
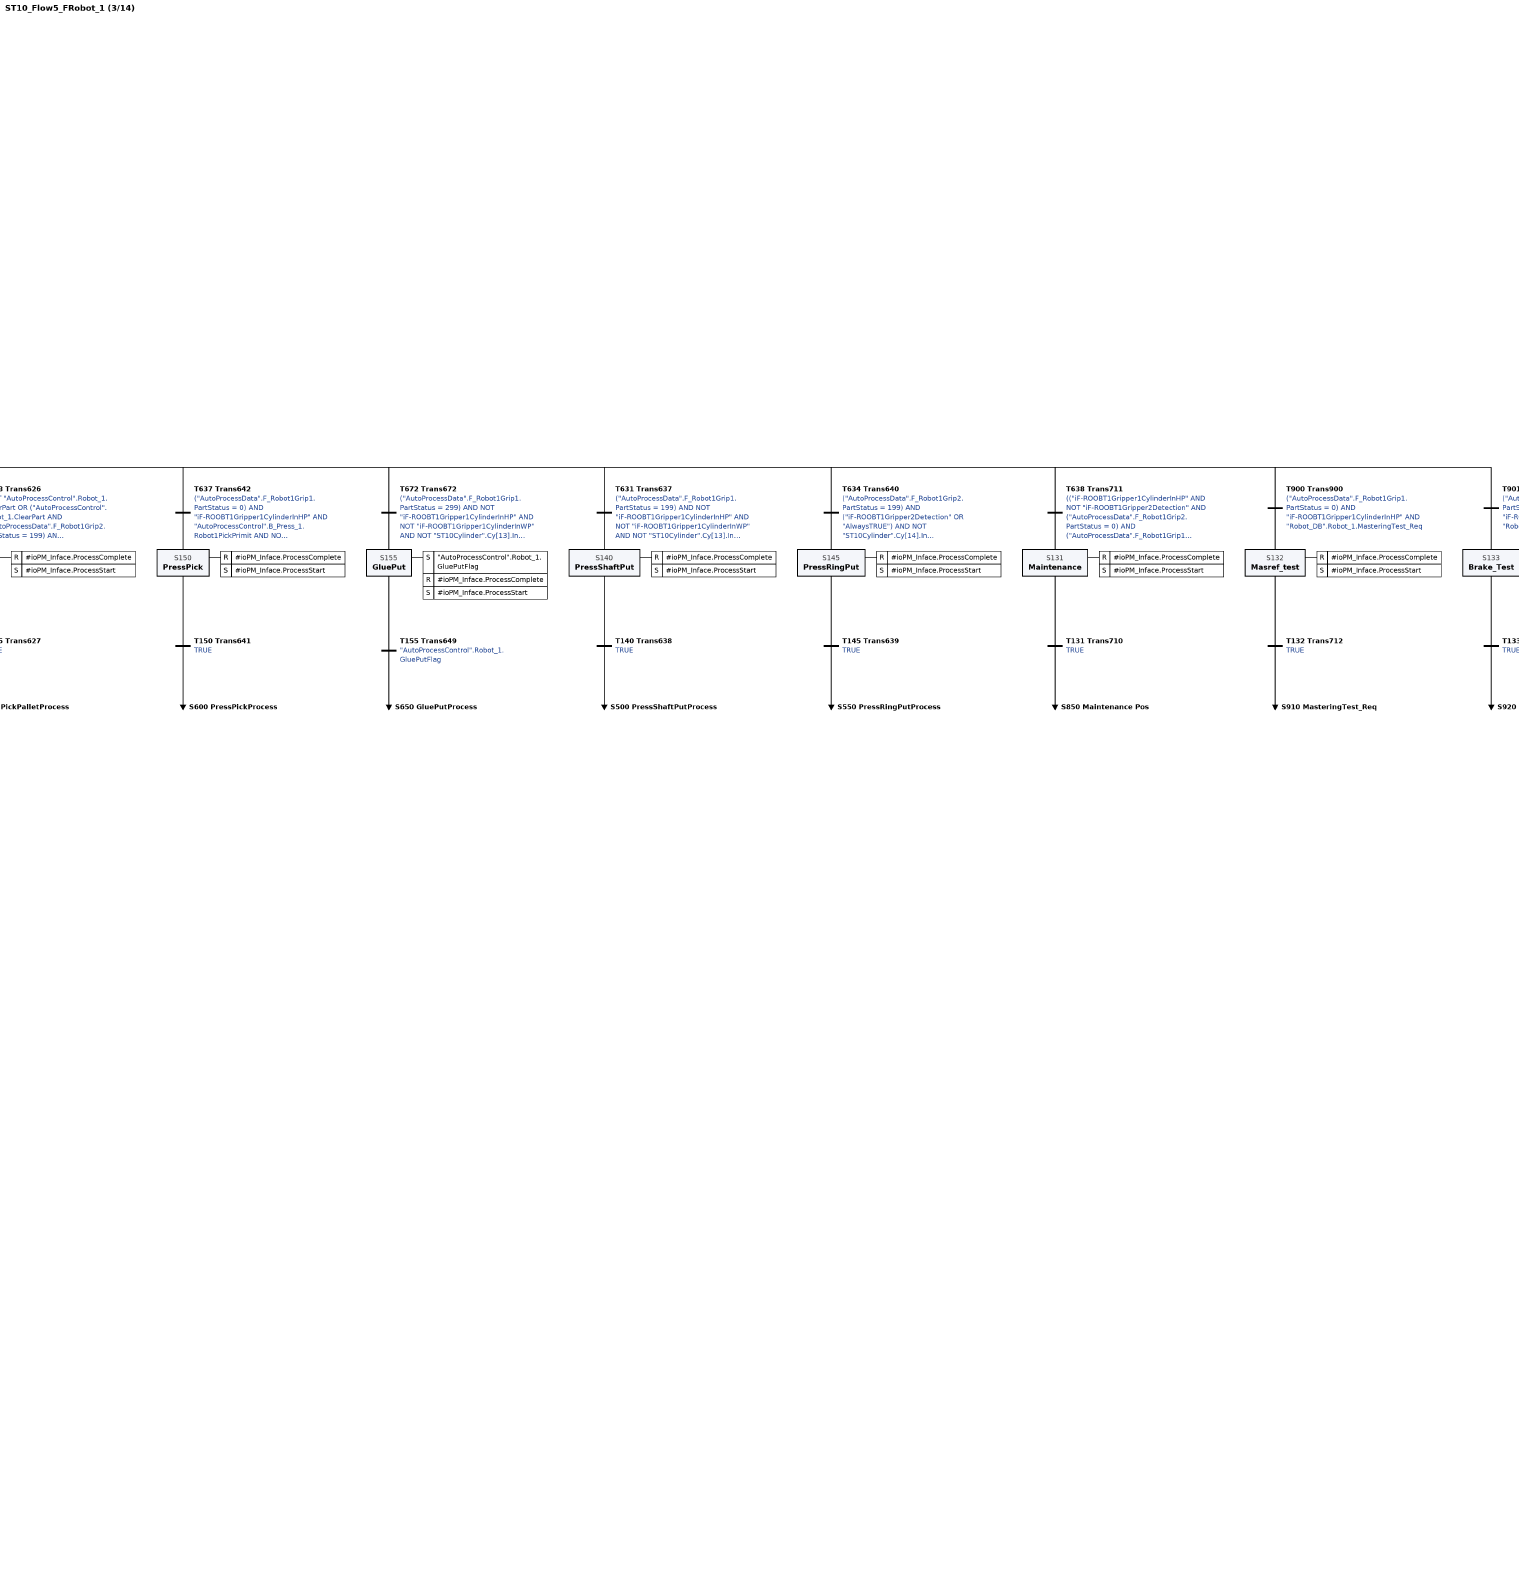
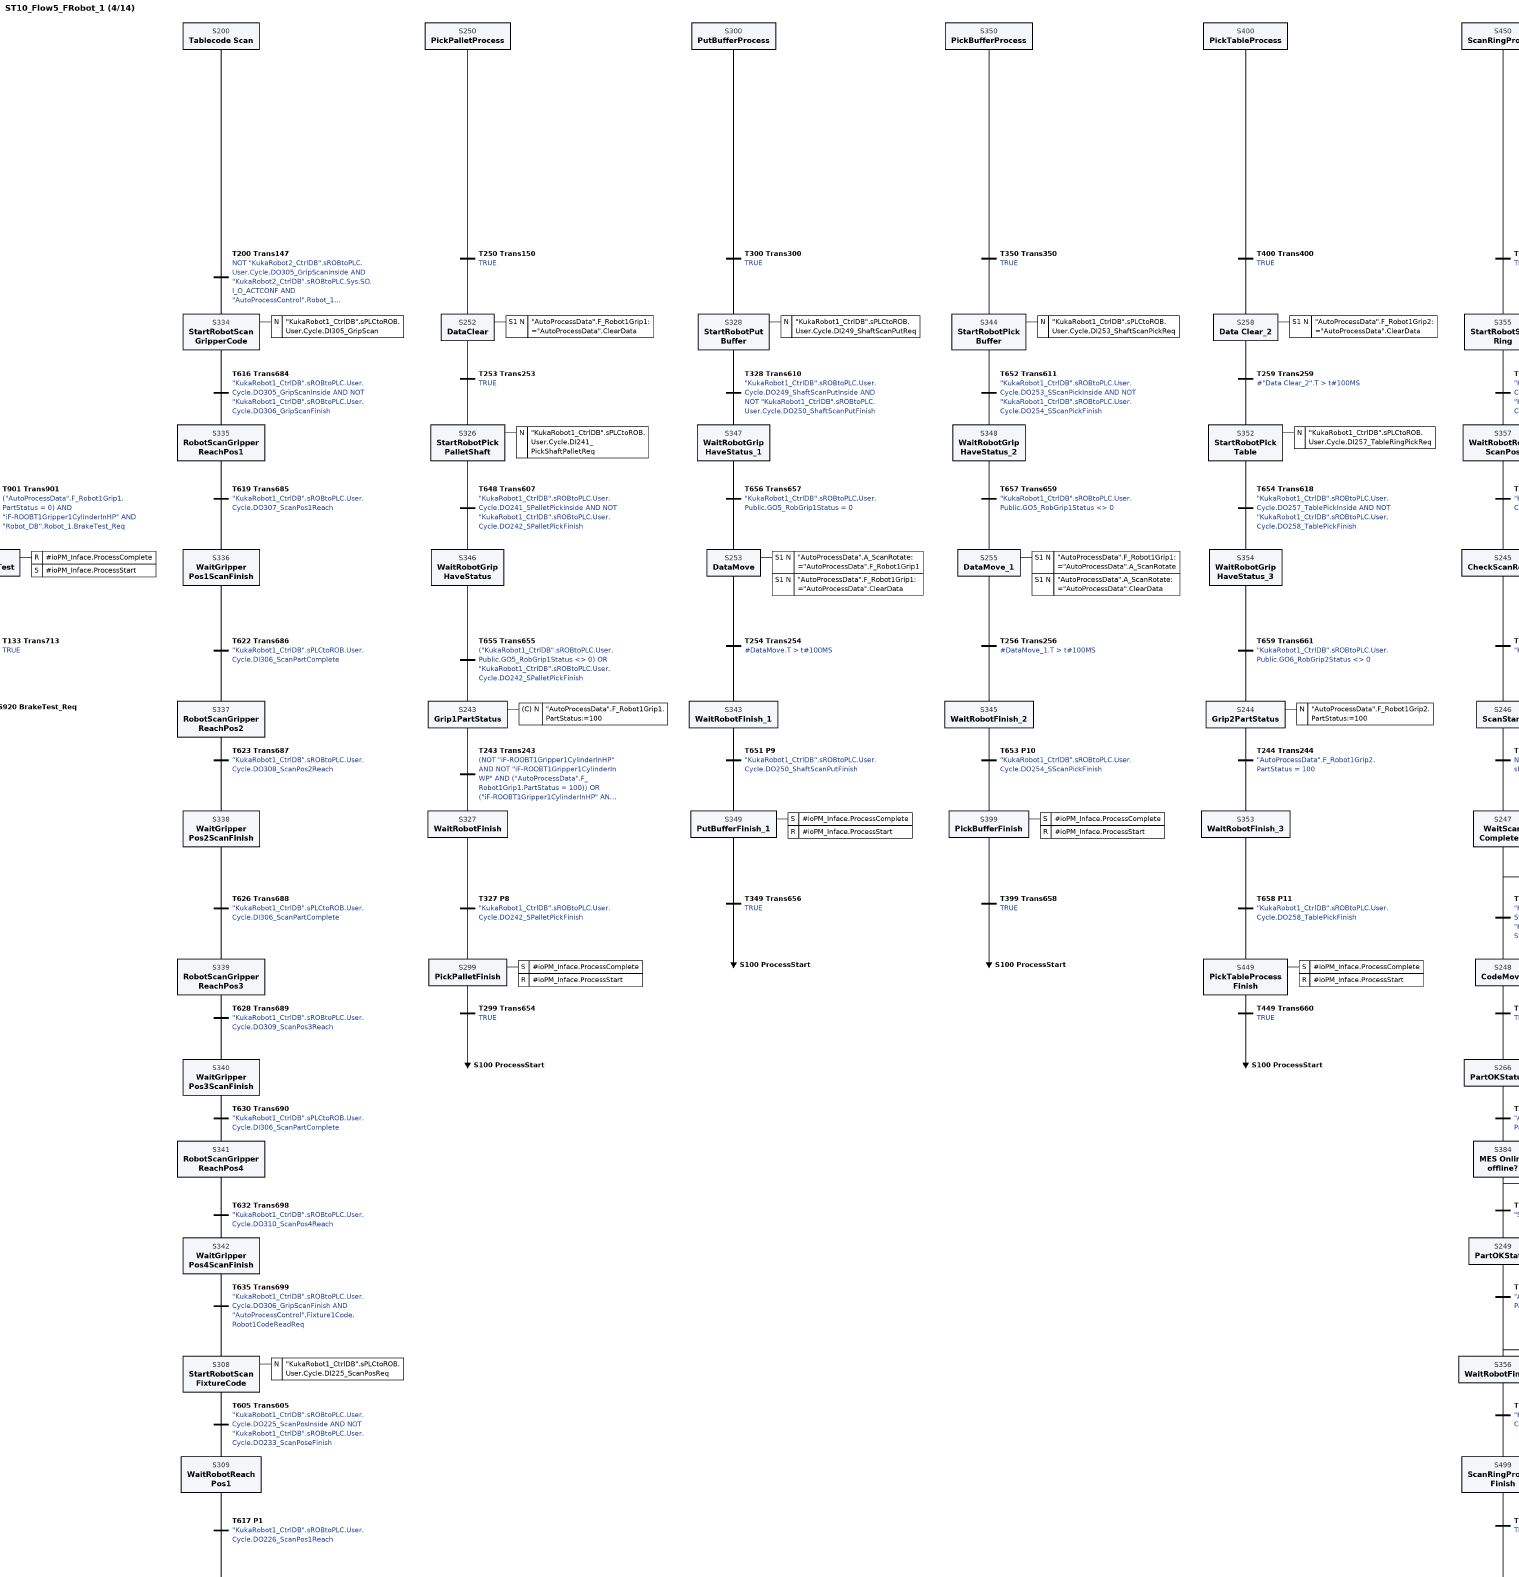
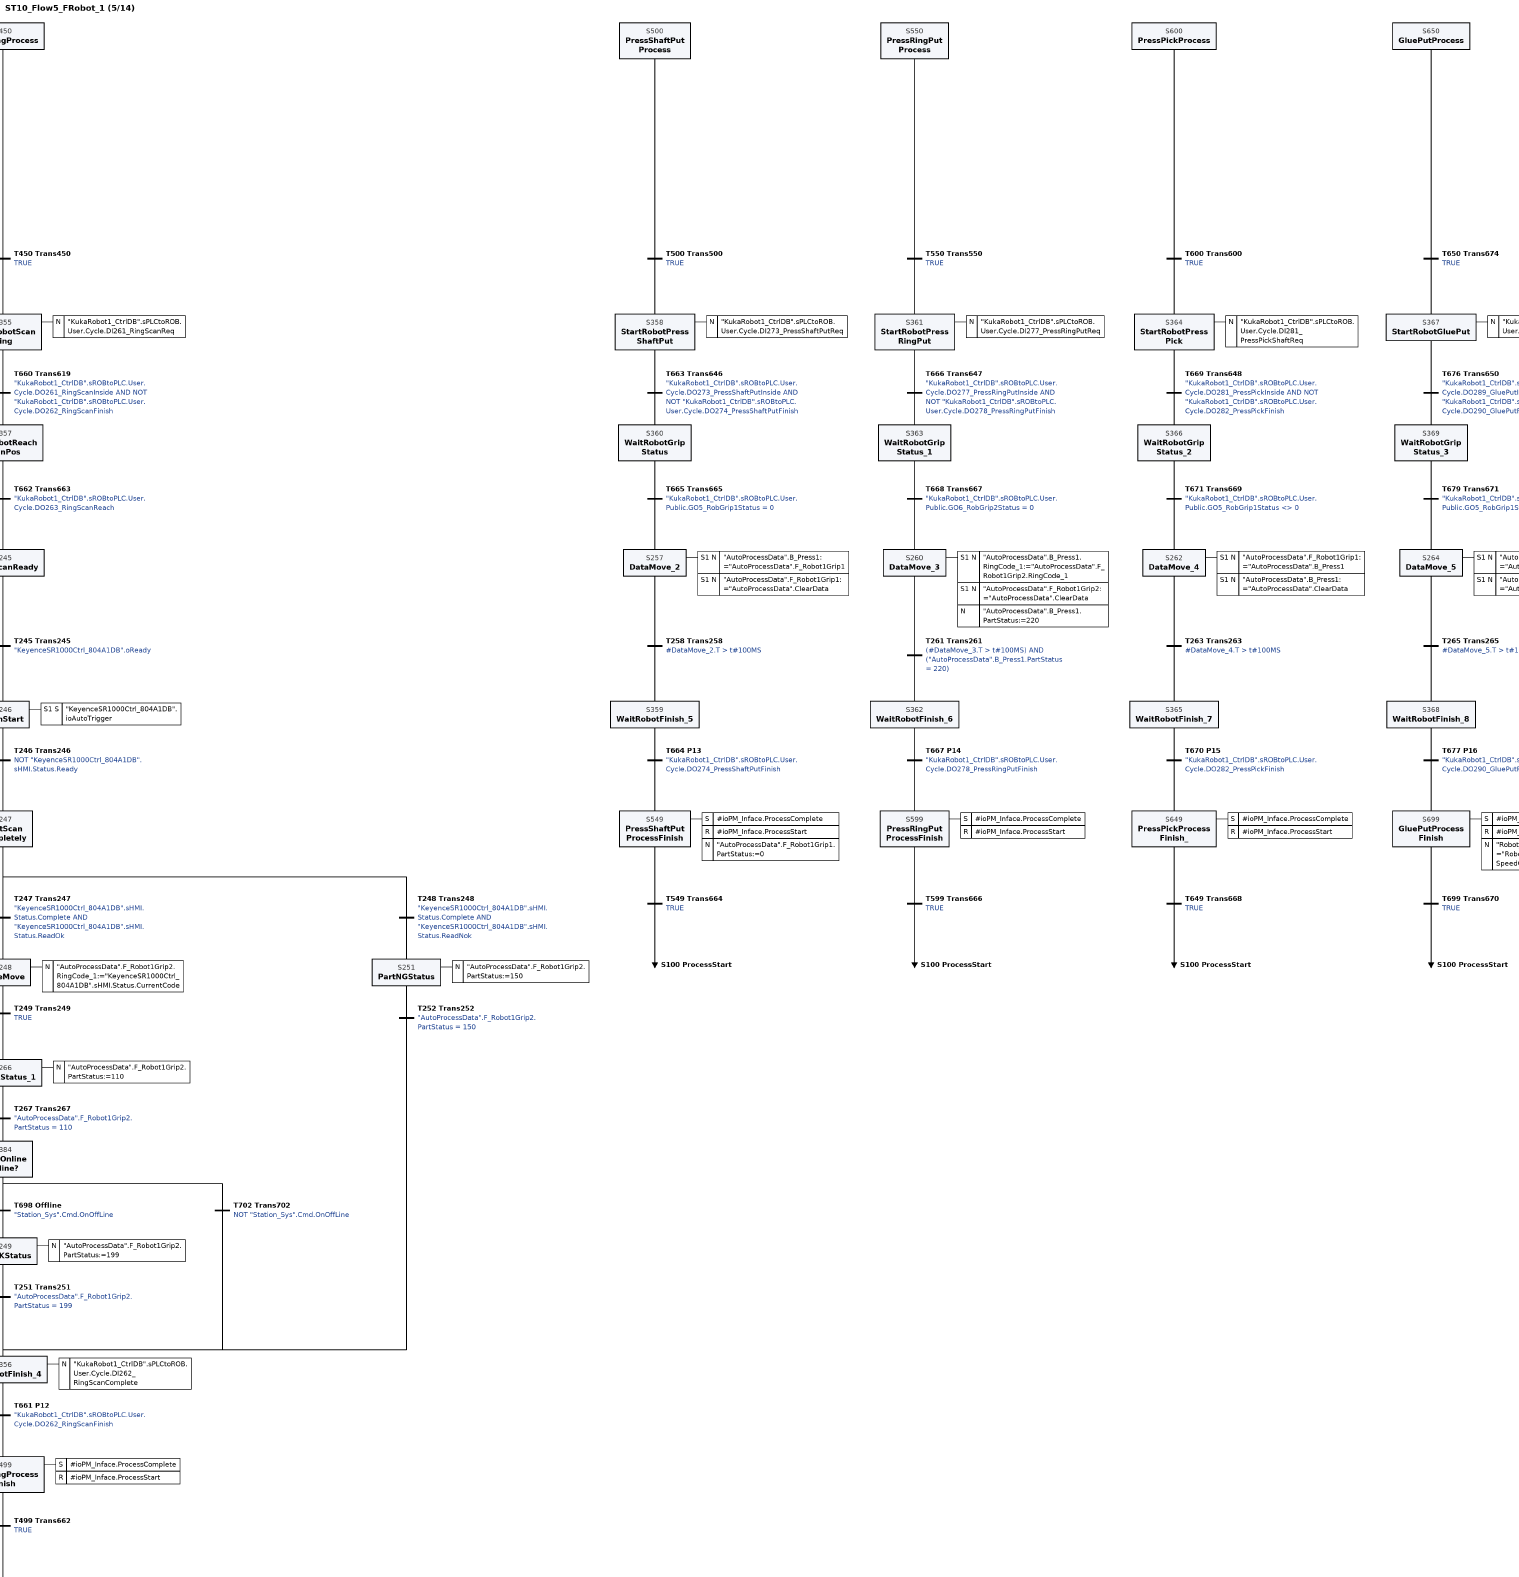
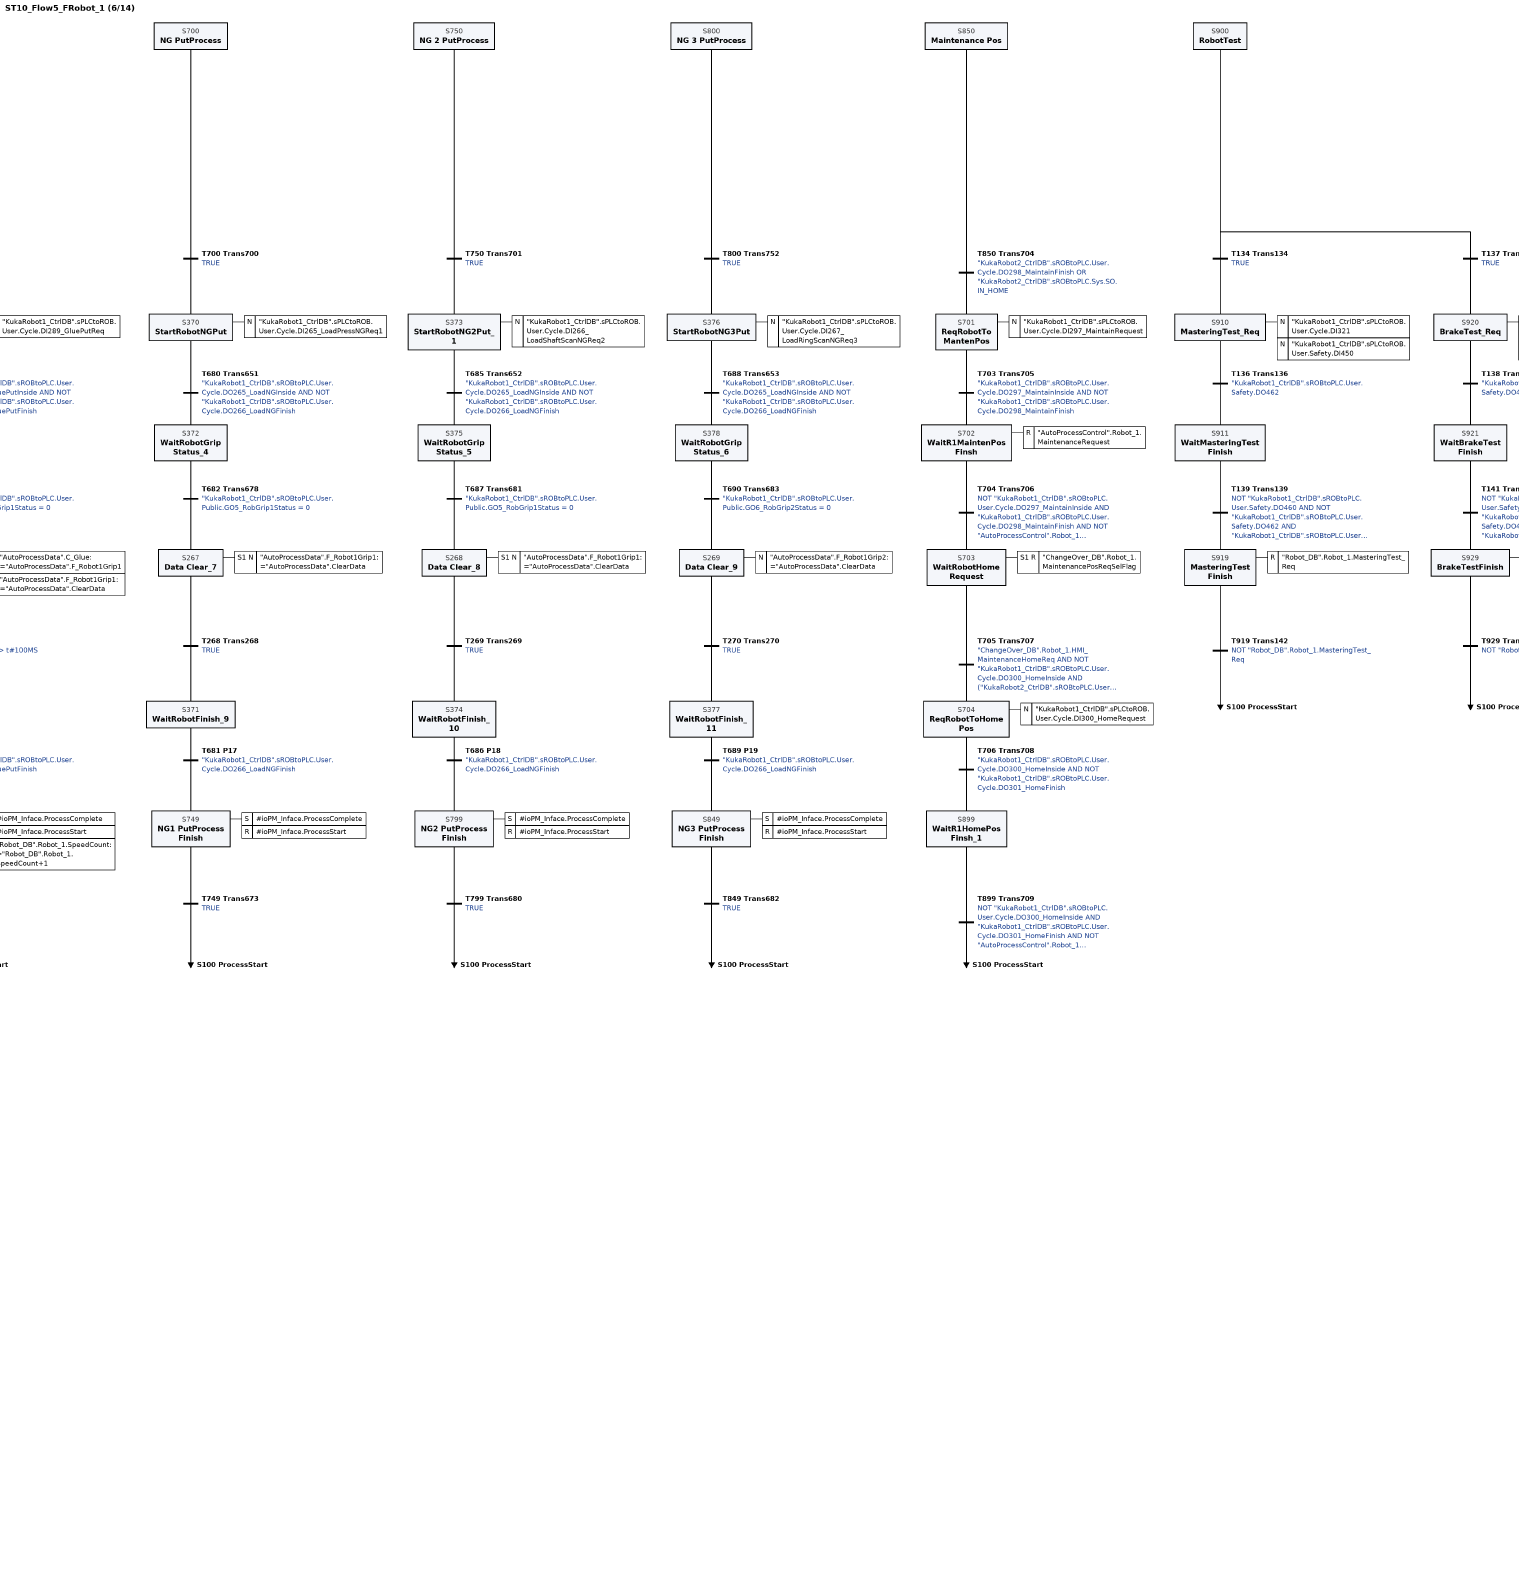
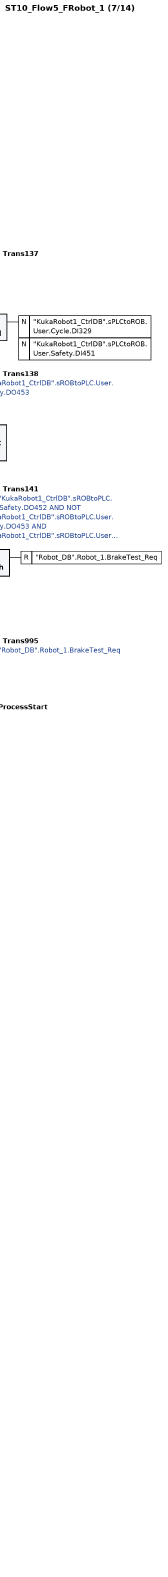
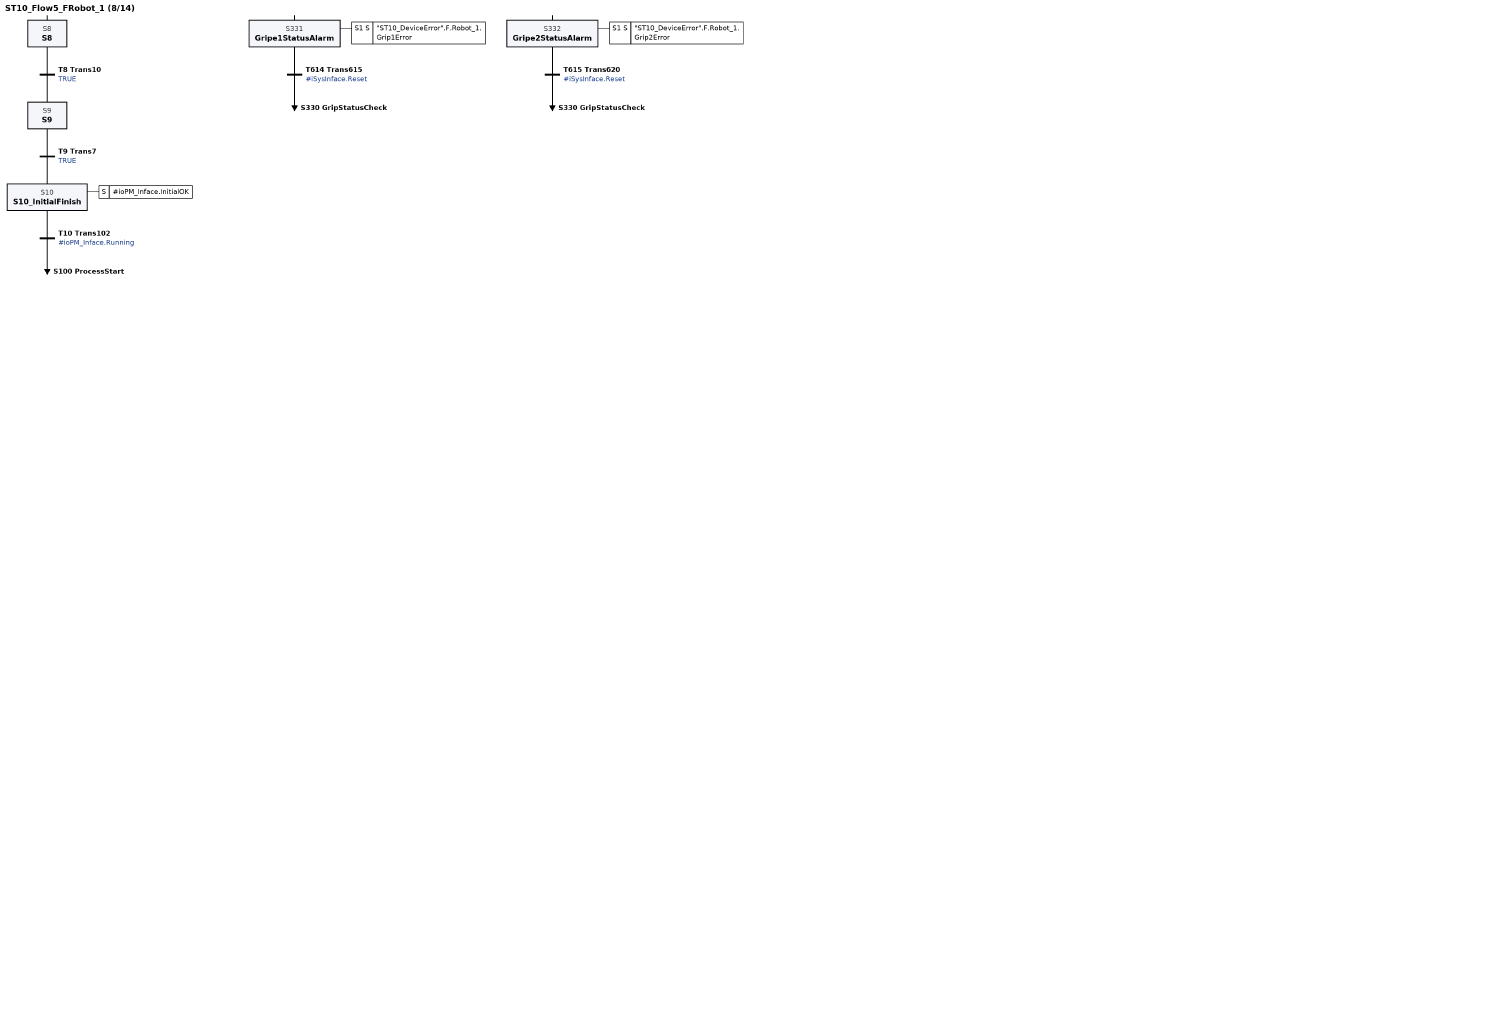
